REGION Network 198: Step[3048] : Pad Top Left/Right Vacc Off
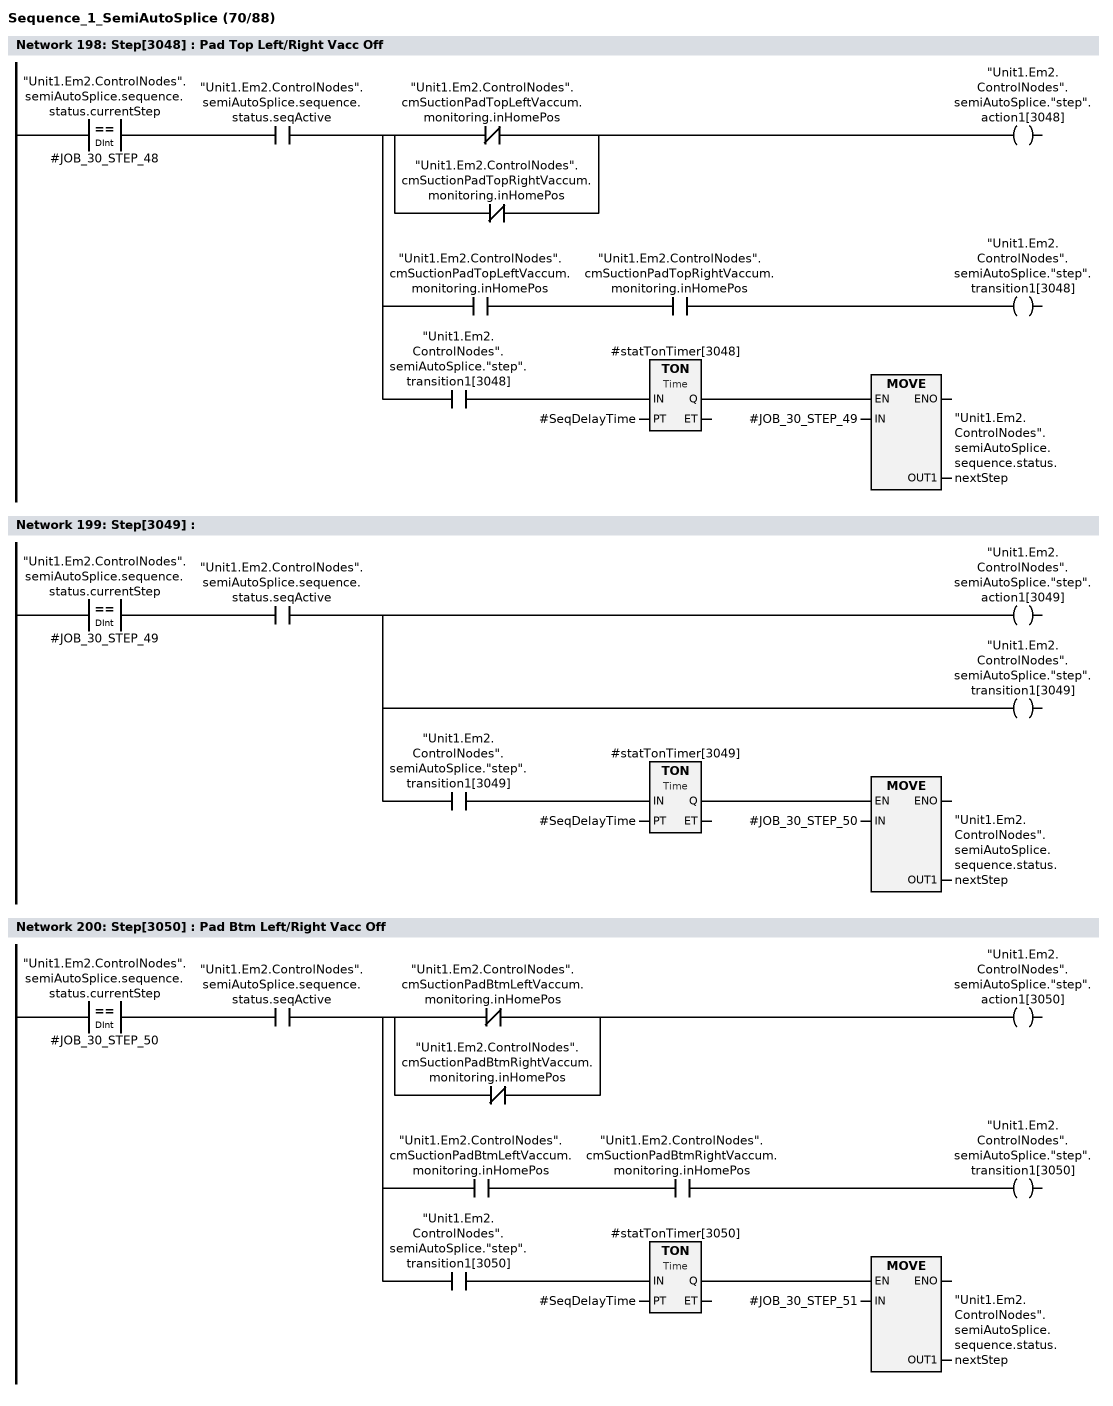
   RUNG wire#powerrail
      { S7_Templates := "SrcType := DInt" } EQ_Contact(in1 := "Unit1.Em2.ControlNodes".semiAutoSplice.sequence.status.currentStep, in2 := #JOB_30_STEP_48)
      Contact( "Unit1.Em2.ControlNodes".semiAutoSplice.sequence.status.seqActive )
      wire#w1
      I_Contact( "Unit1.Em2.ControlNodes".cmSuctionPadTopLeftVaccum.monitoring.inHomePos )
      wire#w2
      Coil( "Unit1.Em2.ControlNodes".semiAutoSplice."step".action1[3048] )
   END_RUNG
   RUNG wire#w1
      I_Contact( "Unit1.Em2.ControlNodes".cmSuctionPadTopRightVaccum.monitoring.inHomePos )
   END_RUNG wire#w2
   RUNG wire#w1
      Contact( "Unit1.Em2.ControlNodes".cmSuctionPadTopLeftVaccum.monitoring.inHomePos )
      Contact( "Unit1.Em2.ControlNodes".cmSuctionPadTopRightVaccum.monitoring.inHomePos )
      Coil( "Unit1.Em2.ControlNodes".semiAutoSplice."step".transition1[3048] )
   END_RUNG
   RUNG wire#w1
      Contact( "Unit1.Em2.ControlNodes".semiAutoSplice."step".transition1[3048] )
      { S7_Templates := "time_type := Time" } #statTonTimer[3048].TON(pt := #SeqDelayTime, et =>)
      Move(in := #JOB_30_STEP_49, out1 => "Unit1.Em2.ControlNodes".semiAutoSplice.sequence.status.nextStep)
   END_RUNG
   // the same network as SCL:
   #_w1 := ("Unit1.Em2.ControlNodes".semiAutoSplice.sequence.status.currentStep = #JOB_30_STEP_48) AND "Unit1.Em2.ControlNodes".semiAutoSplice.sequence.status.seqActive;
   "Unit1.Em2.ControlNodes".semiAutoSplice."step".action1[3048] := #_w1 AND (NOT "Unit1.Em2.ControlNodes".cmSuctionPadTopLeftVaccum.monitoring.inHomePos OR NOT "Unit1.Em2.ControlNodes".cmSuctionPadTopRightVaccum.monitoring.inHomePos);
   "Unit1.Em2.ControlNodes".semiAutoSplice."step".transition1[3048] := #_w1 AND "Unit1.Em2.ControlNodes".cmSuctionPadTopLeftVaccum.monitoring.inHomePos AND "Unit1.Em2.ControlNodes".cmSuctionPadTopRightVaccum.monitoring.inHomePos;
   #statTonTimer[3048].TON(IN := #_w1 AND "Unit1.Em2.ControlNodes".semiAutoSplice."step".transition1[3048],
                           PT := #SeqDelayTime);
   IF #statTonTimer[3048].Q THEN
       "Unit1.Em2.ControlNodes".semiAutoSplice.sequence.status.nextStep := #JOB_30_STEP_49;
   END_IF;
END_REGION

REGION Network 199: Step[3049] :
   RUNG wire#powerrail
      { S7_Templates := "SrcType := DInt" } EQ_Contact(in1 := "Unit1.Em2.ControlNodes".semiAutoSplice.sequence.status.currentStep, in2 := #JOB_30_STEP_49)
      Contact( "Unit1.Em2.ControlNodes".semiAutoSplice.sequence.status.seqActive )
      wire#w1
      Coil( "Unit1.Em2.ControlNodes".semiAutoSplice."step".action1[3049] )
   END_RUNG
   RUNG wire#w1
      Coil( "Unit1.Em2.ControlNodes".semiAutoSplice."step".transition1[3049] )
   END_RUNG
   RUNG wire#w1
      Contact( "Unit1.Em2.ControlNodes".semiAutoSplice."step".transition1[3049] )
      { S7_Templates := "time_type := Time" } #statTonTimer[3049].TON(pt := #SeqDelayTime, et =>)
      Move(in := #JOB_30_STEP_50, out1 => "Unit1.Em2.ControlNodes".semiAutoSplice.sequence.status.nextStep)
   END_RUNG
   // the same network as SCL:
   "Unit1.Em2.ControlNodes".semiAutoSplice."step".action1[3049] := ("Unit1.Em2.ControlNodes".semiAutoSplice.sequence.status.currentStep = #JOB_30_STEP_49) AND "Unit1.Em2.ControlNodes".semiAutoSplice.sequence.status.seqActive;
   "Unit1.Em2.ControlNodes".semiAutoSplice."step".transition1[3049] := ("Unit1.Em2.ControlNodes".semiAutoSplice.sequence.status.currentStep = #JOB_30_STEP_49) AND "Unit1.Em2.ControlNodes".semiAutoSplice.sequence.status.seqActive;
   #statTonTimer[3049].TON(IN := ("Unit1.Em2.ControlNodes".semiAutoSplice.sequence.status.currentStep = #JOB_30_STEP_49) AND "Unit1.Em2.ControlNodes".semiAutoSplice.sequence.status.seqActive AND "Unit1.Em2.ControlNodes".semiAutoSplice."step".transition1[3049],
                           PT := #SeqDelayTime);
   IF #statTonTimer[3049].Q THEN
       "Unit1.Em2.ControlNodes".semiAutoSplice.sequence.status.nextStep := #JOB_30_STEP_50;
   END_IF;
END_REGION

REGION Network 200: Step[3050] : Pad Btm Left/Right Vacc Off
   RUNG wire#powerrail
      { S7_Templates := "SrcType := DInt" } EQ_Contact(in1 := "Unit1.Em2.ControlNodes".semiAutoSplice.sequence.status.currentStep, in2 := #JOB_30_STEP_50)
      Contact( "Unit1.Em2.ControlNodes".semiAutoSplice.sequence.status.seqActive )
      wire#w1
      I_Contact( "Unit1.Em2.ControlNodes".cmSuctionPadBtmLeftVaccum.monitoring.inHomePos )
      wire#w2
      Coil( "Unit1.Em2.ControlNodes".semiAutoSplice."step".action1[3050] )
   END_RUNG
   RUNG wire#w1
      I_Contact( "Unit1.Em2.ControlNodes".cmSuctionPadBtmRightVaccum.monitoring.inHomePos )
   END_RUNG wire#w2
   RUNG wire#w1
      Contact( "Unit1.Em2.ControlNodes".cmSuctionPadBtmLeftVaccum.monitoring.inHomePos )
      Contact( "Unit1.Em2.ControlNodes".cmSuctionPadBtmRightVaccum.monitoring.inHomePos )
      Coil( "Unit1.Em2.ControlNodes".semiAutoSplice."step".transition1[3050] )
   END_RUNG
   RUNG wire#w1
      Contact( "Unit1.Em2.ControlNodes".semiAutoSplice."step".transition1[3050] )
      { S7_Templates := "time_type := Time" } #statTonTimer[3050].TON(pt := #SeqDelayTime, et =>)
      Move(in := #JOB_30_STEP_51, out1 => "Unit1.Em2.ControlNodes".semiAutoSplice.sequence.status.nextStep)
   END_RUNG
   // the same network as SCL:
   #_w1 := ("Unit1.Em2.ControlNodes".semiAutoSplice.sequence.status.currentStep = #JOB_30_STEP_50) AND "Unit1.Em2.ControlNodes".semiAutoSplice.sequence.status.seqActive;
   "Unit1.Em2.ControlNodes".semiAutoSplice."step".action1[3050] := #_w1 AND (NOT "Unit1.Em2.ControlNodes".cmSuctionPadBtmLeftVaccum.monitoring.inHomePos OR NOT "Unit1.Em2.ControlNodes".cmSuctionPadBtmRightVaccum.monitoring.inHomePos);
   "Unit1.Em2.ControlNodes".semiAutoSplice."step".transition1[3050] := #_w1 AND "Unit1.Em2.ControlNodes".cmSuctionPadBtmLeftVaccum.monitoring.inHomePos AND "Unit1.Em2.ControlNodes".cmSuctionPadBtmRightVaccum.monitoring.inHomePos;
   #statTonTimer[3050].TON(IN := #_w1 AND "Unit1.Em2.ControlNodes".semiAutoSplice."step".transition1[3050],
                           PT := #SeqDelayTime);
   IF #statTonTimer[3050].Q THEN
       "Unit1.Em2.ControlNodes".semiAutoSplice.sequence.status.nextStep := #JOB_30_STEP_51;
   END_IF;
END_REGION

REGION Network 201: Step[3051] :
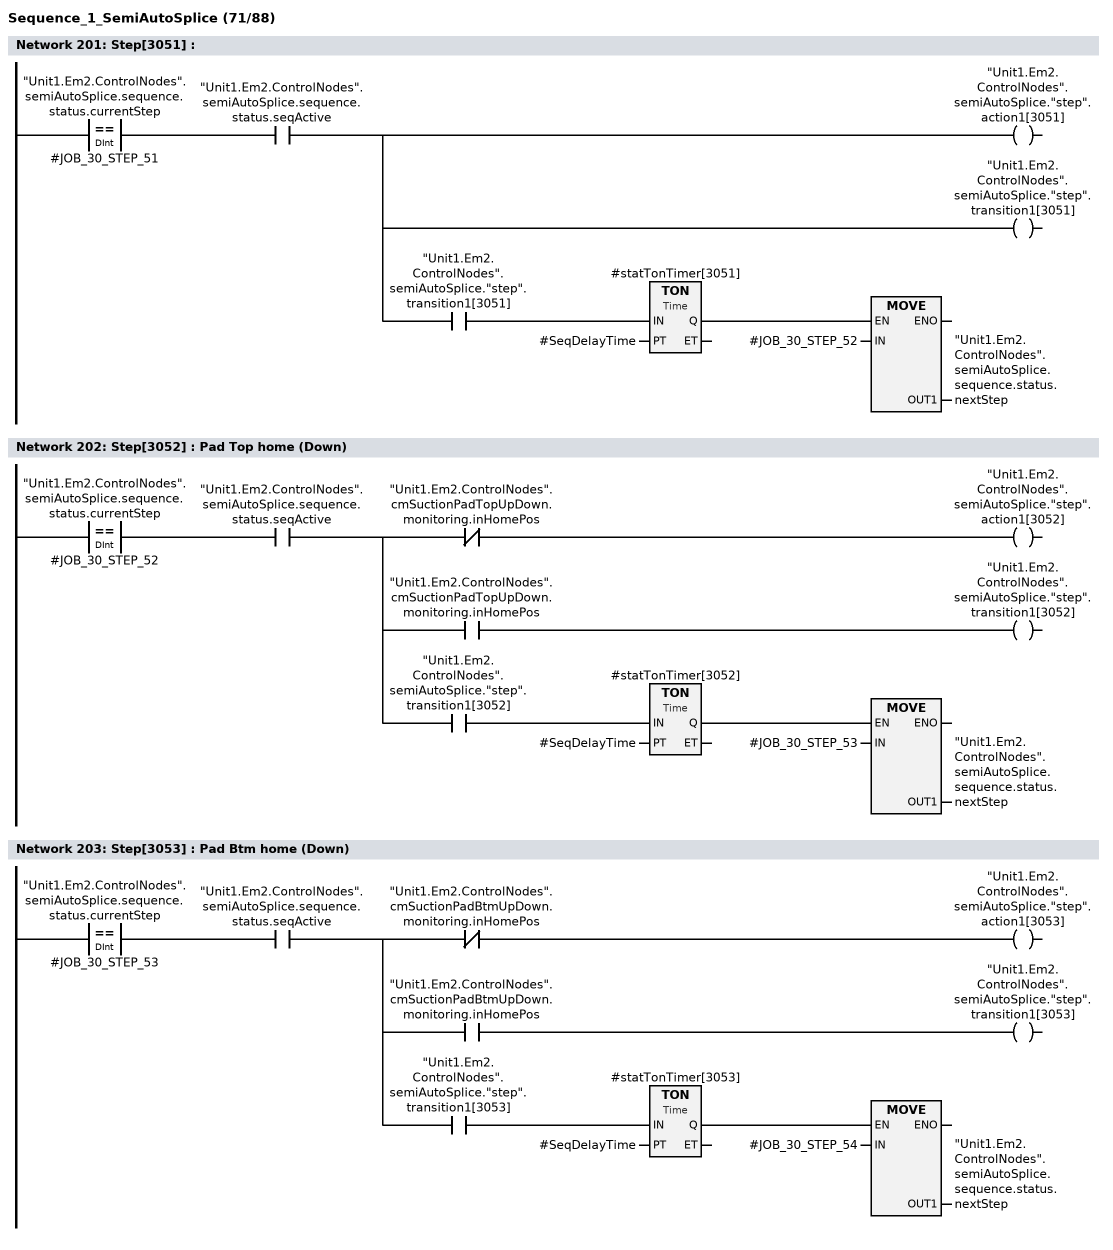
   RUNG wire#powerrail
      { S7_Templates := "SrcType := DInt" } EQ_Contact(in1 := "Unit1.Em2.ControlNodes".semiAutoSplice.sequence.status.currentStep, in2 := #JOB_30_STEP_51)
      Contact( "Unit1.Em2.ControlNodes".semiAutoSplice.sequence.status.seqActive )
      wire#w1
      Coil( "Unit1.Em2.ControlNodes".semiAutoSplice."step".action1[3051] )
   END_RUNG
   RUNG wire#w1
      Coil( "Unit1.Em2.ControlNodes".semiAutoSplice."step".transition1[3051] )
   END_RUNG
   RUNG wire#w1
      Contact( "Unit1.Em2.ControlNodes".semiAutoSplice."step".transition1[3051] )
      { S7_Templates := "time_type := Time" } #statTonTimer[3051].TON(pt := #SeqDelayTime, et =>)
      Move(in := #JOB_30_STEP_52, out1 => "Unit1.Em2.ControlNodes".semiAutoSplice.sequence.status.nextStep)
   END_RUNG
   // the same network as SCL:
   "Unit1.Em2.ControlNodes".semiAutoSplice."step".action1[3051] := ("Unit1.Em2.ControlNodes".semiAutoSplice.sequence.status.currentStep = #JOB_30_STEP_51) AND "Unit1.Em2.ControlNodes".semiAutoSplice.sequence.status.seqActive;
   "Unit1.Em2.ControlNodes".semiAutoSplice."step".transition1[3051] := ("Unit1.Em2.ControlNodes".semiAutoSplice.sequence.status.currentStep = #JOB_30_STEP_51) AND "Unit1.Em2.ControlNodes".semiAutoSplice.sequence.status.seqActive;
   #statTonTimer[3051].TON(IN := ("Unit1.Em2.ControlNodes".semiAutoSplice.sequence.status.currentStep = #JOB_30_STEP_51) AND "Unit1.Em2.ControlNodes".semiAutoSplice.sequence.status.seqActive AND "Unit1.Em2.ControlNodes".semiAutoSplice."step".transition1[3051],
                           PT := #SeqDelayTime);
   IF #statTonTimer[3051].Q THEN
       "Unit1.Em2.ControlNodes".semiAutoSplice.sequence.status.nextStep := #JOB_30_STEP_52;
   END_IF;
END_REGION

REGION Network 202: Step[3052] : Pad Top home (Down)
   RUNG wire#powerrail
      { S7_Templates := "SrcType := DInt" } EQ_Contact(in1 := "Unit1.Em2.ControlNodes".semiAutoSplice.sequence.status.currentStep, in2 := #JOB_30_STEP_52)
      Contact( "Unit1.Em2.ControlNodes".semiAutoSplice.sequence.status.seqActive )
      wire#w1
      I_Contact( "Unit1.Em2.ControlNodes".cmSuctionPadTopUpDown.monitoring.inHomePos )
      Coil( "Unit1.Em2.ControlNodes".semiAutoSplice."step".action1[3052] )
   END_RUNG
   RUNG wire#w1
      Contact( "Unit1.Em2.ControlNodes".cmSuctionPadTopUpDown.monitoring.inHomePos )
      Coil( "Unit1.Em2.ControlNodes".semiAutoSplice."step".transition1[3052] )
   END_RUNG
   RUNG wire#w1
      Contact( "Unit1.Em2.ControlNodes".semiAutoSplice."step".transition1[3052] )
      { S7_Templates := "time_type := Time" } #statTonTimer[3052].TON(pt := #SeqDelayTime, et =>)
      Move(in := #JOB_30_STEP_53, out1 => "Unit1.Em2.ControlNodes".semiAutoSplice.sequence.status.nextStep)
   END_RUNG
   // the same network as SCL:
   #_w1 := ("Unit1.Em2.ControlNodes".semiAutoSplice.sequence.status.currentStep = #JOB_30_STEP_52) AND "Unit1.Em2.ControlNodes".semiAutoSplice.sequence.status.seqActive;
   "Unit1.Em2.ControlNodes".semiAutoSplice."step".action1[3052] := #_w1 AND NOT "Unit1.Em2.ControlNodes".cmSuctionPadTopUpDown.monitoring.inHomePos;
   "Unit1.Em2.ControlNodes".semiAutoSplice."step".transition1[3052] := #_w1 AND "Unit1.Em2.ControlNodes".cmSuctionPadTopUpDown.monitoring.inHomePos;
   #statTonTimer[3052].TON(IN := #_w1 AND "Unit1.Em2.ControlNodes".semiAutoSplice."step".transition1[3052],
                           PT := #SeqDelayTime);
   IF #statTonTimer[3052].Q THEN
       "Unit1.Em2.ControlNodes".semiAutoSplice.sequence.status.nextStep := #JOB_30_STEP_53;
   END_IF;
END_REGION

REGION Network 203: Step[3053] : Pad Btm home (Down)
   RUNG wire#powerrail
      { S7_Templates := "SrcType := DInt" } EQ_Contact(in1 := "Unit1.Em2.ControlNodes".semiAutoSplice.sequence.status.currentStep, in2 := #JOB_30_STEP_53)
      Contact( "Unit1.Em2.ControlNodes".semiAutoSplice.sequence.status.seqActive )
      wire#w1
      I_Contact( "Unit1.Em2.ControlNodes".cmSuctionPadBtmUpDown.monitoring.inHomePos )
      Coil( "Unit1.Em2.ControlNodes".semiAutoSplice."step".action1[3053] )
   END_RUNG
   RUNG wire#w1
      Contact( "Unit1.Em2.ControlNodes".cmSuctionPadBtmUpDown.monitoring.inHomePos )
      Coil( "Unit1.Em2.ControlNodes".semiAutoSplice."step".transition1[3053] )
   END_RUNG
   RUNG wire#w1
      Contact( "Unit1.Em2.ControlNodes".semiAutoSplice."step".transition1[3053] )
      { S7_Templates := "time_type := Time" } #statTonTimer[3053].TON(pt := #SeqDelayTime, et =>)
      Move(in := #JOB_30_STEP_54, out1 => "Unit1.Em2.ControlNodes".semiAutoSplice.sequence.status.nextStep)
   END_RUNG
   // the same network as SCL:
   #_w1 := ("Unit1.Em2.ControlNodes".semiAutoSplice.sequence.status.currentStep = #JOB_30_STEP_53) AND "Unit1.Em2.ControlNodes".semiAutoSplice.sequence.status.seqActive;
   "Unit1.Em2.ControlNodes".semiAutoSplice."step".action1[3053] := #_w1 AND NOT "Unit1.Em2.ControlNodes".cmSuctionPadBtmUpDown.monitoring.inHomePos;
   "Unit1.Em2.ControlNodes".semiAutoSplice."step".transition1[3053] := #_w1 AND "Unit1.Em2.ControlNodes".cmSuctionPadBtmUpDown.monitoring.inHomePos;
   #statTonTimer[3053].TON(IN := #_w1 AND "Unit1.Em2.ControlNodes".semiAutoSplice."step".transition1[3053],
                           PT := #SeqDelayTime);
   IF #statTonTimer[3053].Q THEN
       "Unit1.Em2.ControlNodes".semiAutoSplice.sequence.status.nextStep := #JOB_30_STEP_54;
   END_IF;
END_REGION

REGION Network 204: Step[3054] :
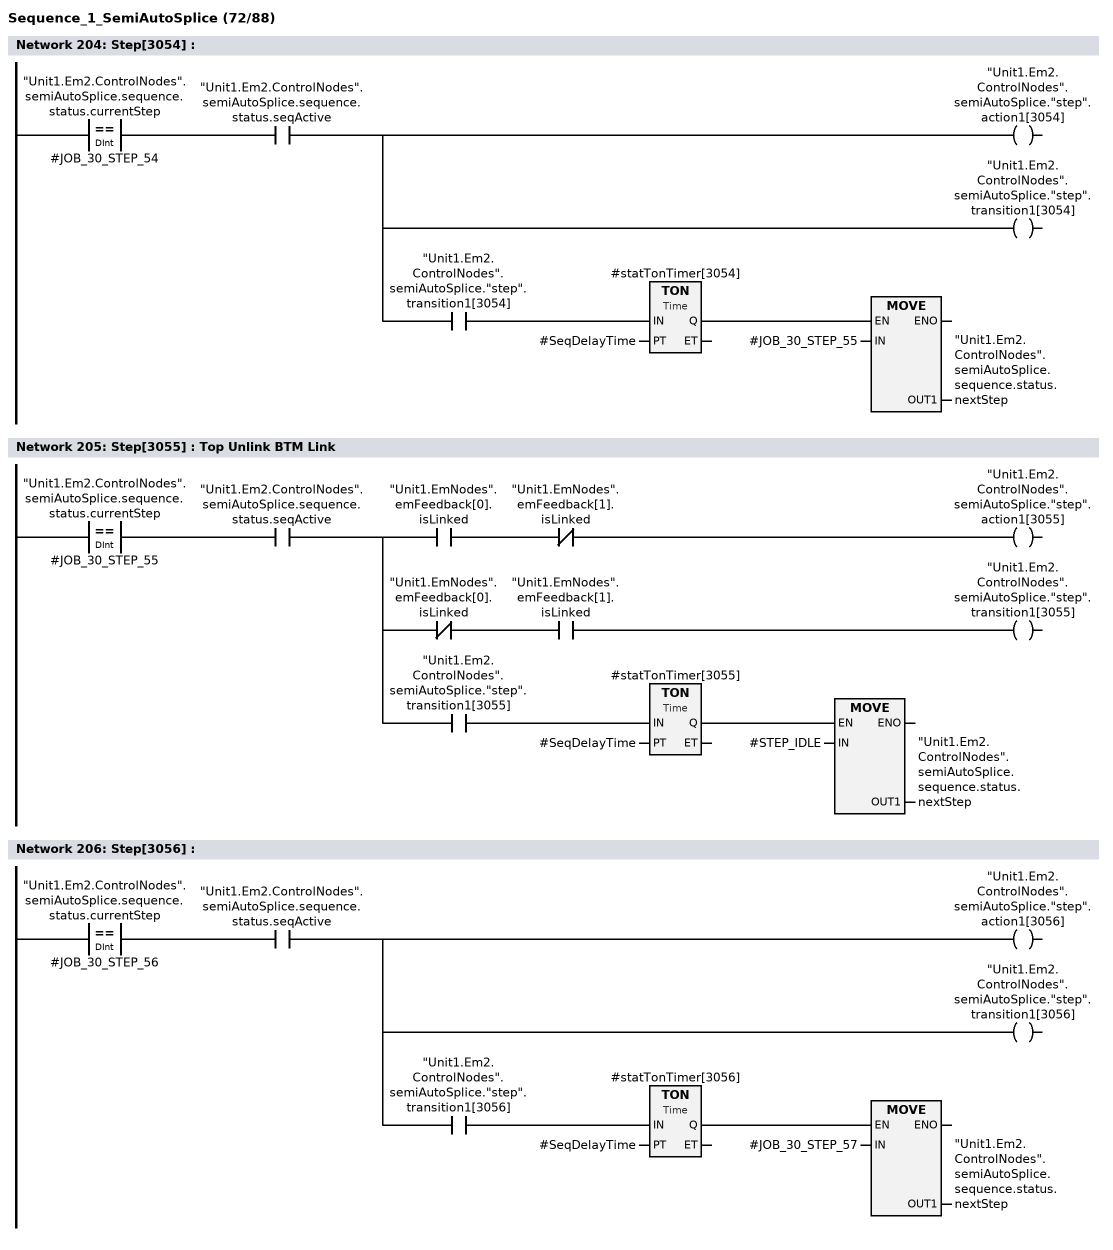
   RUNG wire#powerrail
      { S7_Templates := "SrcType := DInt" } EQ_Contact(in1 := "Unit1.Em2.ControlNodes".semiAutoSplice.sequence.status.currentStep, in2 := #JOB_30_STEP_54)
      Contact( "Unit1.Em2.ControlNodes".semiAutoSplice.sequence.status.seqActive )
      wire#w1
      Coil( "Unit1.Em2.ControlNodes".semiAutoSplice."step".action1[3054] )
   END_RUNG
   RUNG wire#w1
      Coil( "Unit1.Em2.ControlNodes".semiAutoSplice."step".transition1[3054] )
   END_RUNG
   RUNG wire#w1
      Contact( "Unit1.Em2.ControlNodes".semiAutoSplice."step".transition1[3054] )
      { S7_Templates := "time_type := Time" } #statTonTimer[3054].TON(pt := #SeqDelayTime, et =>)
      Move(in := #JOB_30_STEP_55, out1 => "Unit1.Em2.ControlNodes".semiAutoSplice.sequence.status.nextStep)
   END_RUNG
   // the same network as SCL:
   "Unit1.Em2.ControlNodes".semiAutoSplice."step".action1[3054] := ("Unit1.Em2.ControlNodes".semiAutoSplice.sequence.status.currentStep = #JOB_30_STEP_54) AND "Unit1.Em2.ControlNodes".semiAutoSplice.sequence.status.seqActive;
   "Unit1.Em2.ControlNodes".semiAutoSplice."step".transition1[3054] := ("Unit1.Em2.ControlNodes".semiAutoSplice.sequence.status.currentStep = #JOB_30_STEP_54) AND "Unit1.Em2.ControlNodes".semiAutoSplice.sequence.status.seqActive;
   #statTonTimer[3054].TON(IN := ("Unit1.Em2.ControlNodes".semiAutoSplice.sequence.status.currentStep = #JOB_30_STEP_54) AND "Unit1.Em2.ControlNodes".semiAutoSplice.sequence.status.seqActive AND "Unit1.Em2.ControlNodes".semiAutoSplice."step".transition1[3054],
                           PT := #SeqDelayTime);
   IF #statTonTimer[3054].Q THEN
       "Unit1.Em2.ControlNodes".semiAutoSplice.sequence.status.nextStep := #JOB_30_STEP_55;
   END_IF;
END_REGION

REGION Network 205: Step[3055] : Top Unlink BTM Link
   RUNG wire#powerrail
      { S7_Templates := "SrcType := DInt" } EQ_Contact(in1 := "Unit1.Em2.ControlNodes".semiAutoSplice.sequence.status.currentStep, in2 := #JOB_30_STEP_55)
      Contact( "Unit1.Em2.ControlNodes".semiAutoSplice.sequence.status.seqActive )
      wire#w1
      Contact( "Unit1.EmNodes".emFeedback[0].isLinked )
      I_Contact( "Unit1.EmNodes".emFeedback[1].isLinked )
      Coil( "Unit1.Em2.ControlNodes".semiAutoSplice."step".action1[3055] )
   END_RUNG
   RUNG wire#w1
      I_Contact( "Unit1.EmNodes".emFeedback[0].isLinked )
      Contact( "Unit1.EmNodes".emFeedback[1].isLinked )
      Coil( "Unit1.Em2.ControlNodes".semiAutoSplice."step".transition1[3055] )
   END_RUNG
   RUNG wire#w1
      Contact( "Unit1.Em2.ControlNodes".semiAutoSplice."step".transition1[3055] )
      { S7_Templates := "time_type := Time" } #statTonTimer[3055].TON(pt := #SeqDelayTime, et =>)
      Move(in := #STEP_IDLE, out1 => "Unit1.Em2.ControlNodes".semiAutoSplice.sequence.status.nextStep)
   END_RUNG
   // the same network as SCL:
   #_w1 := ("Unit1.Em2.ControlNodes".semiAutoSplice.sequence.status.currentStep = #JOB_30_STEP_55) AND "Unit1.Em2.ControlNodes".semiAutoSplice.sequence.status.seqActive;
   "Unit1.Em2.ControlNodes".semiAutoSplice."step".action1[3055] := #_w1 AND "Unit1.EmNodes".emFeedback[0].isLinked AND NOT "Unit1.EmNodes".emFeedback[1].isLinked;
   "Unit1.Em2.ControlNodes".semiAutoSplice."step".transition1[3055] := #_w1 AND NOT "Unit1.EmNodes".emFeedback[0].isLinked AND "Unit1.EmNodes".emFeedback[1].isLinked;
   #statTonTimer[3055].TON(IN := #_w1 AND "Unit1.Em2.ControlNodes".semiAutoSplice."step".transition1[3055],
                           PT := #SeqDelayTime);
   IF #statTonTimer[3055].Q THEN
       "Unit1.Em2.ControlNodes".semiAutoSplice.sequence.status.nextStep := #STEP_IDLE;
   END_IF;
END_REGION

REGION Network 206: Step[3056] :
   RUNG wire#powerrail
      { S7_Templates := "SrcType := DInt" } EQ_Contact(in1 := "Unit1.Em2.ControlNodes".semiAutoSplice.sequence.status.currentStep, in2 := #JOB_30_STEP_56)
      Contact( "Unit1.Em2.ControlNodes".semiAutoSplice.sequence.status.seqActive )
      wire#w1
      Coil( "Unit1.Em2.ControlNodes".semiAutoSplice."step".action1[3056] )
   END_RUNG
   RUNG wire#w1
      Coil( "Unit1.Em2.ControlNodes".semiAutoSplice."step".transition1[3056] )
   END_RUNG
   RUNG wire#w1
      Contact( "Unit1.Em2.ControlNodes".semiAutoSplice."step".transition1[3056] )
      { S7_Templates := "time_type := Time" } #statTonTimer[3056].TON(pt := #SeqDelayTime, et =>)
      Move(in := #JOB_30_STEP_57, out1 => "Unit1.Em2.ControlNodes".semiAutoSplice.sequence.status.nextStep)
   END_RUNG
   // the same network as SCL:
   "Unit1.Em2.ControlNodes".semiAutoSplice."step".action1[3056] := ("Unit1.Em2.ControlNodes".semiAutoSplice.sequence.status.currentStep = #JOB_30_STEP_56) AND "Unit1.Em2.ControlNodes".semiAutoSplice.sequence.status.seqActive;
   "Unit1.Em2.ControlNodes".semiAutoSplice."step".transition1[3056] := ("Unit1.Em2.ControlNodes".semiAutoSplice.sequence.status.currentStep = #JOB_30_STEP_56) AND "Unit1.Em2.ControlNodes".semiAutoSplice.sequence.status.seqActive;
   #statTonTimer[3056].TON(IN := ("Unit1.Em2.ControlNodes".semiAutoSplice.sequence.status.currentStep = #JOB_30_STEP_56) AND "Unit1.Em2.ControlNodes".semiAutoSplice.sequence.status.seqActive AND "Unit1.Em2.ControlNodes".semiAutoSplice."step".transition1[3056],
                           PT := #SeqDelayTime);
   IF #statTonTimer[3056].Q THEN
       "Unit1.Em2.ControlNodes".semiAutoSplice.sequence.status.nextStep := #JOB_30_STEP_57;
   END_IF;
END_REGION

REGION Network 207: Step[3057] : BTM Link BTM Left/right Vacc Off (Top Left/Right Vacc On)
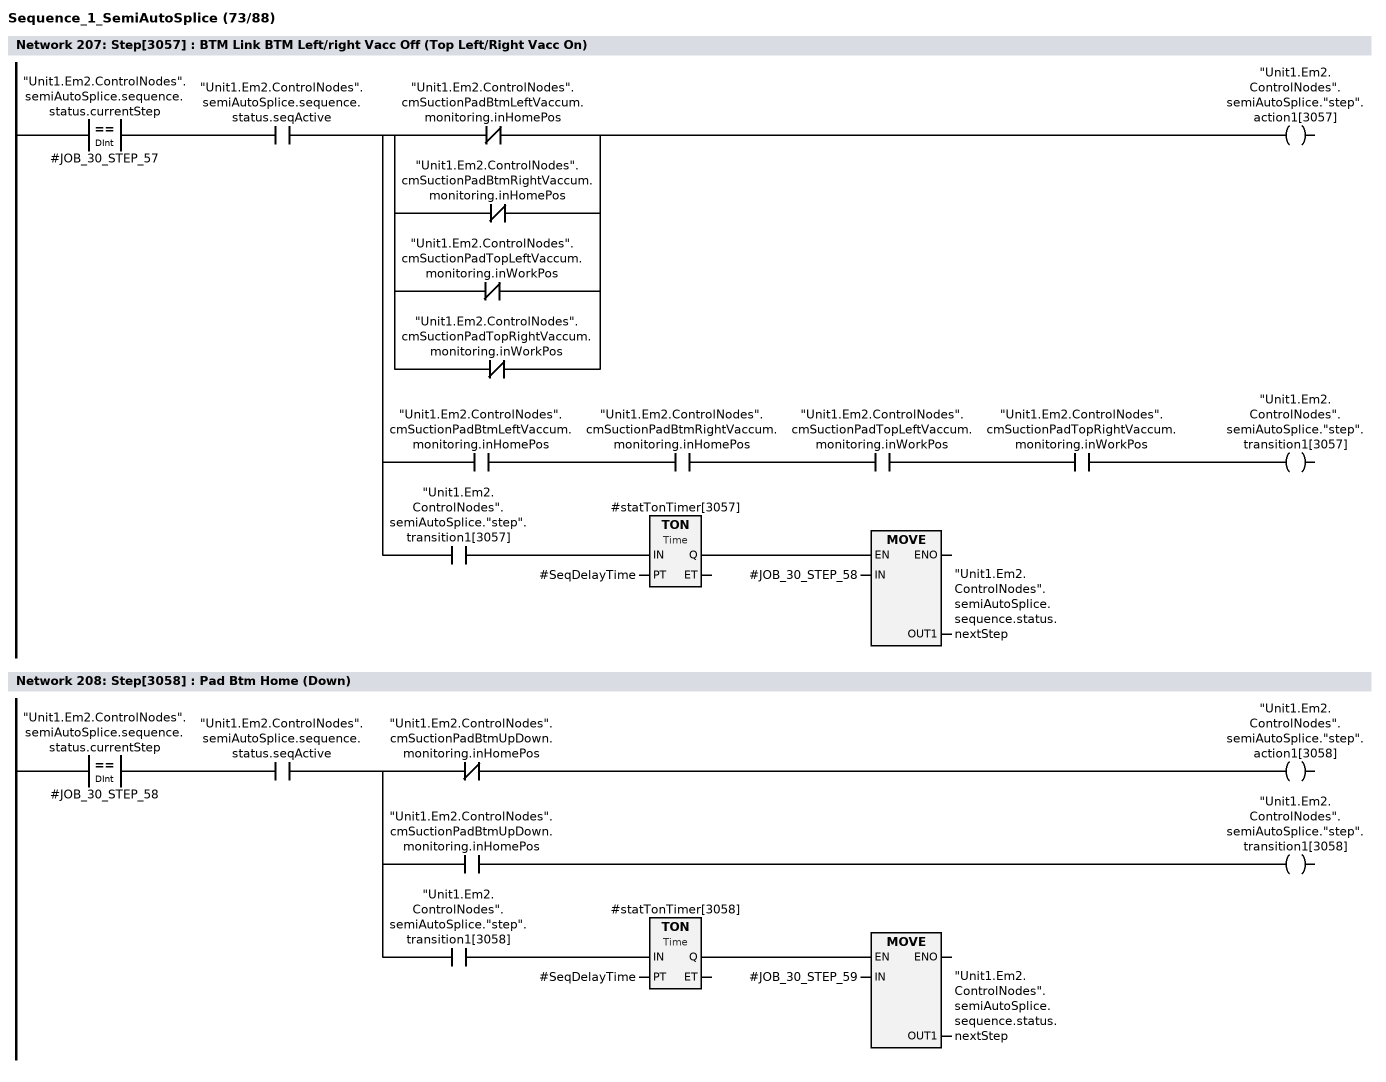
   RUNG wire#powerrail
      { S7_Templates := "SrcType := DInt" } EQ_Contact(in1 := "Unit1.Em2.ControlNodes".semiAutoSplice.sequence.status.currentStep, in2 := #JOB_30_STEP_57)
      Contact( "Unit1.Em2.ControlNodes".semiAutoSplice.sequence.status.seqActive )
      wire#w1
      I_Contact( "Unit1.Em2.ControlNodes".cmSuctionPadBtmLeftVaccum.monitoring.inHomePos )
      wire#w2
      Coil( "Unit1.Em2.ControlNodes".semiAutoSplice."step".action1[3057] )
   END_RUNG
   RUNG wire#w1
      I_Contact( "Unit1.Em2.ControlNodes".cmSuctionPadBtmRightVaccum.monitoring.inHomePos )
   END_RUNG wire#w2
   RUNG wire#w1
      I_Contact( "Unit1.Em2.ControlNodes".cmSuctionPadTopLeftVaccum.monitoring.inWorkPos )
   END_RUNG wire#w2
   RUNG wire#w1
      I_Contact( "Unit1.Em2.ControlNodes".cmSuctionPadTopRightVaccum.monitoring.inWorkPos )
   END_RUNG wire#w2
   RUNG wire#w1
      Contact( "Unit1.Em2.ControlNodes".cmSuctionPadBtmLeftVaccum.monitoring.inHomePos )
      Contact( "Unit1.Em2.ControlNodes".cmSuctionPadBtmRightVaccum.monitoring.inHomePos )
      Contact( "Unit1.Em2.ControlNodes".cmSuctionPadTopLeftVaccum.monitoring.inWorkPos )
      Contact( "Unit1.Em2.ControlNodes".cmSuctionPadTopRightVaccum.monitoring.inWorkPos )
      Coil( "Unit1.Em2.ControlNodes".semiAutoSplice."step".transition1[3057] )
   END_RUNG
   RUNG wire#w1
      Contact( "Unit1.Em2.ControlNodes".semiAutoSplice."step".transition1[3057] )
      { S7_Templates := "time_type := Time" } #statTonTimer[3057].TON(pt := #SeqDelayTime, et =>)
      Move(in := #JOB_30_STEP_58, out1 => "Unit1.Em2.ControlNodes".semiAutoSplice.sequence.status.nextStep)
   END_RUNG
   // the same network as SCL:
   #_w1 := ("Unit1.Em2.ControlNodes".semiAutoSplice.sequence.status.currentStep = #JOB_30_STEP_57) AND "Unit1.Em2.ControlNodes".semiAutoSplice.sequence.status.seqActive;
   "Unit1.Em2.ControlNodes".semiAutoSplice."step".action1[3057] := #_w1 AND (NOT "Unit1.Em2.ControlNodes".cmSuctionPadBtmLeftVaccum.monitoring.inHomePos OR NOT "Unit1.Em2.ControlNodes".cmSuctionPadBtmRightVaccum.monitoring.inHomePos OR NOT "Unit1.Em2.ControlNodes".cmSuctionPadTopLeftVaccum.monitoring.inWorkPos OR NOT "Unit1.Em2.ControlNodes".cmSuctionPadTopRightVaccum.monitoring.inWorkPos);
   "Unit1.Em2.ControlNodes".semiAutoSplice."step".transition1[3057] := #_w1 AND "Unit1.Em2.ControlNodes".cmSuctionPadBtmLeftVaccum.monitoring.inHomePos AND "Unit1.Em2.ControlNodes".cmSuctionPadBtmRightVaccum.monitoring.inHomePos AND "Unit1.Em2.ControlNodes".cmSuctionPadTopLeftVaccum.monitoring.inWorkPos AND "Unit1.Em2.ControlNodes".cmSuctionPadTopRightVaccum.monitoring.inWorkPos;
   #statTonTimer[3057].TON(IN := #_w1 AND "Unit1.Em2.ControlNodes".semiAutoSplice."step".transition1[3057],
                           PT := #SeqDelayTime);
   IF #statTonTimer[3057].Q THEN
       "Unit1.Em2.ControlNodes".semiAutoSplice.sequence.status.nextStep := #JOB_30_STEP_58;
   END_IF;
END_REGION

REGION Network 208: Step[3058] : Pad Btm Home (Down)
   RUNG wire#powerrail
      { S7_Templates := "SrcType := DInt" } EQ_Contact(in1 := "Unit1.Em2.ControlNodes".semiAutoSplice.sequence.status.currentStep, in2 := #JOB_30_STEP_58)
      Contact( "Unit1.Em2.ControlNodes".semiAutoSplice.sequence.status.seqActive )
      wire#w1
      I_Contact( "Unit1.Em2.ControlNodes".cmSuctionPadBtmUpDown.monitoring.inHomePos )
      Coil( "Unit1.Em2.ControlNodes".semiAutoSplice."step".action1[3058] )
   END_RUNG
   RUNG wire#w1
      Contact( "Unit1.Em2.ControlNodes".cmSuctionPadBtmUpDown.monitoring.inHomePos )
      Coil( "Unit1.Em2.ControlNodes".semiAutoSplice."step".transition1[3058] )
   END_RUNG
   RUNG wire#w1
      Contact( "Unit1.Em2.ControlNodes".semiAutoSplice."step".transition1[3058] )
      { S7_Templates := "time_type := Time" } #statTonTimer[3058].TON(pt := #SeqDelayTime, et =>)
      Move(in := #JOB_30_STEP_59, out1 => "Unit1.Em2.ControlNodes".semiAutoSplice.sequence.status.nextStep)
   END_RUNG
   // the same network as SCL:
   #_w1 := ("Unit1.Em2.ControlNodes".semiAutoSplice.sequence.status.currentStep = #JOB_30_STEP_58) AND "Unit1.Em2.ControlNodes".semiAutoSplice.sequence.status.seqActive;
   "Unit1.Em2.ControlNodes".semiAutoSplice."step".action1[3058] := #_w1 AND NOT "Unit1.Em2.ControlNodes".cmSuctionPadBtmUpDown.monitoring.inHomePos;
   "Unit1.Em2.ControlNodes".semiAutoSplice."step".transition1[3058] := #_w1 AND "Unit1.Em2.ControlNodes".cmSuctionPadBtmUpDown.monitoring.inHomePos;
   #statTonTimer[3058].TON(IN := #_w1 AND "Unit1.Em2.ControlNodes".semiAutoSplice."step".transition1[3058],
                           PT := #SeqDelayTime);
   IF #statTonTimer[3058].Q THEN
       "Unit1.Em2.ControlNodes".semiAutoSplice.sequence.status.nextStep := #JOB_30_STEP_59;
   END_IF;
END_REGION

REGION Network 209: Step[3059] :
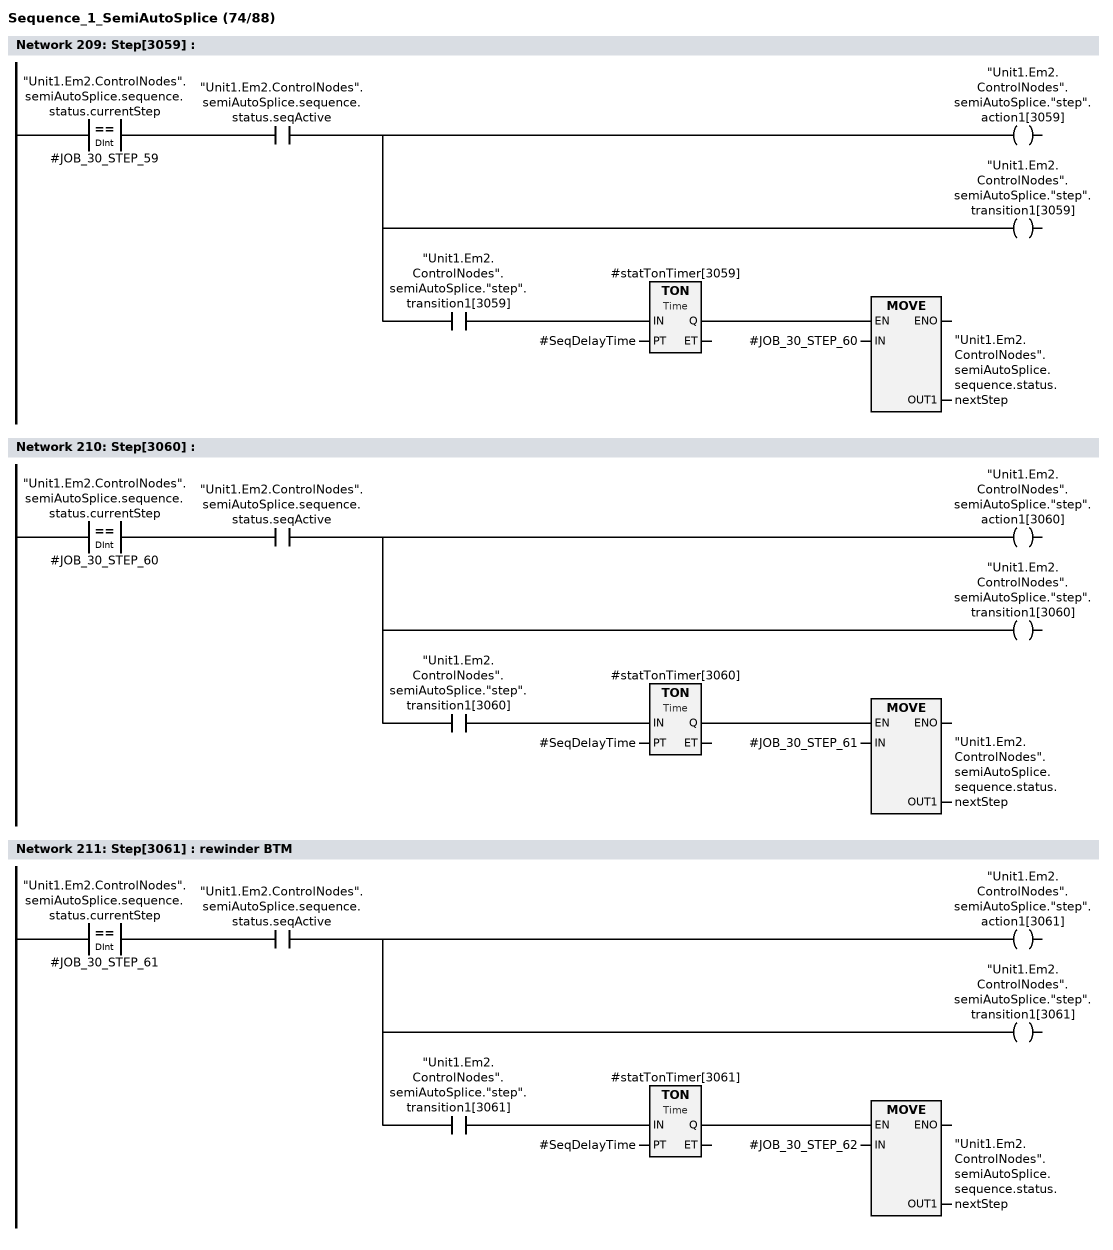
   RUNG wire#powerrail
      { S7_Templates := "SrcType := DInt" } EQ_Contact(in1 := "Unit1.Em2.ControlNodes".semiAutoSplice.sequence.status.currentStep, in2 := #JOB_30_STEP_59)
      Contact( "Unit1.Em2.ControlNodes".semiAutoSplice.sequence.status.seqActive )
      wire#w1
      Coil( "Unit1.Em2.ControlNodes".semiAutoSplice."step".action1[3059] )
   END_RUNG
   RUNG wire#w1
      Coil( "Unit1.Em2.ControlNodes".semiAutoSplice."step".transition1[3059] )
   END_RUNG
   RUNG wire#w1
      Contact( "Unit1.Em2.ControlNodes".semiAutoSplice."step".transition1[3059] )
      { S7_Templates := "time_type := Time" } #statTonTimer[3059].TON(pt := #SeqDelayTime, et =>)
      Move(in := #JOB_30_STEP_60, out1 => "Unit1.Em2.ControlNodes".semiAutoSplice.sequence.status.nextStep)
   END_RUNG
   // the same network as SCL:
   "Unit1.Em2.ControlNodes".semiAutoSplice."step".action1[3059] := ("Unit1.Em2.ControlNodes".semiAutoSplice.sequence.status.currentStep = #JOB_30_STEP_59) AND "Unit1.Em2.ControlNodes".semiAutoSplice.sequence.status.seqActive;
   "Unit1.Em2.ControlNodes".semiAutoSplice."step".transition1[3059] := ("Unit1.Em2.ControlNodes".semiAutoSplice.sequence.status.currentStep = #JOB_30_STEP_59) AND "Unit1.Em2.ControlNodes".semiAutoSplice.sequence.status.seqActive;
   #statTonTimer[3059].TON(IN := ("Unit1.Em2.ControlNodes".semiAutoSplice.sequence.status.currentStep = #JOB_30_STEP_59) AND "Unit1.Em2.ControlNodes".semiAutoSplice.sequence.status.seqActive AND "Unit1.Em2.ControlNodes".semiAutoSplice."step".transition1[3059],
                           PT := #SeqDelayTime);
   IF #statTonTimer[3059].Q THEN
       "Unit1.Em2.ControlNodes".semiAutoSplice.sequence.status.nextStep := #JOB_30_STEP_60;
   END_IF;
END_REGION

REGION Network 210: Step[3060] :
   RUNG wire#powerrail
      { S7_Templates := "SrcType := DInt" } EQ_Contact(in1 := "Unit1.Em2.ControlNodes".semiAutoSplice.sequence.status.currentStep, in2 := #JOB_30_STEP_60)
      Contact( "Unit1.Em2.ControlNodes".semiAutoSplice.sequence.status.seqActive )
      wire#w1
      Coil( "Unit1.Em2.ControlNodes".semiAutoSplice."step".action1[3060] )
   END_RUNG
   RUNG wire#w1
      Coil( "Unit1.Em2.ControlNodes".semiAutoSplice."step".transition1[3060] )
   END_RUNG
   RUNG wire#w1
      Contact( "Unit1.Em2.ControlNodes".semiAutoSplice."step".transition1[3060] )
      { S7_Templates := "time_type := Time" } #statTonTimer[3060].TON(pt := #SeqDelayTime, et =>)
      Move(in := #JOB_30_STEP_61, out1 => "Unit1.Em2.ControlNodes".semiAutoSplice.sequence.status.nextStep)
   END_RUNG
   // the same network as SCL:
   "Unit1.Em2.ControlNodes".semiAutoSplice."step".action1[3060] := ("Unit1.Em2.ControlNodes".semiAutoSplice.sequence.status.currentStep = #JOB_30_STEP_60) AND "Unit1.Em2.ControlNodes".semiAutoSplice.sequence.status.seqActive;
   "Unit1.Em2.ControlNodes".semiAutoSplice."step".transition1[3060] := ("Unit1.Em2.ControlNodes".semiAutoSplice.sequence.status.currentStep = #JOB_30_STEP_60) AND "Unit1.Em2.ControlNodes".semiAutoSplice.sequence.status.seqActive;
   #statTonTimer[3060].TON(IN := ("Unit1.Em2.ControlNodes".semiAutoSplice.sequence.status.currentStep = #JOB_30_STEP_60) AND "Unit1.Em2.ControlNodes".semiAutoSplice.sequence.status.seqActive AND "Unit1.Em2.ControlNodes".semiAutoSplice."step".transition1[3060],
                           PT := #SeqDelayTime);
   IF #statTonTimer[3060].Q THEN
       "Unit1.Em2.ControlNodes".semiAutoSplice.sequence.status.nextStep := #JOB_30_STEP_61;
   END_IF;
END_REGION

REGION Network 211: Step[3061] : rewinder BTM
   RUNG wire#powerrail
      { S7_Templates := "SrcType := DInt" } EQ_Contact(in1 := "Unit1.Em2.ControlNodes".semiAutoSplice.sequence.status.currentStep, in2 := #JOB_30_STEP_61)
      Contact( "Unit1.Em2.ControlNodes".semiAutoSplice.sequence.status.seqActive )
      wire#w1
      Coil( "Unit1.Em2.ControlNodes".semiAutoSplice."step".action1[3061] )
   END_RUNG
   RUNG wire#w1
      Coil( "Unit1.Em2.ControlNodes".semiAutoSplice."step".transition1[3061] )
   END_RUNG
   RUNG wire#w1
      Contact( "Unit1.Em2.ControlNodes".semiAutoSplice."step".transition1[3061] )
      { S7_Templates := "time_type := Time" } #statTonTimer[3061].TON(pt := #SeqDelayTime, et =>)
      Move(in := #JOB_30_STEP_62, out1 => "Unit1.Em2.ControlNodes".semiAutoSplice.sequence.status.nextStep)
   END_RUNG
   // the same network as SCL:
   "Unit1.Em2.ControlNodes".semiAutoSplice."step".action1[3061] := ("Unit1.Em2.ControlNodes".semiAutoSplice.sequence.status.currentStep = #JOB_30_STEP_61) AND "Unit1.Em2.ControlNodes".semiAutoSplice.sequence.status.seqActive;
   "Unit1.Em2.ControlNodes".semiAutoSplice."step".transition1[3061] := ("Unit1.Em2.ControlNodes".semiAutoSplice.sequence.status.currentStep = #JOB_30_STEP_61) AND "Unit1.Em2.ControlNodes".semiAutoSplice.sequence.status.seqActive;
   #statTonTimer[3061].TON(IN := ("Unit1.Em2.ControlNodes".semiAutoSplice.sequence.status.currentStep = #JOB_30_STEP_61) AND "Unit1.Em2.ControlNodes".semiAutoSplice.sequence.status.seqActive AND "Unit1.Em2.ControlNodes".semiAutoSplice."step".transition1[3061],
                           PT := #SeqDelayTime);
   IF #statTonTimer[3061].Q THEN
       "Unit1.Em2.ControlNodes".semiAutoSplice.sequence.status.nextStep := #JOB_30_STEP_62;
   END_IF;
END_REGION

REGION Network 212: Step[3062] :
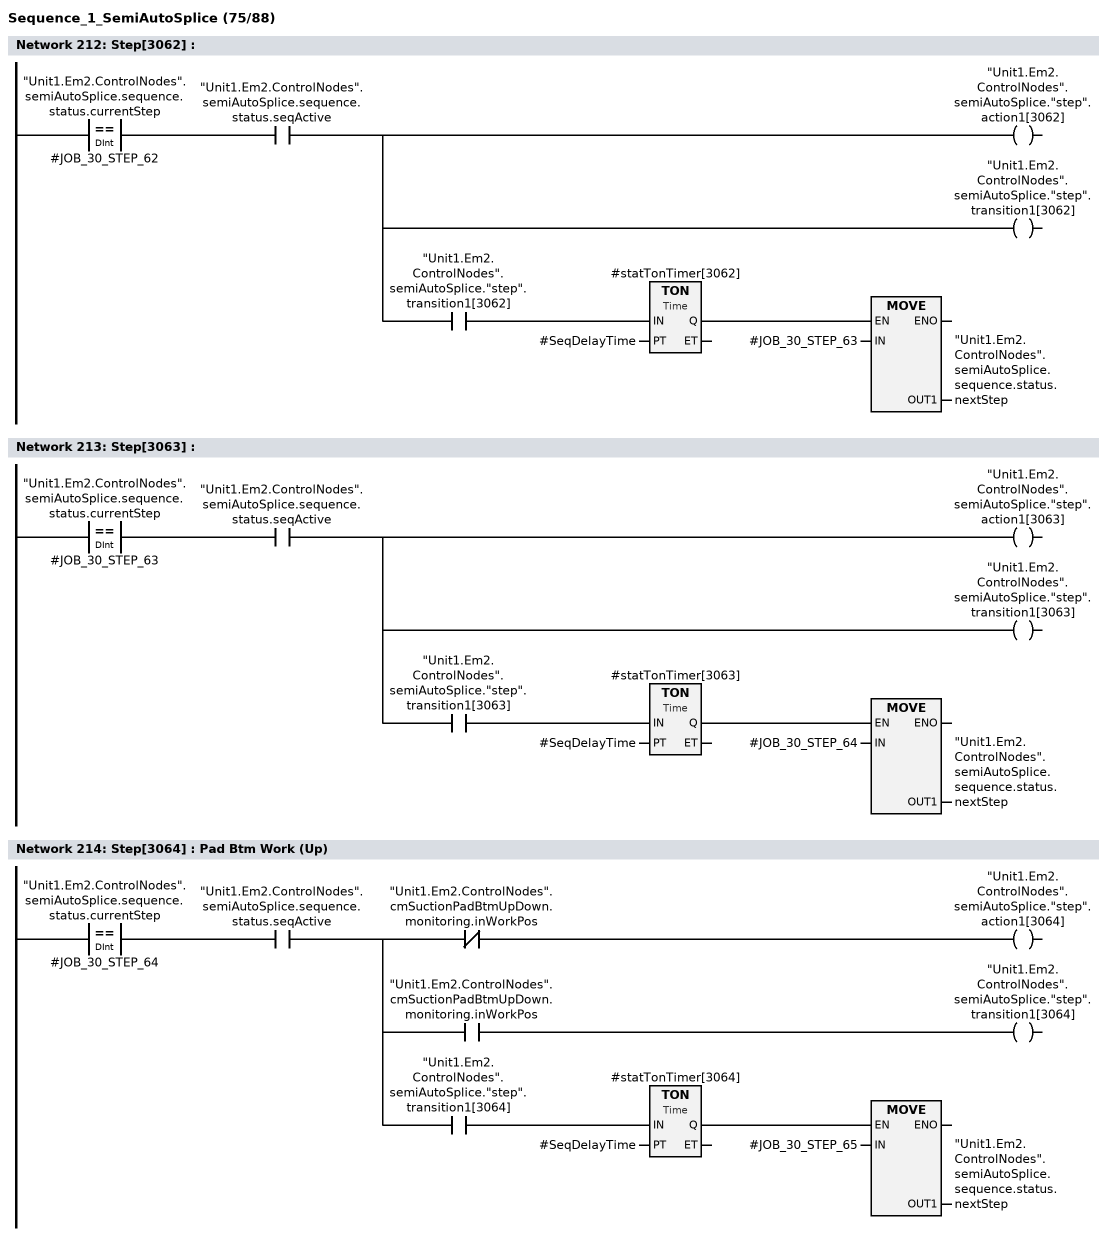
   RUNG wire#powerrail
      { S7_Templates := "SrcType := DInt" } EQ_Contact(in1 := "Unit1.Em2.ControlNodes".semiAutoSplice.sequence.status.currentStep, in2 := #JOB_30_STEP_62)
      Contact( "Unit1.Em2.ControlNodes".semiAutoSplice.sequence.status.seqActive )
      wire#w1
      Coil( "Unit1.Em2.ControlNodes".semiAutoSplice."step".action1[3062] )
   END_RUNG
   RUNG wire#w1
      Coil( "Unit1.Em2.ControlNodes".semiAutoSplice."step".transition1[3062] )
   END_RUNG
   RUNG wire#w1
      Contact( "Unit1.Em2.ControlNodes".semiAutoSplice."step".transition1[3062] )
      { S7_Templates := "time_type := Time" } #statTonTimer[3062].TON(pt := #SeqDelayTime, et =>)
      Move(in := #JOB_30_STEP_63, out1 => "Unit1.Em2.ControlNodes".semiAutoSplice.sequence.status.nextStep)
   END_RUNG
   // the same network as SCL:
   "Unit1.Em2.ControlNodes".semiAutoSplice."step".action1[3062] := ("Unit1.Em2.ControlNodes".semiAutoSplice.sequence.status.currentStep = #JOB_30_STEP_62) AND "Unit1.Em2.ControlNodes".semiAutoSplice.sequence.status.seqActive;
   "Unit1.Em2.ControlNodes".semiAutoSplice."step".transition1[3062] := ("Unit1.Em2.ControlNodes".semiAutoSplice.sequence.status.currentStep = #JOB_30_STEP_62) AND "Unit1.Em2.ControlNodes".semiAutoSplice.sequence.status.seqActive;
   #statTonTimer[3062].TON(IN := ("Unit1.Em2.ControlNodes".semiAutoSplice.sequence.status.currentStep = #JOB_30_STEP_62) AND "Unit1.Em2.ControlNodes".semiAutoSplice.sequence.status.seqActive AND "Unit1.Em2.ControlNodes".semiAutoSplice."step".transition1[3062],
                           PT := #SeqDelayTime);
   IF #statTonTimer[3062].Q THEN
       "Unit1.Em2.ControlNodes".semiAutoSplice.sequence.status.nextStep := #JOB_30_STEP_63;
   END_IF;
END_REGION

REGION Network 213: Step[3063] :
   RUNG wire#powerrail
      { S7_Templates := "SrcType := DInt" } EQ_Contact(in1 := "Unit1.Em2.ControlNodes".semiAutoSplice.sequence.status.currentStep, in2 := #JOB_30_STEP_63)
      Contact( "Unit1.Em2.ControlNodes".semiAutoSplice.sequence.status.seqActive )
      wire#w1
      Coil( "Unit1.Em2.ControlNodes".semiAutoSplice."step".action1[3063] )
   END_RUNG
   RUNG wire#w1
      Coil( "Unit1.Em2.ControlNodes".semiAutoSplice."step".transition1[3063] )
   END_RUNG
   RUNG wire#w1
      Contact( "Unit1.Em2.ControlNodes".semiAutoSplice."step".transition1[3063] )
      { S7_Templates := "time_type := Time" } #statTonTimer[3063].TON(pt := #SeqDelayTime, et =>)
      Move(in := #JOB_30_STEP_64, out1 => "Unit1.Em2.ControlNodes".semiAutoSplice.sequence.status.nextStep)
   END_RUNG
   // the same network as SCL:
   "Unit1.Em2.ControlNodes".semiAutoSplice."step".action1[3063] := ("Unit1.Em2.ControlNodes".semiAutoSplice.sequence.status.currentStep = #JOB_30_STEP_63) AND "Unit1.Em2.ControlNodes".semiAutoSplice.sequence.status.seqActive;
   "Unit1.Em2.ControlNodes".semiAutoSplice."step".transition1[3063] := ("Unit1.Em2.ControlNodes".semiAutoSplice.sequence.status.currentStep = #JOB_30_STEP_63) AND "Unit1.Em2.ControlNodes".semiAutoSplice.sequence.status.seqActive;
   #statTonTimer[3063].TON(IN := ("Unit1.Em2.ControlNodes".semiAutoSplice.sequence.status.currentStep = #JOB_30_STEP_63) AND "Unit1.Em2.ControlNodes".semiAutoSplice.sequence.status.seqActive AND "Unit1.Em2.ControlNodes".semiAutoSplice."step".transition1[3063],
                           PT := #SeqDelayTime);
   IF #statTonTimer[3063].Q THEN
       "Unit1.Em2.ControlNodes".semiAutoSplice.sequence.status.nextStep := #JOB_30_STEP_64;
   END_IF;
END_REGION

REGION Network 214: Step[3064] : Pad Btm Work (Up)
   RUNG wire#powerrail
      { S7_Templates := "SrcType := DInt" } EQ_Contact(in1 := "Unit1.Em2.ControlNodes".semiAutoSplice.sequence.status.currentStep, in2 := #JOB_30_STEP_64)
      Contact( "Unit1.Em2.ControlNodes".semiAutoSplice.sequence.status.seqActive )
      wire#w1
      I_Contact( "Unit1.Em2.ControlNodes".cmSuctionPadBtmUpDown.monitoring.inWorkPos )
      Coil( "Unit1.Em2.ControlNodes".semiAutoSplice."step".action1[3064] )
   END_RUNG
   RUNG wire#w1
      Contact( "Unit1.Em2.ControlNodes".cmSuctionPadBtmUpDown.monitoring.inWorkPos )
      Coil( "Unit1.Em2.ControlNodes".semiAutoSplice."step".transition1[3064] )
   END_RUNG
   RUNG wire#w1
      Contact( "Unit1.Em2.ControlNodes".semiAutoSplice."step".transition1[3064] )
      { S7_Templates := "time_type := Time" } #statTonTimer[3064].TON(pt := #SeqDelayTime, et =>)
      Move(in := #JOB_30_STEP_65, out1 => "Unit1.Em2.ControlNodes".semiAutoSplice.sequence.status.nextStep)
   END_RUNG
   // the same network as SCL:
   #_w1 := ("Unit1.Em2.ControlNodes".semiAutoSplice.sequence.status.currentStep = #JOB_30_STEP_64) AND "Unit1.Em2.ControlNodes".semiAutoSplice.sequence.status.seqActive;
   "Unit1.Em2.ControlNodes".semiAutoSplice."step".action1[3064] := #_w1 AND NOT "Unit1.Em2.ControlNodes".cmSuctionPadBtmUpDown.monitoring.inWorkPos;
   "Unit1.Em2.ControlNodes".semiAutoSplice."step".transition1[3064] := #_w1 AND "Unit1.Em2.ControlNodes".cmSuctionPadBtmUpDown.monitoring.inWorkPos;
   #statTonTimer[3064].TON(IN := #_w1 AND "Unit1.Em2.ControlNodes".semiAutoSplice."step".transition1[3064],
                           PT := #SeqDelayTime);
   IF #statTonTimer[3064].Q THEN
       "Unit1.Em2.ControlNodes".semiAutoSplice.sequence.status.nextStep := #JOB_30_STEP_65;
   END_IF;
END_REGION

REGION Network 215: Step[3065] :
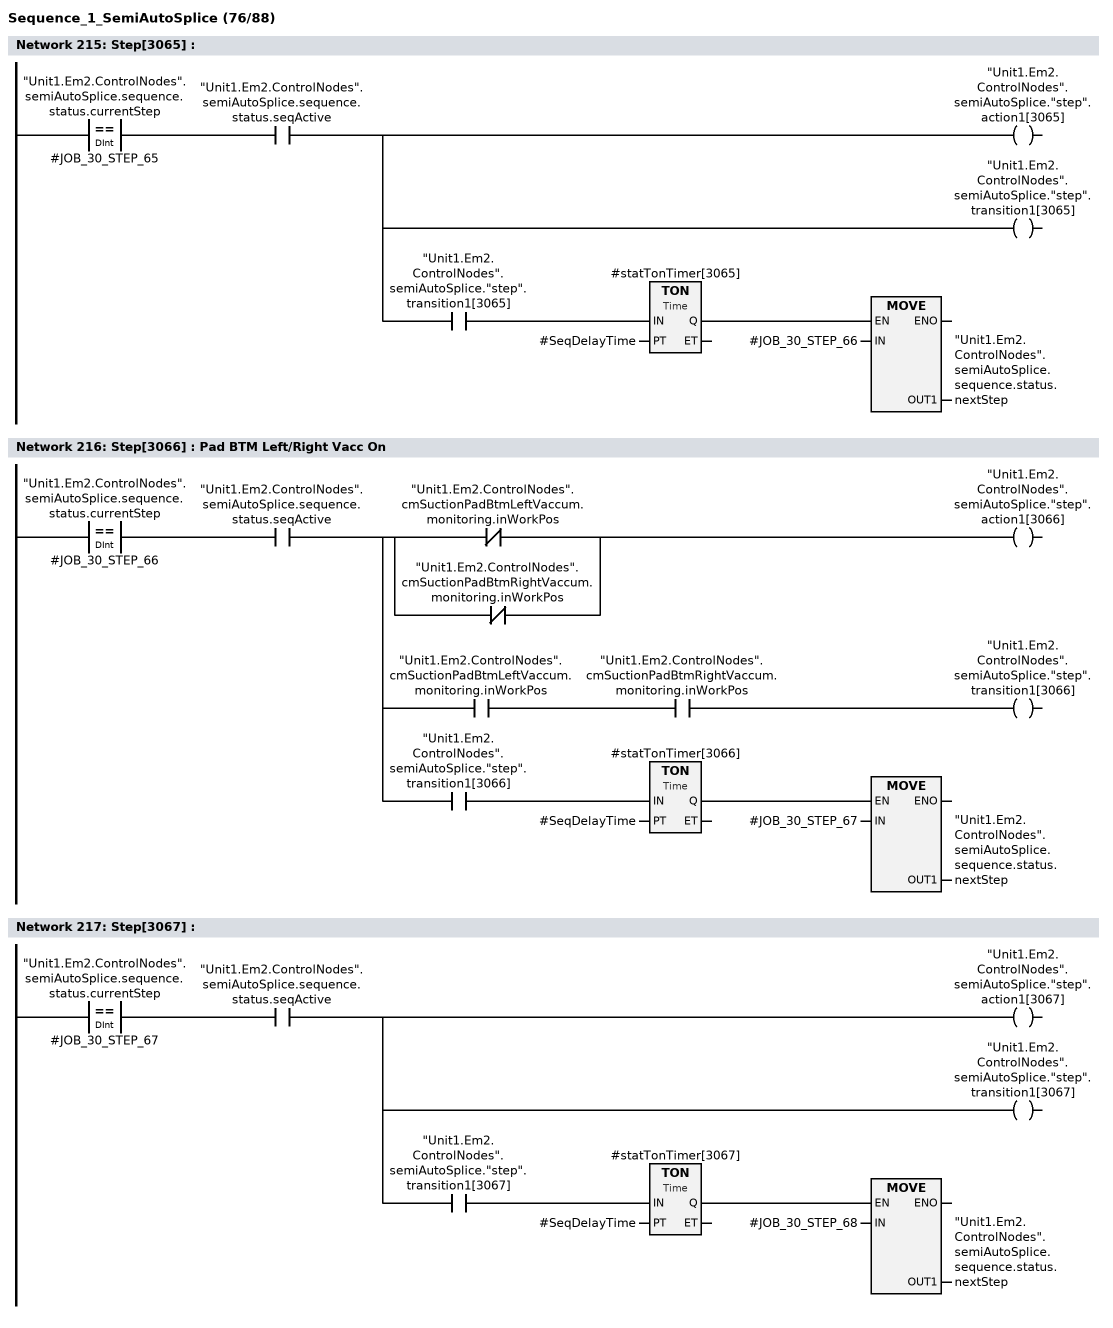
   RUNG wire#powerrail
      { S7_Templates := "SrcType := DInt" } EQ_Contact(in1 := "Unit1.Em2.ControlNodes".semiAutoSplice.sequence.status.currentStep, in2 := #JOB_30_STEP_65)
      Contact( "Unit1.Em2.ControlNodes".semiAutoSplice.sequence.status.seqActive )
      wire#w1
      Coil( "Unit1.Em2.ControlNodes".semiAutoSplice."step".action1[3065] )
   END_RUNG
   RUNG wire#w1
      Coil( "Unit1.Em2.ControlNodes".semiAutoSplice."step".transition1[3065] )
   END_RUNG
   RUNG wire#w1
      Contact( "Unit1.Em2.ControlNodes".semiAutoSplice."step".transition1[3065] )
      { S7_Templates := "time_type := Time" } #statTonTimer[3065].TON(pt := #SeqDelayTime, et =>)
      Move(in := #JOB_30_STEP_66, out1 => "Unit1.Em2.ControlNodes".semiAutoSplice.sequence.status.nextStep)
   END_RUNG
   // the same network as SCL:
   "Unit1.Em2.ControlNodes".semiAutoSplice."step".action1[3065] := ("Unit1.Em2.ControlNodes".semiAutoSplice.sequence.status.currentStep = #JOB_30_STEP_65) AND "Unit1.Em2.ControlNodes".semiAutoSplice.sequence.status.seqActive;
   "Unit1.Em2.ControlNodes".semiAutoSplice."step".transition1[3065] := ("Unit1.Em2.ControlNodes".semiAutoSplice.sequence.status.currentStep = #JOB_30_STEP_65) AND "Unit1.Em2.ControlNodes".semiAutoSplice.sequence.status.seqActive;
   #statTonTimer[3065].TON(IN := ("Unit1.Em2.ControlNodes".semiAutoSplice.sequence.status.currentStep = #JOB_30_STEP_65) AND "Unit1.Em2.ControlNodes".semiAutoSplice.sequence.status.seqActive AND "Unit1.Em2.ControlNodes".semiAutoSplice."step".transition1[3065],
                           PT := #SeqDelayTime);
   IF #statTonTimer[3065].Q THEN
       "Unit1.Em2.ControlNodes".semiAutoSplice.sequence.status.nextStep := #JOB_30_STEP_66;
   END_IF;
END_REGION

REGION Network 216: Step[3066] : Pad BTM Left/Right Vacc On
   RUNG wire#powerrail
      { S7_Templates := "SrcType := DInt" } EQ_Contact(in1 := "Unit1.Em2.ControlNodes".semiAutoSplice.sequence.status.currentStep, in2 := #JOB_30_STEP_66)
      Contact( "Unit1.Em2.ControlNodes".semiAutoSplice.sequence.status.seqActive )
      wire#w1
      I_Contact( "Unit1.Em2.ControlNodes".cmSuctionPadBtmLeftVaccum.monitoring.inWorkPos )
      wire#w2
      Coil( "Unit1.Em2.ControlNodes".semiAutoSplice."step".action1[3066] )
   END_RUNG
   RUNG wire#w1
      I_Contact( "Unit1.Em2.ControlNodes".cmSuctionPadBtmRightVaccum.monitoring.inWorkPos )
   END_RUNG wire#w2
   RUNG wire#w1
      Contact( "Unit1.Em2.ControlNodes".cmSuctionPadBtmLeftVaccum.monitoring.inWorkPos )
      Contact( "Unit1.Em2.ControlNodes".cmSuctionPadBtmRightVaccum.monitoring.inWorkPos )
      Coil( "Unit1.Em2.ControlNodes".semiAutoSplice."step".transition1[3066] )
   END_RUNG
   RUNG wire#w1
      Contact( "Unit1.Em2.ControlNodes".semiAutoSplice."step".transition1[3066] )
      { S7_Templates := "time_type := Time" } #statTonTimer[3066].TON(pt := #SeqDelayTime, et =>)
      Move(in := #JOB_30_STEP_67, out1 => "Unit1.Em2.ControlNodes".semiAutoSplice.sequence.status.nextStep)
   END_RUNG
   // the same network as SCL:
   #_w1 := ("Unit1.Em2.ControlNodes".semiAutoSplice.sequence.status.currentStep = #JOB_30_STEP_66) AND "Unit1.Em2.ControlNodes".semiAutoSplice.sequence.status.seqActive;
   "Unit1.Em2.ControlNodes".semiAutoSplice."step".action1[3066] := #_w1 AND (NOT "Unit1.Em2.ControlNodes".cmSuctionPadBtmLeftVaccum.monitoring.inWorkPos OR NOT "Unit1.Em2.ControlNodes".cmSuctionPadBtmRightVaccum.monitoring.inWorkPos);
   "Unit1.Em2.ControlNodes".semiAutoSplice."step".transition1[3066] := #_w1 AND "Unit1.Em2.ControlNodes".cmSuctionPadBtmLeftVaccum.monitoring.inWorkPos AND "Unit1.Em2.ControlNodes".cmSuctionPadBtmRightVaccum.monitoring.inWorkPos;
   #statTonTimer[3066].TON(IN := #_w1 AND "Unit1.Em2.ControlNodes".semiAutoSplice."step".transition1[3066],
                           PT := #SeqDelayTime);
   IF #statTonTimer[3066].Q THEN
       "Unit1.Em2.ControlNodes".semiAutoSplice.sequence.status.nextStep := #JOB_30_STEP_67;
   END_IF;
END_REGION

REGION Network 217: Step[3067] :
   RUNG wire#powerrail
      { S7_Templates := "SrcType := DInt" } EQ_Contact(in1 := "Unit1.Em2.ControlNodes".semiAutoSplice.sequence.status.currentStep, in2 := #JOB_30_STEP_67)
      Contact( "Unit1.Em2.ControlNodes".semiAutoSplice.sequence.status.seqActive )
      wire#w1
      Coil( "Unit1.Em2.ControlNodes".semiAutoSplice."step".action1[3067] )
   END_RUNG
   RUNG wire#w1
      Coil( "Unit1.Em2.ControlNodes".semiAutoSplice."step".transition1[3067] )
   END_RUNG
   RUNG wire#w1
      Contact( "Unit1.Em2.ControlNodes".semiAutoSplice."step".transition1[3067] )
      { S7_Templates := "time_type := Time" } #statTonTimer[3067].TON(pt := #SeqDelayTime, et =>)
      Move(in := #JOB_30_STEP_68, out1 => "Unit1.Em2.ControlNodes".semiAutoSplice.sequence.status.nextStep)
   END_RUNG
   // the same network as SCL:
   "Unit1.Em2.ControlNodes".semiAutoSplice."step".action1[3067] := ("Unit1.Em2.ControlNodes".semiAutoSplice.sequence.status.currentStep = #JOB_30_STEP_67) AND "Unit1.Em2.ControlNodes".semiAutoSplice.sequence.status.seqActive;
   "Unit1.Em2.ControlNodes".semiAutoSplice."step".transition1[3067] := ("Unit1.Em2.ControlNodes".semiAutoSplice.sequence.status.currentStep = #JOB_30_STEP_67) AND "Unit1.Em2.ControlNodes".semiAutoSplice.sequence.status.seqActive;
   #statTonTimer[3067].TON(IN := ("Unit1.Em2.ControlNodes".semiAutoSplice.sequence.status.currentStep = #JOB_30_STEP_67) AND "Unit1.Em2.ControlNodes".semiAutoSplice.sequence.status.seqActive AND "Unit1.Em2.ControlNodes".semiAutoSplice."step".transition1[3067],
                           PT := #SeqDelayTime);
   IF #statTonTimer[3067].Q THEN
       "Unit1.Em2.ControlNodes".semiAutoSplice.sequence.status.nextStep := #JOB_30_STEP_68;
   END_IF;
END_REGION

REGION Network 218: Step[3068] :
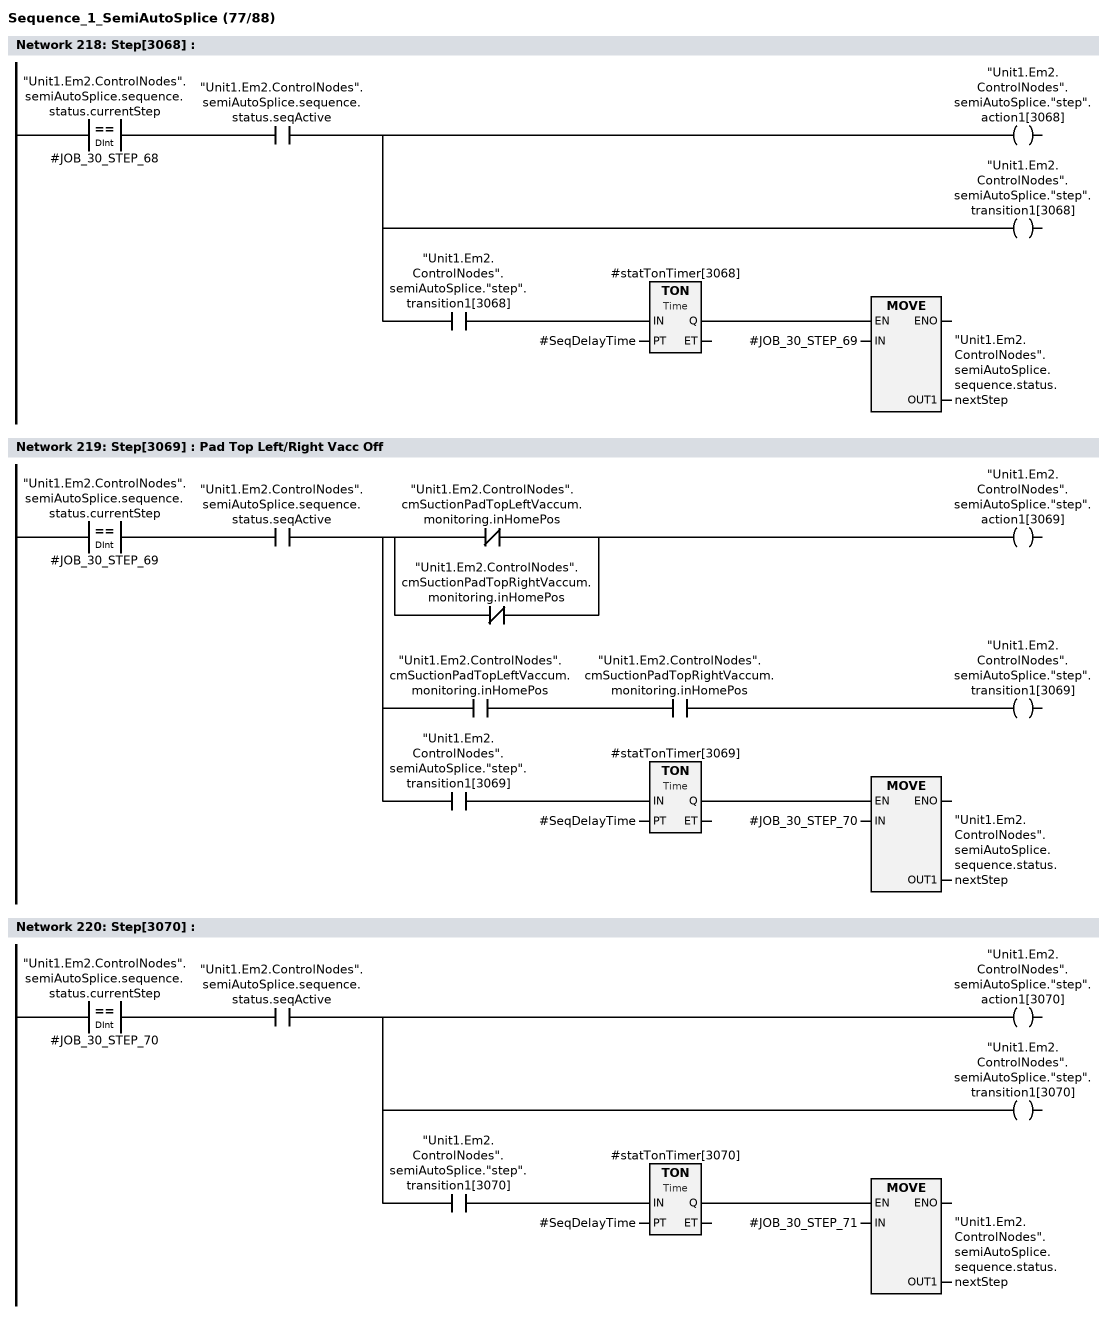
   RUNG wire#powerrail
      { S7_Templates := "SrcType := DInt" } EQ_Contact(in1 := "Unit1.Em2.ControlNodes".semiAutoSplice.sequence.status.currentStep, in2 := #JOB_30_STEP_68)
      Contact( "Unit1.Em2.ControlNodes".semiAutoSplice.sequence.status.seqActive )
      wire#w1
      Coil( "Unit1.Em2.ControlNodes".semiAutoSplice."step".action1[3068] )
   END_RUNG
   RUNG wire#w1
      Coil( "Unit1.Em2.ControlNodes".semiAutoSplice."step".transition1[3068] )
   END_RUNG
   RUNG wire#w1
      Contact( "Unit1.Em2.ControlNodes".semiAutoSplice."step".transition1[3068] )
      { S7_Templates := "time_type := Time" } #statTonTimer[3068].TON(pt := #SeqDelayTime, et =>)
      Move(in := #JOB_30_STEP_69, out1 => "Unit1.Em2.ControlNodes".semiAutoSplice.sequence.status.nextStep)
   END_RUNG
   // the same network as SCL:
   "Unit1.Em2.ControlNodes".semiAutoSplice."step".action1[3068] := ("Unit1.Em2.ControlNodes".semiAutoSplice.sequence.status.currentStep = #JOB_30_STEP_68) AND "Unit1.Em2.ControlNodes".semiAutoSplice.sequence.status.seqActive;
   "Unit1.Em2.ControlNodes".semiAutoSplice."step".transition1[3068] := ("Unit1.Em2.ControlNodes".semiAutoSplice.sequence.status.currentStep = #JOB_30_STEP_68) AND "Unit1.Em2.ControlNodes".semiAutoSplice.sequence.status.seqActive;
   #statTonTimer[3068].TON(IN := ("Unit1.Em2.ControlNodes".semiAutoSplice.sequence.status.currentStep = #JOB_30_STEP_68) AND "Unit1.Em2.ControlNodes".semiAutoSplice.sequence.status.seqActive AND "Unit1.Em2.ControlNodes".semiAutoSplice."step".transition1[3068],
                           PT := #SeqDelayTime);
   IF #statTonTimer[3068].Q THEN
       "Unit1.Em2.ControlNodes".semiAutoSplice.sequence.status.nextStep := #JOB_30_STEP_69;
   END_IF;
END_REGION

REGION Network 219: Step[3069] : Pad Top Left/Right Vacc Off
   RUNG wire#powerrail
      { S7_Templates := "SrcType := DInt" } EQ_Contact(in1 := "Unit1.Em2.ControlNodes".semiAutoSplice.sequence.status.currentStep, in2 := #JOB_30_STEP_69)
      Contact( "Unit1.Em2.ControlNodes".semiAutoSplice.sequence.status.seqActive )
      wire#w1
      I_Contact( "Unit1.Em2.ControlNodes".cmSuctionPadTopLeftVaccum.monitoring.inHomePos )
      wire#w2
      Coil( "Unit1.Em2.ControlNodes".semiAutoSplice."step".action1[3069] )
   END_RUNG
   RUNG wire#w1
      I_Contact( "Unit1.Em2.ControlNodes".cmSuctionPadTopRightVaccum.monitoring.inHomePos )
   END_RUNG wire#w2
   RUNG wire#w1
      Contact( "Unit1.Em2.ControlNodes".cmSuctionPadTopLeftVaccum.monitoring.inHomePos )
      Contact( "Unit1.Em2.ControlNodes".cmSuctionPadTopRightVaccum.monitoring.inHomePos )
      Coil( "Unit1.Em2.ControlNodes".semiAutoSplice."step".transition1[3069] )
   END_RUNG
   RUNG wire#w1
      Contact( "Unit1.Em2.ControlNodes".semiAutoSplice."step".transition1[3069] )
      { S7_Templates := "time_type := Time" } #statTonTimer[3069].TON(pt := #SeqDelayTime, et =>)
      Move(in := #JOB_30_STEP_70, out1 => "Unit1.Em2.ControlNodes".semiAutoSplice.sequence.status.nextStep)
   END_RUNG
   // the same network as SCL:
   #_w1 := ("Unit1.Em2.ControlNodes".semiAutoSplice.sequence.status.currentStep = #JOB_30_STEP_69) AND "Unit1.Em2.ControlNodes".semiAutoSplice.sequence.status.seqActive;
   "Unit1.Em2.ControlNodes".semiAutoSplice."step".action1[3069] := #_w1 AND (NOT "Unit1.Em2.ControlNodes".cmSuctionPadTopLeftVaccum.monitoring.inHomePos OR NOT "Unit1.Em2.ControlNodes".cmSuctionPadTopRightVaccum.monitoring.inHomePos);
   "Unit1.Em2.ControlNodes".semiAutoSplice."step".transition1[3069] := #_w1 AND "Unit1.Em2.ControlNodes".cmSuctionPadTopLeftVaccum.monitoring.inHomePos AND "Unit1.Em2.ControlNodes".cmSuctionPadTopRightVaccum.monitoring.inHomePos;
   #statTonTimer[3069].TON(IN := #_w1 AND "Unit1.Em2.ControlNodes".semiAutoSplice."step".transition1[3069],
                           PT := #SeqDelayTime);
   IF #statTonTimer[3069].Q THEN
       "Unit1.Em2.ControlNodes".semiAutoSplice.sequence.status.nextStep := #JOB_30_STEP_70;
   END_IF;
END_REGION

REGION Network 220: Step[3070] :
   RUNG wire#powerrail
      { S7_Templates := "SrcType := DInt" } EQ_Contact(in1 := "Unit1.Em2.ControlNodes".semiAutoSplice.sequence.status.currentStep, in2 := #JOB_30_STEP_70)
      Contact( "Unit1.Em2.ControlNodes".semiAutoSplice.sequence.status.seqActive )
      wire#w1
      Coil( "Unit1.Em2.ControlNodes".semiAutoSplice."step".action1[3070] )
   END_RUNG
   RUNG wire#w1
      Coil( "Unit1.Em2.ControlNodes".semiAutoSplice."step".transition1[3070] )
   END_RUNG
   RUNG wire#w1
      Contact( "Unit1.Em2.ControlNodes".semiAutoSplice."step".transition1[3070] )
      { S7_Templates := "time_type := Time" } #statTonTimer[3070].TON(pt := #SeqDelayTime, et =>)
      Move(in := #JOB_30_STEP_71, out1 => "Unit1.Em2.ControlNodes".semiAutoSplice.sequence.status.nextStep)
   END_RUNG
   // the same network as SCL:
   "Unit1.Em2.ControlNodes".semiAutoSplice."step".action1[3070] := ("Unit1.Em2.ControlNodes".semiAutoSplice.sequence.status.currentStep = #JOB_30_STEP_70) AND "Unit1.Em2.ControlNodes".semiAutoSplice.sequence.status.seqActive;
   "Unit1.Em2.ControlNodes".semiAutoSplice."step".transition1[3070] := ("Unit1.Em2.ControlNodes".semiAutoSplice.sequence.status.currentStep = #JOB_30_STEP_70) AND "Unit1.Em2.ControlNodes".semiAutoSplice.sequence.status.seqActive;
   #statTonTimer[3070].TON(IN := ("Unit1.Em2.ControlNodes".semiAutoSplice.sequence.status.currentStep = #JOB_30_STEP_70) AND "Unit1.Em2.ControlNodes".semiAutoSplice.sequence.status.seqActive AND "Unit1.Em2.ControlNodes".semiAutoSplice."step".transition1[3070],
                           PT := #SeqDelayTime);
   IF #statTonTimer[3070].Q THEN
       "Unit1.Em2.ControlNodes".semiAutoSplice.sequence.status.nextStep := #JOB_30_STEP_71;
   END_IF;
END_REGION

REGION Network 221: Step[3071] :
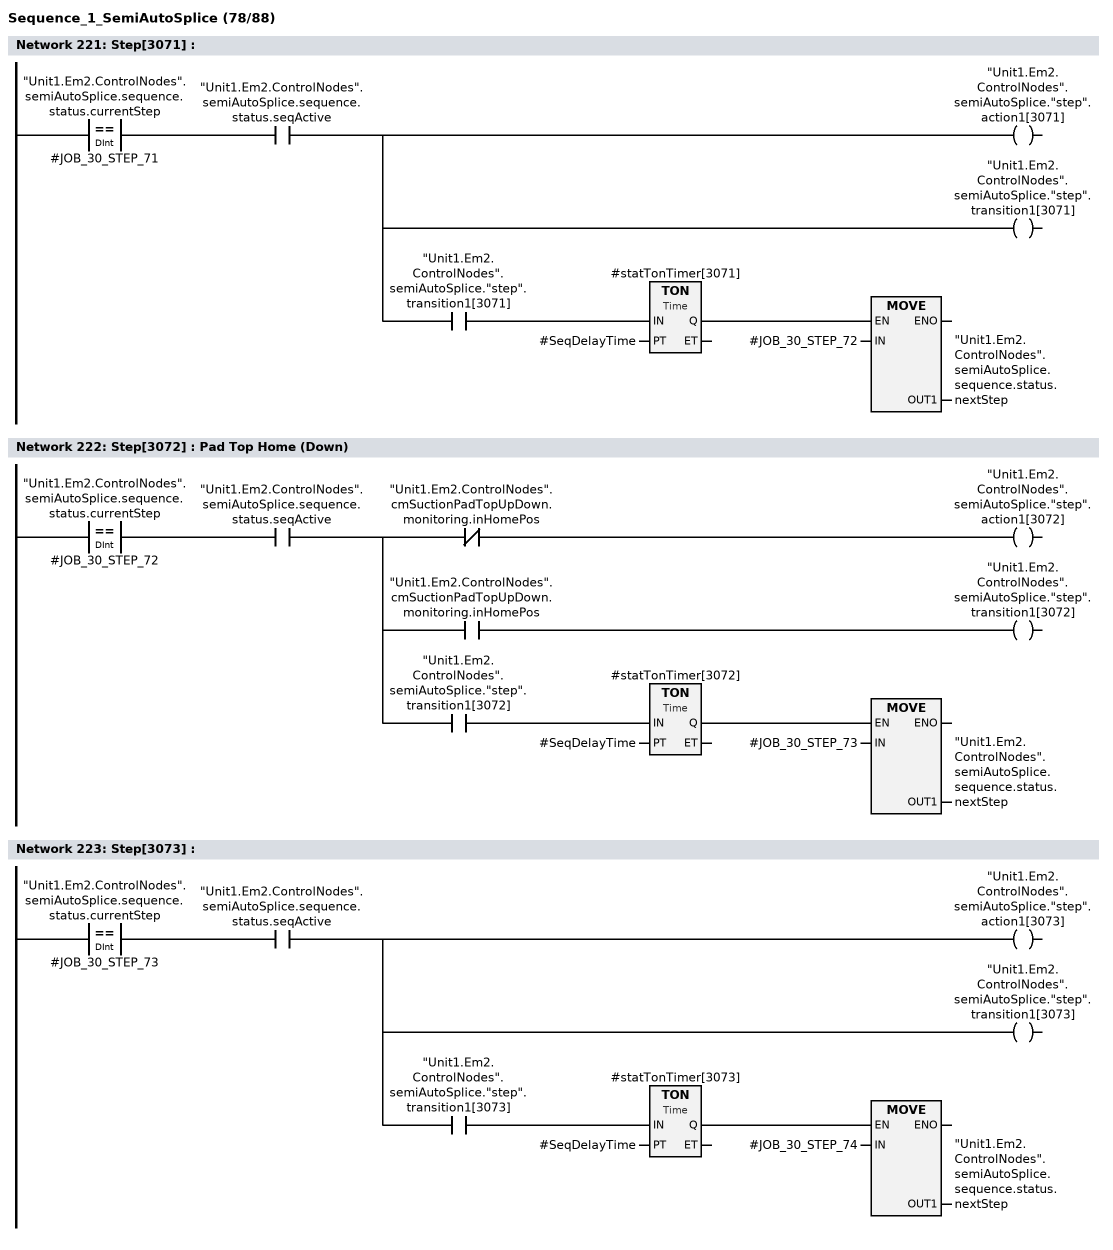
   RUNG wire#powerrail
      { S7_Templates := "SrcType := DInt" } EQ_Contact(in1 := "Unit1.Em2.ControlNodes".semiAutoSplice.sequence.status.currentStep, in2 := #JOB_30_STEP_71)
      Contact( "Unit1.Em2.ControlNodes".semiAutoSplice.sequence.status.seqActive )
      wire#w1
      Coil( "Unit1.Em2.ControlNodes".semiAutoSplice."step".action1[3071] )
   END_RUNG
   RUNG wire#w1
      Coil( "Unit1.Em2.ControlNodes".semiAutoSplice."step".transition1[3071] )
   END_RUNG
   RUNG wire#w1
      Contact( "Unit1.Em2.ControlNodes".semiAutoSplice."step".transition1[3071] )
      { S7_Templates := "time_type := Time" } #statTonTimer[3071].TON(pt := #SeqDelayTime, et =>)
      Move(in := #JOB_30_STEP_72, out1 => "Unit1.Em2.ControlNodes".semiAutoSplice.sequence.status.nextStep)
   END_RUNG
   // the same network as SCL:
   "Unit1.Em2.ControlNodes".semiAutoSplice."step".action1[3071] := ("Unit1.Em2.ControlNodes".semiAutoSplice.sequence.status.currentStep = #JOB_30_STEP_71) AND "Unit1.Em2.ControlNodes".semiAutoSplice.sequence.status.seqActive;
   "Unit1.Em2.ControlNodes".semiAutoSplice."step".transition1[3071] := ("Unit1.Em2.ControlNodes".semiAutoSplice.sequence.status.currentStep = #JOB_30_STEP_71) AND "Unit1.Em2.ControlNodes".semiAutoSplice.sequence.status.seqActive;
   #statTonTimer[3071].TON(IN := ("Unit1.Em2.ControlNodes".semiAutoSplice.sequence.status.currentStep = #JOB_30_STEP_71) AND "Unit1.Em2.ControlNodes".semiAutoSplice.sequence.status.seqActive AND "Unit1.Em2.ControlNodes".semiAutoSplice."step".transition1[3071],
                           PT := #SeqDelayTime);
   IF #statTonTimer[3071].Q THEN
       "Unit1.Em2.ControlNodes".semiAutoSplice.sequence.status.nextStep := #JOB_30_STEP_72;
   END_IF;
END_REGION

REGION Network 222: Step[3072] : Pad Top Home (Down)
   RUNG wire#powerrail
      { S7_Templates := "SrcType := DInt" } EQ_Contact(in1 := "Unit1.Em2.ControlNodes".semiAutoSplice.sequence.status.currentStep, in2 := #JOB_30_STEP_72)
      Contact( "Unit1.Em2.ControlNodes".semiAutoSplice.sequence.status.seqActive )
      wire#w1
      I_Contact( "Unit1.Em2.ControlNodes".cmSuctionPadTopUpDown.monitoring.inHomePos )
      Coil( "Unit1.Em2.ControlNodes".semiAutoSplice."step".action1[3072] )
   END_RUNG
   RUNG wire#w1
      Contact( "Unit1.Em2.ControlNodes".cmSuctionPadTopUpDown.monitoring.inHomePos )
      Coil( "Unit1.Em2.ControlNodes".semiAutoSplice."step".transition1[3072] )
   END_RUNG
   RUNG wire#w1
      Contact( "Unit1.Em2.ControlNodes".semiAutoSplice."step".transition1[3072] )
      { S7_Templates := "time_type := Time" } #statTonTimer[3072].TON(pt := #SeqDelayTime, et =>)
      Move(in := #JOB_30_STEP_73, out1 => "Unit1.Em2.ControlNodes".semiAutoSplice.sequence.status.nextStep)
   END_RUNG
   // the same network as SCL:
   #_w1 := ("Unit1.Em2.ControlNodes".semiAutoSplice.sequence.status.currentStep = #JOB_30_STEP_72) AND "Unit1.Em2.ControlNodes".semiAutoSplice.sequence.status.seqActive;
   "Unit1.Em2.ControlNodes".semiAutoSplice."step".action1[3072] := #_w1 AND NOT "Unit1.Em2.ControlNodes".cmSuctionPadTopUpDown.monitoring.inHomePos;
   "Unit1.Em2.ControlNodes".semiAutoSplice."step".transition1[3072] := #_w1 AND "Unit1.Em2.ControlNodes".cmSuctionPadTopUpDown.monitoring.inHomePos;
   #statTonTimer[3072].TON(IN := #_w1 AND "Unit1.Em2.ControlNodes".semiAutoSplice."step".transition1[3072],
                           PT := #SeqDelayTime);
   IF #statTonTimer[3072].Q THEN
       "Unit1.Em2.ControlNodes".semiAutoSplice.sequence.status.nextStep := #JOB_30_STEP_73;
   END_IF;
END_REGION

REGION Network 223: Step[3073] :
   RUNG wire#powerrail
      { S7_Templates := "SrcType := DInt" } EQ_Contact(in1 := "Unit1.Em2.ControlNodes".semiAutoSplice.sequence.status.currentStep, in2 := #JOB_30_STEP_73)
      Contact( "Unit1.Em2.ControlNodes".semiAutoSplice.sequence.status.seqActive )
      wire#w1
      Coil( "Unit1.Em2.ControlNodes".semiAutoSplice."step".action1[3073] )
   END_RUNG
   RUNG wire#w1
      Coil( "Unit1.Em2.ControlNodes".semiAutoSplice."step".transition1[3073] )
   END_RUNG
   RUNG wire#w1
      Contact( "Unit1.Em2.ControlNodes".semiAutoSplice."step".transition1[3073] )
      { S7_Templates := "time_type := Time" } #statTonTimer[3073].TON(pt := #SeqDelayTime, et =>)
      Move(in := #JOB_30_STEP_74, out1 => "Unit1.Em2.ControlNodes".semiAutoSplice.sequence.status.nextStep)
   END_RUNG
   // the same network as SCL:
   "Unit1.Em2.ControlNodes".semiAutoSplice."step".action1[3073] := ("Unit1.Em2.ControlNodes".semiAutoSplice.sequence.status.currentStep = #JOB_30_STEP_73) AND "Unit1.Em2.ControlNodes".semiAutoSplice.sequence.status.seqActive;
   "Unit1.Em2.ControlNodes".semiAutoSplice."step".transition1[3073] := ("Unit1.Em2.ControlNodes".semiAutoSplice.sequence.status.currentStep = #JOB_30_STEP_73) AND "Unit1.Em2.ControlNodes".semiAutoSplice.sequence.status.seqActive;
   #statTonTimer[3073].TON(IN := ("Unit1.Em2.ControlNodes".semiAutoSplice.sequence.status.currentStep = #JOB_30_STEP_73) AND "Unit1.Em2.ControlNodes".semiAutoSplice.sequence.status.seqActive AND "Unit1.Em2.ControlNodes".semiAutoSplice."step".transition1[3073],
                           PT := #SeqDelayTime);
   IF #statTonTimer[3073].Q THEN
       "Unit1.Em2.ControlNodes".semiAutoSplice.sequence.status.nextStep := #JOB_30_STEP_74;
   END_IF;
END_REGION

REGION Network 224: Step[3074] : Head rotate Top work (FWD)
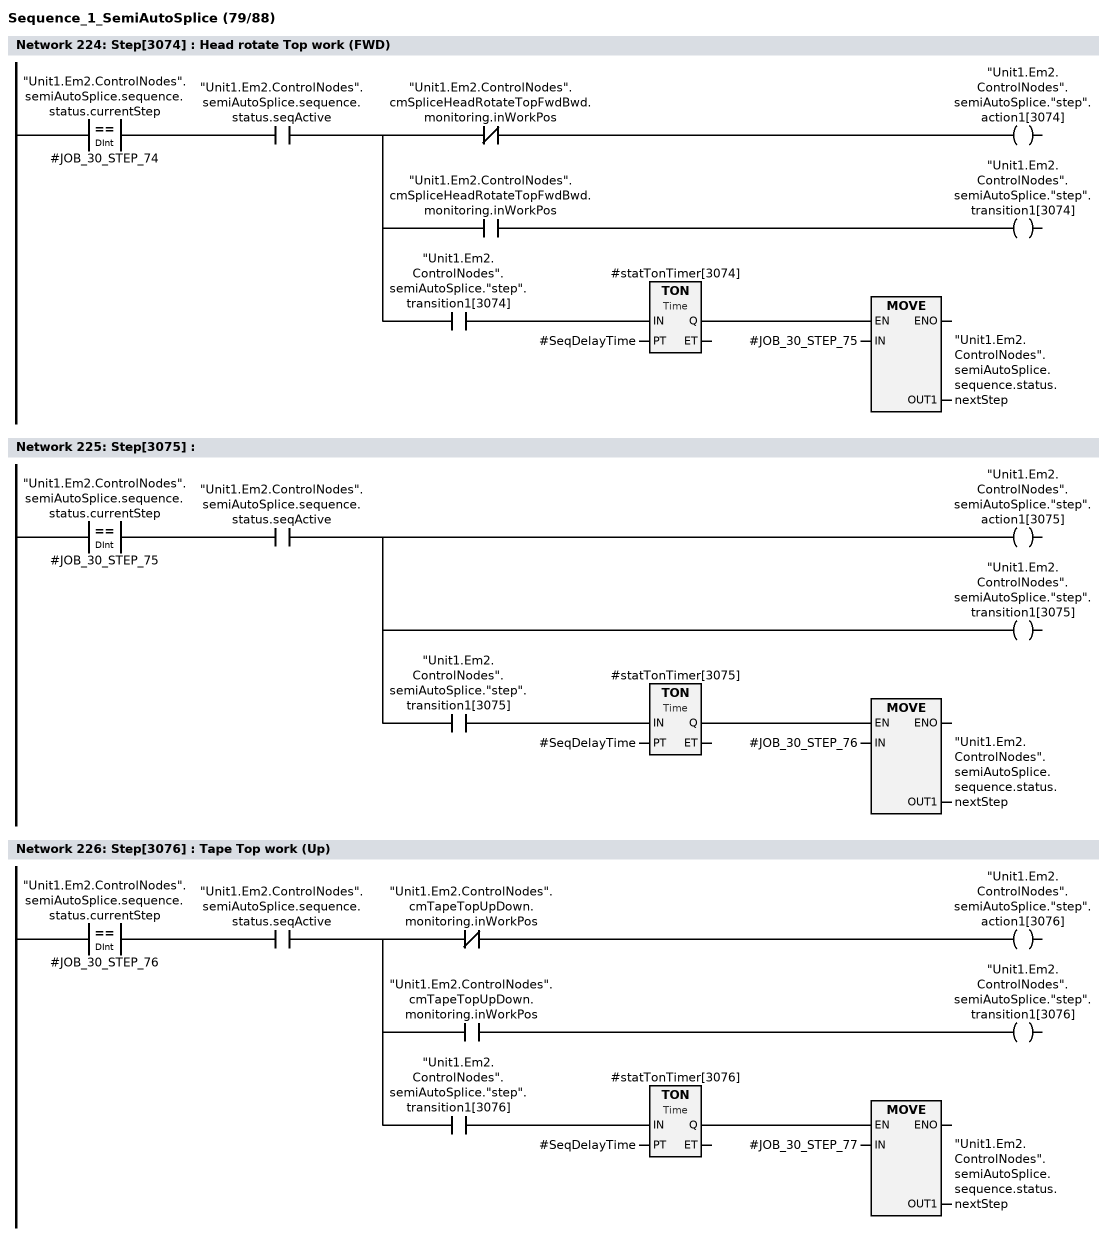
   RUNG wire#powerrail
      { S7_Templates := "SrcType := DInt" } EQ_Contact(in1 := "Unit1.Em2.ControlNodes".semiAutoSplice.sequence.status.currentStep, in2 := #JOB_30_STEP_74)
      Contact( "Unit1.Em2.ControlNodes".semiAutoSplice.sequence.status.seqActive )
      wire#w1
      I_Contact( "Unit1.Em2.ControlNodes".cmSpliceHeadRotateTopFwdBwd.monitoring.inWorkPos )
      Coil( "Unit1.Em2.ControlNodes".semiAutoSplice."step".action1[3074] )
   END_RUNG
   RUNG wire#w1
      Contact( "Unit1.Em2.ControlNodes".cmSpliceHeadRotateTopFwdBwd.monitoring.inWorkPos )
      Coil( "Unit1.Em2.ControlNodes".semiAutoSplice."step".transition1[3074] )
   END_RUNG
   RUNG wire#w1
      Contact( "Unit1.Em2.ControlNodes".semiAutoSplice."step".transition1[3074] )
      { S7_Templates := "time_type := Time" } #statTonTimer[3074].TON(pt := #SeqDelayTime, et =>)
      Move(in := #JOB_30_STEP_75, out1 => "Unit1.Em2.ControlNodes".semiAutoSplice.sequence.status.nextStep)
   END_RUNG
   // the same network as SCL:
   #_w1 := ("Unit1.Em2.ControlNodes".semiAutoSplice.sequence.status.currentStep = #JOB_30_STEP_74) AND "Unit1.Em2.ControlNodes".semiAutoSplice.sequence.status.seqActive;
   "Unit1.Em2.ControlNodes".semiAutoSplice."step".action1[3074] := #_w1 AND NOT "Unit1.Em2.ControlNodes".cmSpliceHeadRotateTopFwdBwd.monitoring.inWorkPos;
   "Unit1.Em2.ControlNodes".semiAutoSplice."step".transition1[3074] := #_w1 AND "Unit1.Em2.ControlNodes".cmSpliceHeadRotateTopFwdBwd.monitoring.inWorkPos;
   #statTonTimer[3074].TON(IN := #_w1 AND "Unit1.Em2.ControlNodes".semiAutoSplice."step".transition1[3074],
                           PT := #SeqDelayTime);
   IF #statTonTimer[3074].Q THEN
       "Unit1.Em2.ControlNodes".semiAutoSplice.sequence.status.nextStep := #JOB_30_STEP_75;
   END_IF;
END_REGION

REGION Network 225: Step[3075] :
   RUNG wire#powerrail
      { S7_Templates := "SrcType := DInt" } EQ_Contact(in1 := "Unit1.Em2.ControlNodes".semiAutoSplice.sequence.status.currentStep, in2 := #JOB_30_STEP_75)
      Contact( "Unit1.Em2.ControlNodes".semiAutoSplice.sequence.status.seqActive )
      wire#w1
      Coil( "Unit1.Em2.ControlNodes".semiAutoSplice."step".action1[3075] )
   END_RUNG
   RUNG wire#w1
      Coil( "Unit1.Em2.ControlNodes".semiAutoSplice."step".transition1[3075] )
   END_RUNG
   RUNG wire#w1
      Contact( "Unit1.Em2.ControlNodes".semiAutoSplice."step".transition1[3075] )
      { S7_Templates := "time_type := Time" } #statTonTimer[3075].TON(pt := #SeqDelayTime, et =>)
      Move(in := #JOB_30_STEP_76, out1 => "Unit1.Em2.ControlNodes".semiAutoSplice.sequence.status.nextStep)
   END_RUNG
   // the same network as SCL:
   "Unit1.Em2.ControlNodes".semiAutoSplice."step".action1[3075] := ("Unit1.Em2.ControlNodes".semiAutoSplice.sequence.status.currentStep = #JOB_30_STEP_75) AND "Unit1.Em2.ControlNodes".semiAutoSplice.sequence.status.seqActive;
   "Unit1.Em2.ControlNodes".semiAutoSplice."step".transition1[3075] := ("Unit1.Em2.ControlNodes".semiAutoSplice.sequence.status.currentStep = #JOB_30_STEP_75) AND "Unit1.Em2.ControlNodes".semiAutoSplice.sequence.status.seqActive;
   #statTonTimer[3075].TON(IN := ("Unit1.Em2.ControlNodes".semiAutoSplice.sequence.status.currentStep = #JOB_30_STEP_75) AND "Unit1.Em2.ControlNodes".semiAutoSplice.sequence.status.seqActive AND "Unit1.Em2.ControlNodes".semiAutoSplice."step".transition1[3075],
                           PT := #SeqDelayTime);
   IF #statTonTimer[3075].Q THEN
       "Unit1.Em2.ControlNodes".semiAutoSplice.sequence.status.nextStep := #JOB_30_STEP_76;
   END_IF;
END_REGION

REGION Network 226: Step[3076] : Tape Top work (Up)
   RUNG wire#powerrail
      { S7_Templates := "SrcType := DInt" } EQ_Contact(in1 := "Unit1.Em2.ControlNodes".semiAutoSplice.sequence.status.currentStep, in2 := #JOB_30_STEP_76)
      Contact( "Unit1.Em2.ControlNodes".semiAutoSplice.sequence.status.seqActive )
      wire#w1
      I_Contact( "Unit1.Em2.ControlNodes".cmTapeTopUpDown.monitoring.inWorkPos )
      Coil( "Unit1.Em2.ControlNodes".semiAutoSplice."step".action1[3076] )
   END_RUNG
   RUNG wire#w1
      Contact( "Unit1.Em2.ControlNodes".cmTapeTopUpDown.monitoring.inWorkPos )
      Coil( "Unit1.Em2.ControlNodes".semiAutoSplice."step".transition1[3076] )
   END_RUNG
   RUNG wire#w1
      Contact( "Unit1.Em2.ControlNodes".semiAutoSplice."step".transition1[3076] )
      { S7_Templates := "time_type := Time" } #statTonTimer[3076].TON(pt := #SeqDelayTime, et =>)
      Move(in := #JOB_30_STEP_77, out1 => "Unit1.Em2.ControlNodes".semiAutoSplice.sequence.status.nextStep)
   END_RUNG
   // the same network as SCL:
   #_w1 := ("Unit1.Em2.ControlNodes".semiAutoSplice.sequence.status.currentStep = #JOB_30_STEP_76) AND "Unit1.Em2.ControlNodes".semiAutoSplice.sequence.status.seqActive;
   "Unit1.Em2.ControlNodes".semiAutoSplice."step".action1[3076] := #_w1 AND NOT "Unit1.Em2.ControlNodes".cmTapeTopUpDown.monitoring.inWorkPos;
   "Unit1.Em2.ControlNodes".semiAutoSplice."step".transition1[3076] := #_w1 AND "Unit1.Em2.ControlNodes".cmTapeTopUpDown.monitoring.inWorkPos;
   #statTonTimer[3076].TON(IN := #_w1 AND "Unit1.Em2.ControlNodes".semiAutoSplice."step".transition1[3076],
                           PT := #SeqDelayTime);
   IF #statTonTimer[3076].Q THEN
       "Unit1.Em2.ControlNodes".semiAutoSplice.sequence.status.nextStep := #JOB_30_STEP_77;
   END_IF;
END_REGION

REGION Network 227: Step[3077] :
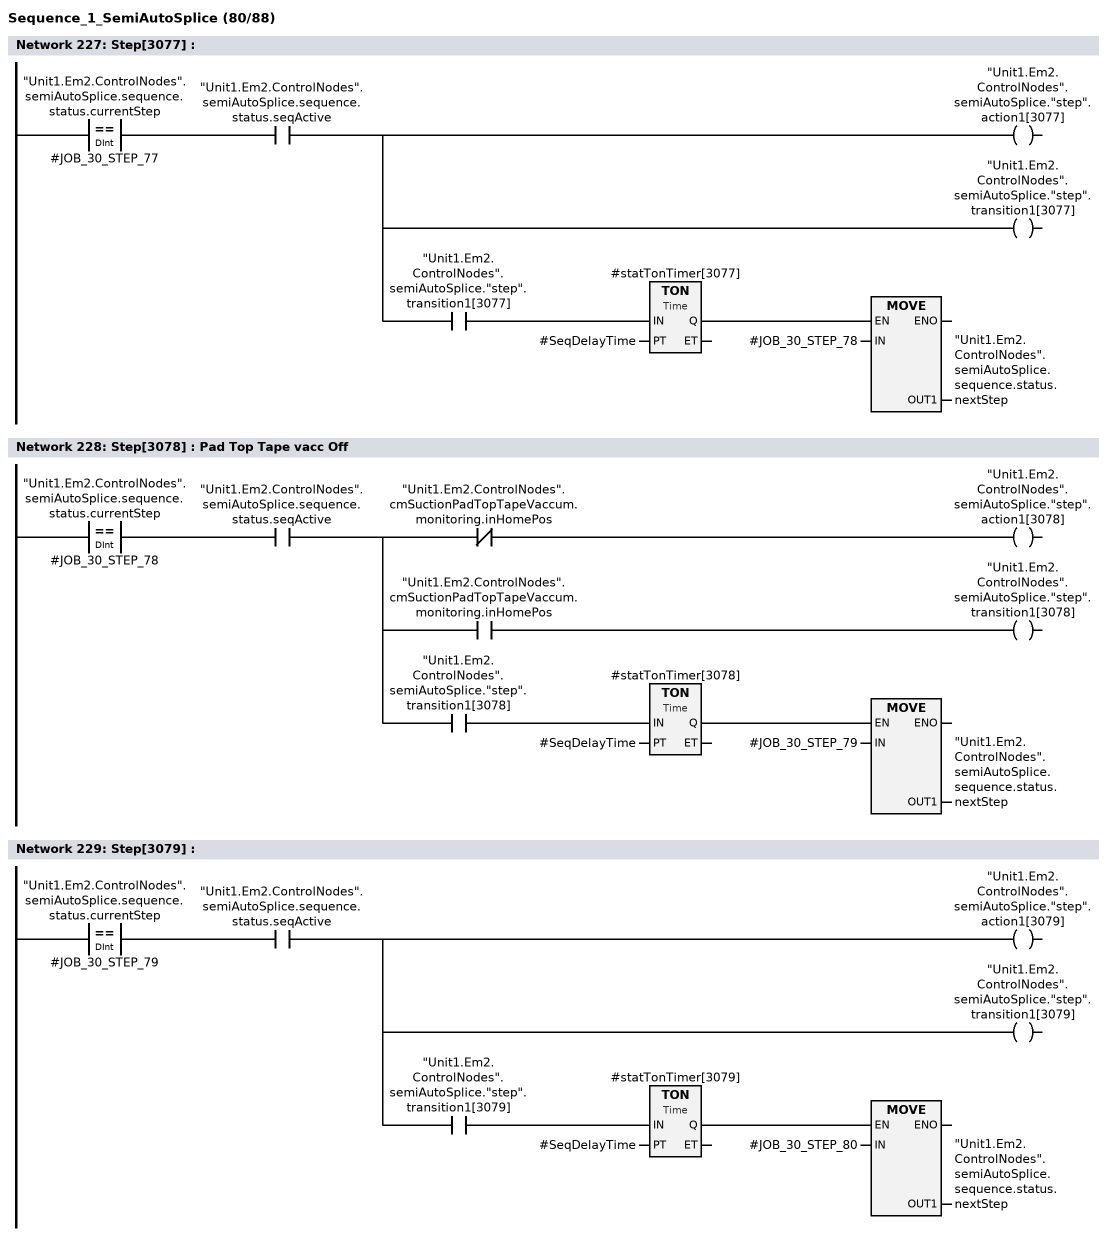
   RUNG wire#powerrail
      { S7_Templates := "SrcType := DInt" } EQ_Contact(in1 := "Unit1.Em2.ControlNodes".semiAutoSplice.sequence.status.currentStep, in2 := #JOB_30_STEP_77)
      Contact( "Unit1.Em2.ControlNodes".semiAutoSplice.sequence.status.seqActive )
      wire#w1
      Coil( "Unit1.Em2.ControlNodes".semiAutoSplice."step".action1[3077] )
   END_RUNG
   RUNG wire#w1
      Coil( "Unit1.Em2.ControlNodes".semiAutoSplice."step".transition1[3077] )
   END_RUNG
   RUNG wire#w1
      Contact( "Unit1.Em2.ControlNodes".semiAutoSplice."step".transition1[3077] )
      { S7_Templates := "time_type := Time" } #statTonTimer[3077].TON(pt := #SeqDelayTime, et =>)
      Move(in := #JOB_30_STEP_78, out1 => "Unit1.Em2.ControlNodes".semiAutoSplice.sequence.status.nextStep)
   END_RUNG
   // the same network as SCL:
   "Unit1.Em2.ControlNodes".semiAutoSplice."step".action1[3077] := ("Unit1.Em2.ControlNodes".semiAutoSplice.sequence.status.currentStep = #JOB_30_STEP_77) AND "Unit1.Em2.ControlNodes".semiAutoSplice.sequence.status.seqActive;
   "Unit1.Em2.ControlNodes".semiAutoSplice."step".transition1[3077] := ("Unit1.Em2.ControlNodes".semiAutoSplice.sequence.status.currentStep = #JOB_30_STEP_77) AND "Unit1.Em2.ControlNodes".semiAutoSplice.sequence.status.seqActive;
   #statTonTimer[3077].TON(IN := ("Unit1.Em2.ControlNodes".semiAutoSplice.sequence.status.currentStep = #JOB_30_STEP_77) AND "Unit1.Em2.ControlNodes".semiAutoSplice.sequence.status.seqActive AND "Unit1.Em2.ControlNodes".semiAutoSplice."step".transition1[3077],
                           PT := #SeqDelayTime);
   IF #statTonTimer[3077].Q THEN
       "Unit1.Em2.ControlNodes".semiAutoSplice.sequence.status.nextStep := #JOB_30_STEP_78;
   END_IF;
END_REGION

REGION Network 228: Step[3078] : Pad Top Tape vacc Off
   RUNG wire#powerrail
      { S7_Templates := "SrcType := DInt" } EQ_Contact(in1 := "Unit1.Em2.ControlNodes".semiAutoSplice.sequence.status.currentStep, in2 := #JOB_30_STEP_78)
      Contact( "Unit1.Em2.ControlNodes".semiAutoSplice.sequence.status.seqActive )
      wire#w1
      I_Contact( "Unit1.Em2.ControlNodes".cmSuctionPadTopTapeVaccum.monitoring.inHomePos )
      Coil( "Unit1.Em2.ControlNodes".semiAutoSplice."step".action1[3078] )
   END_RUNG
   RUNG wire#w1
      Contact( "Unit1.Em2.ControlNodes".cmSuctionPadTopTapeVaccum.monitoring.inHomePos )
      Coil( "Unit1.Em2.ControlNodes".semiAutoSplice."step".transition1[3078] )
   END_RUNG
   RUNG wire#w1
      Contact( "Unit1.Em2.ControlNodes".semiAutoSplice."step".transition1[3078] )
      { S7_Templates := "time_type := Time" } #statTonTimer[3078].TON(pt := #SeqDelayTime, et =>)
      Move(in := #JOB_30_STEP_79, out1 => "Unit1.Em2.ControlNodes".semiAutoSplice.sequence.status.nextStep)
   END_RUNG
   // the same network as SCL:
   #_w1 := ("Unit1.Em2.ControlNodes".semiAutoSplice.sequence.status.currentStep = #JOB_30_STEP_78) AND "Unit1.Em2.ControlNodes".semiAutoSplice.sequence.status.seqActive;
   "Unit1.Em2.ControlNodes".semiAutoSplice."step".action1[3078] := #_w1 AND NOT "Unit1.Em2.ControlNodes".cmSuctionPadTopTapeVaccum.monitoring.inHomePos;
   "Unit1.Em2.ControlNodes".semiAutoSplice."step".transition1[3078] := #_w1 AND "Unit1.Em2.ControlNodes".cmSuctionPadTopTapeVaccum.monitoring.inHomePos;
   #statTonTimer[3078].TON(IN := #_w1 AND "Unit1.Em2.ControlNodes".semiAutoSplice."step".transition1[3078],
                           PT := #SeqDelayTime);
   IF #statTonTimer[3078].Q THEN
       "Unit1.Em2.ControlNodes".semiAutoSplice.sequence.status.nextStep := #JOB_30_STEP_79;
   END_IF;
END_REGION

REGION Network 229: Step[3079] :
   RUNG wire#powerrail
      { S7_Templates := "SrcType := DInt" } EQ_Contact(in1 := "Unit1.Em2.ControlNodes".semiAutoSplice.sequence.status.currentStep, in2 := #JOB_30_STEP_79)
      Contact( "Unit1.Em2.ControlNodes".semiAutoSplice.sequence.status.seqActive )
      wire#w1
      Coil( "Unit1.Em2.ControlNodes".semiAutoSplice."step".action1[3079] )
   END_RUNG
   RUNG wire#w1
      Coil( "Unit1.Em2.ControlNodes".semiAutoSplice."step".transition1[3079] )
   END_RUNG
   RUNG wire#w1
      Contact( "Unit1.Em2.ControlNodes".semiAutoSplice."step".transition1[3079] )
      { S7_Templates := "time_type := Time" } #statTonTimer[3079].TON(pt := #SeqDelayTime, et =>)
      Move(in := #JOB_30_STEP_80, out1 => "Unit1.Em2.ControlNodes".semiAutoSplice.sequence.status.nextStep)
   END_RUNG
   // the same network as SCL:
   "Unit1.Em2.ControlNodes".semiAutoSplice."step".action1[3079] := ("Unit1.Em2.ControlNodes".semiAutoSplice.sequence.status.currentStep = #JOB_30_STEP_79) AND "Unit1.Em2.ControlNodes".semiAutoSplice.sequence.status.seqActive;
   "Unit1.Em2.ControlNodes".semiAutoSplice."step".transition1[3079] := ("Unit1.Em2.ControlNodes".semiAutoSplice.sequence.status.currentStep = #JOB_30_STEP_79) AND "Unit1.Em2.ControlNodes".semiAutoSplice.sequence.status.seqActive;
   #statTonTimer[3079].TON(IN := ("Unit1.Em2.ControlNodes".semiAutoSplice.sequence.status.currentStep = #JOB_30_STEP_79) AND "Unit1.Em2.ControlNodes".semiAutoSplice.sequence.status.seqActive AND "Unit1.Em2.ControlNodes".semiAutoSplice."step".transition1[3079],
                           PT := #SeqDelayTime);
   IF #statTonTimer[3079].Q THEN
       "Unit1.Em2.ControlNodes".semiAutoSplice.sequence.status.nextStep := #JOB_30_STEP_80;
   END_IF;
END_REGION

REGION Network 230: Step[3080] : Tape Top home (Down)
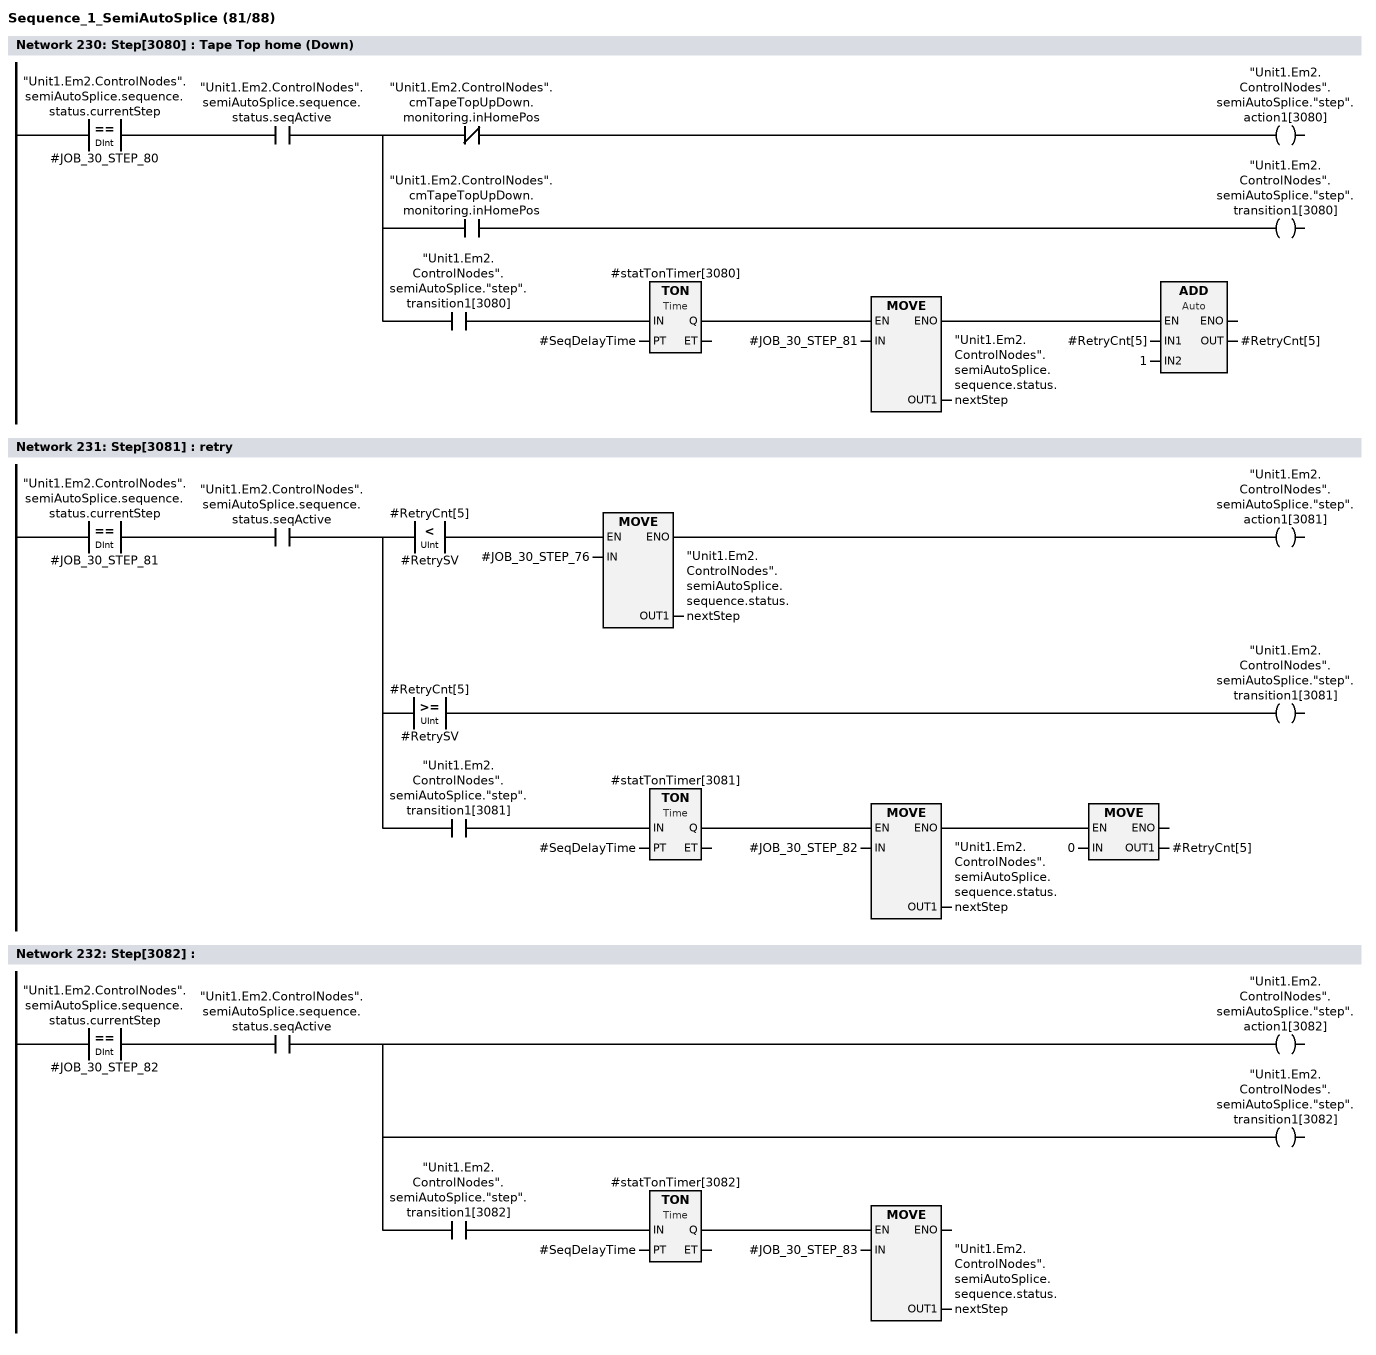
   RUNG wire#powerrail
      { S7_Templates := "SrcType := DInt" } EQ_Contact(in1 := "Unit1.Em2.ControlNodes".semiAutoSplice.sequence.status.currentStep, in2 := #JOB_30_STEP_80)
      Contact( "Unit1.Em2.ControlNodes".semiAutoSplice.sequence.status.seqActive )
      wire#w1
      I_Contact( "Unit1.Em2.ControlNodes".cmTapeTopUpDown.monitoring.inHomePos )
      Coil( "Unit1.Em2.ControlNodes".semiAutoSplice."step".action1[3080] )
   END_RUNG
   RUNG wire#w1
      Contact( "Unit1.Em2.ControlNodes".cmTapeTopUpDown.monitoring.inHomePos )
      Coil( "Unit1.Em2.ControlNodes".semiAutoSplice."step".transition1[3080] )
   END_RUNG
   RUNG wire#w1
      Contact( "Unit1.Em2.ControlNodes".semiAutoSplice."step".transition1[3080] )
      { S7_Templates := "time_type := Time" } #statTonTimer[3080].TON(pt := #SeqDelayTime, et =>)
      Move(in := #JOB_30_STEP_81, out1 => "Unit1.Em2.ControlNodes".semiAutoSplice.sequence.status.nextStep)
      Add(in1 := #RetryCnt[5], in2 := 1, out => #RetryCnt[5])
   END_RUNG
   // the same network as SCL:
   #_w1 := ("Unit1.Em2.ControlNodes".semiAutoSplice.sequence.status.currentStep = #JOB_30_STEP_80) AND "Unit1.Em2.ControlNodes".semiAutoSplice.sequence.status.seqActive;
   "Unit1.Em2.ControlNodes".semiAutoSplice."step".action1[3080] := #_w1 AND NOT "Unit1.Em2.ControlNodes".cmTapeTopUpDown.monitoring.inHomePos;
   "Unit1.Em2.ControlNodes".semiAutoSplice."step".transition1[3080] := #_w1 AND "Unit1.Em2.ControlNodes".cmTapeTopUpDown.monitoring.inHomePos;
   #statTonTimer[3080].TON(IN := #_w1 AND "Unit1.Em2.ControlNodes".semiAutoSplice."step".transition1[3080],
                           PT := #SeqDelayTime);
   IF #statTonTimer[3080].Q THEN
       "Unit1.Em2.ControlNodes".semiAutoSplice.sequence.status.nextStep := #JOB_30_STEP_81;
       #RetryCnt[5] := #RetryCnt[5] + 1;
   END_IF;
END_REGION

REGION Network 231: Step[3081] : retry
   RUNG wire#powerrail
      { S7_Templates := "SrcType := DInt" } EQ_Contact(in1 := "Unit1.Em2.ControlNodes".semiAutoSplice.sequence.status.currentStep, in2 := #JOB_30_STEP_81)
      Contact( "Unit1.Em2.ControlNodes".semiAutoSplice.sequence.status.seqActive )
      wire#w1
      { S7_Templates := "SrcType := UInt" } LT_Contact(in1 := #RetryCnt[5], in2 := #RetrySV)
      Move(in := #JOB_30_STEP_76, out1 => "Unit1.Em2.ControlNodes".semiAutoSplice.sequence.status.nextStep)
      Coil( "Unit1.Em2.ControlNodes".semiAutoSplice."step".action1[3081] )
   END_RUNG
   RUNG wire#w1
      { S7_Templates := "SrcType := UInt" } GE_Contact(in1 := #RetryCnt[5], in2 := #RetrySV)
      Coil( "Unit1.Em2.ControlNodes".semiAutoSplice."step".transition1[3081] )
   END_RUNG
   RUNG wire#w1
      Contact( "Unit1.Em2.ControlNodes".semiAutoSplice."step".transition1[3081] )
      { S7_Templates := "time_type := Time" } #statTonTimer[3081].TON(pt := #SeqDelayTime, et =>)
      Move(in := #JOB_30_STEP_82, out1 => "Unit1.Em2.ControlNodes".semiAutoSplice.sequence.status.nextStep)
      Move(in := 0, out1 => #RetryCnt[5])
   END_RUNG
   // the same network as SCL:
   #_w1 := ("Unit1.Em2.ControlNodes".semiAutoSplice.sequence.status.currentStep = #JOB_30_STEP_81) AND "Unit1.Em2.ControlNodes".semiAutoSplice.sequence.status.seqActive;
   #_w2 := #_w1 AND (#RetryCnt[5] < #RetrySV);
   IF #_w2 THEN "Unit1.Em2.ControlNodes".semiAutoSplice.sequence.status.nextStep := #JOB_30_STEP_76; END_IF;
   "Unit1.Em2.ControlNodes".semiAutoSplice."step".action1[3081] := #_w2;
   "Unit1.Em2.ControlNodes".semiAutoSplice."step".transition1[3081] := #_w1 AND (#RetryCnt[5] >= #RetrySV);
   #statTonTimer[3081].TON(IN := #_w1 AND "Unit1.Em2.ControlNodes".semiAutoSplice."step".transition1[3081],
                           PT := #SeqDelayTime);
   IF #statTonTimer[3081].Q THEN
       "Unit1.Em2.ControlNodes".semiAutoSplice.sequence.status.nextStep := #JOB_30_STEP_82;
       #RetryCnt[5] := 0;
   END_IF;
END_REGION

REGION Network 232: Step[3082] :
   RUNG wire#powerrail
      { S7_Templates := "SrcType := DInt" } EQ_Contact(in1 := "Unit1.Em2.ControlNodes".semiAutoSplice.sequence.status.currentStep, in2 := #JOB_30_STEP_82)
      Contact( "Unit1.Em2.ControlNodes".semiAutoSplice.sequence.status.seqActive )
      wire#w1
      Coil( "Unit1.Em2.ControlNodes".semiAutoSplice."step".action1[3082] )
   END_RUNG
   RUNG wire#w1
      Coil( "Unit1.Em2.ControlNodes".semiAutoSplice."step".transition1[3082] )
   END_RUNG
   RUNG wire#w1
      Contact( "Unit1.Em2.ControlNodes".semiAutoSplice."step".transition1[3082] )
      { S7_Templates := "time_type := Time" } #statTonTimer[3082].TON(pt := #SeqDelayTime, et =>)
      Move(in := #JOB_30_STEP_83, out1 => "Unit1.Em2.ControlNodes".semiAutoSplice.sequence.status.nextStep)
   END_RUNG
   // the same network as SCL:
   "Unit1.Em2.ControlNodes".semiAutoSplice."step".action1[3082] := ("Unit1.Em2.ControlNodes".semiAutoSplice.sequence.status.currentStep = #JOB_30_STEP_82) AND "Unit1.Em2.ControlNodes".semiAutoSplice.sequence.status.seqActive;
   "Unit1.Em2.ControlNodes".semiAutoSplice."step".transition1[3082] := ("Unit1.Em2.ControlNodes".semiAutoSplice.sequence.status.currentStep = #JOB_30_STEP_82) AND "Unit1.Em2.ControlNodes".semiAutoSplice.sequence.status.seqActive;
   #statTonTimer[3082].TON(IN := ("Unit1.Em2.ControlNodes".semiAutoSplice.sequence.status.currentStep = #JOB_30_STEP_82) AND "Unit1.Em2.ControlNodes".semiAutoSplice.sequence.status.seqActive AND "Unit1.Em2.ControlNodes".semiAutoSplice."step".transition1[3082],
                           PT := #SeqDelayTime);
   IF #statTonTimer[3082].Q THEN
       "Unit1.Em2.ControlNodes".semiAutoSplice.sequence.status.nextStep := #JOB_30_STEP_83;
   END_IF;
END_REGION

REGION Network 233: Step[3083] : Head rotate top home (BWD)
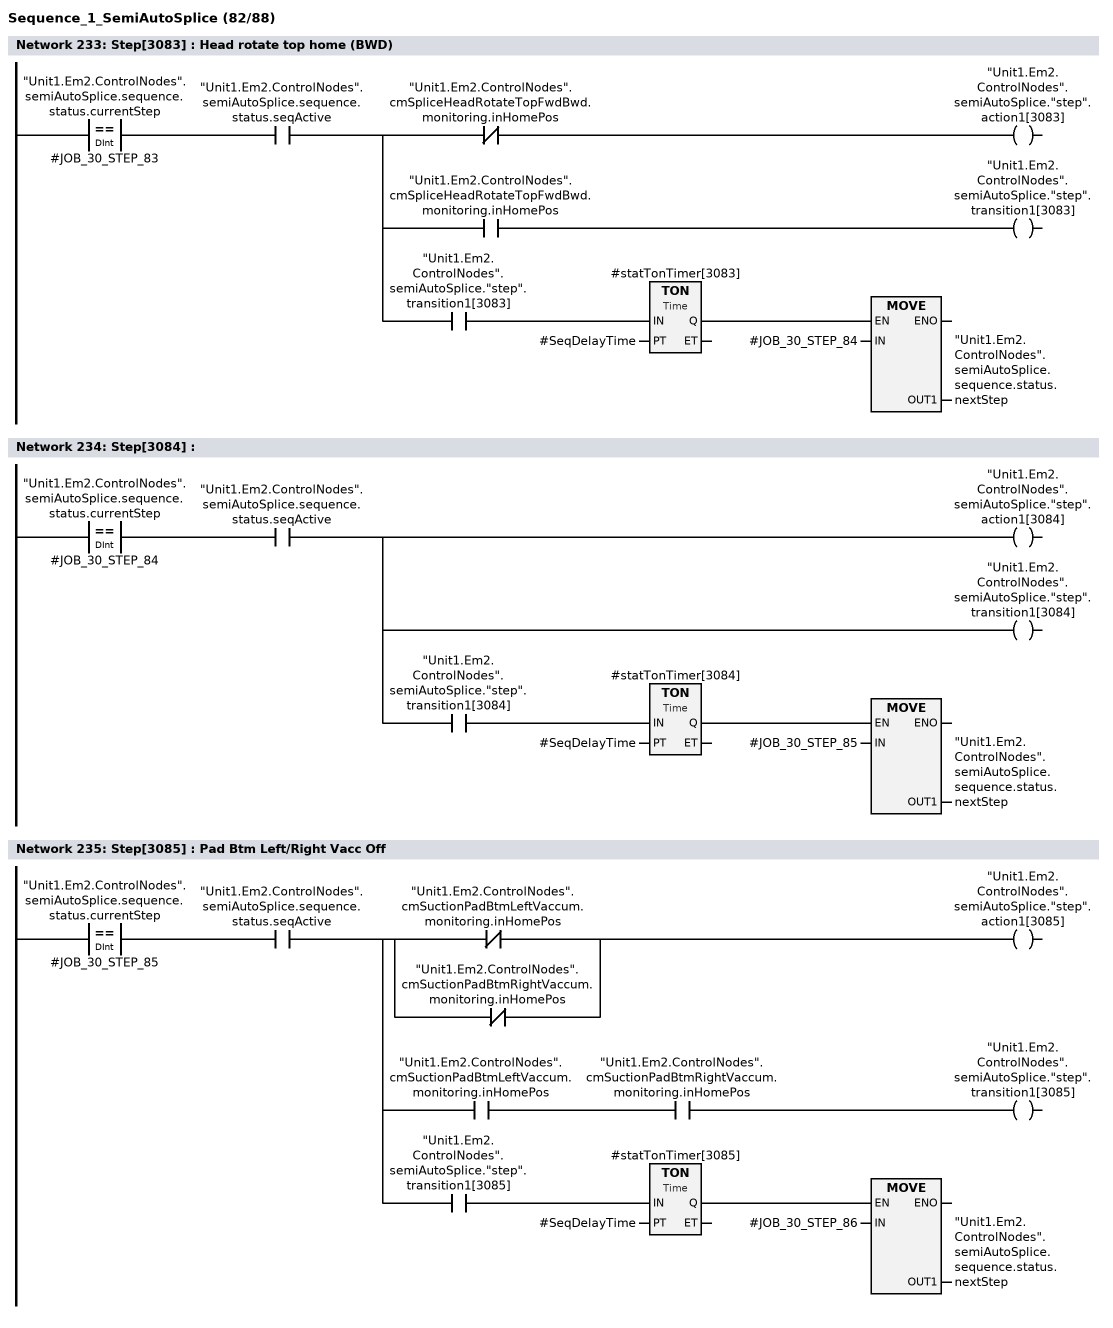
   RUNG wire#powerrail
      { S7_Templates := "SrcType := DInt" } EQ_Contact(in1 := "Unit1.Em2.ControlNodes".semiAutoSplice.sequence.status.currentStep, in2 := #JOB_30_STEP_83)
      Contact( "Unit1.Em2.ControlNodes".semiAutoSplice.sequence.status.seqActive )
      wire#w1
      I_Contact( "Unit1.Em2.ControlNodes".cmSpliceHeadRotateTopFwdBwd.monitoring.inHomePos )
      Coil( "Unit1.Em2.ControlNodes".semiAutoSplice."step".action1[3083] )
   END_RUNG
   RUNG wire#w1
      Contact( "Unit1.Em2.ControlNodes".cmSpliceHeadRotateTopFwdBwd.monitoring.inHomePos )
      Coil( "Unit1.Em2.ControlNodes".semiAutoSplice."step".transition1[3083] )
   END_RUNG
   RUNG wire#w1
      Contact( "Unit1.Em2.ControlNodes".semiAutoSplice."step".transition1[3083] )
      { S7_Templates := "time_type := Time" } #statTonTimer[3083].TON(pt := #SeqDelayTime, et =>)
      Move(in := #JOB_30_STEP_84, out1 => "Unit1.Em2.ControlNodes".semiAutoSplice.sequence.status.nextStep)
   END_RUNG
   // the same network as SCL:
   #_w1 := ("Unit1.Em2.ControlNodes".semiAutoSplice.sequence.status.currentStep = #JOB_30_STEP_83) AND "Unit1.Em2.ControlNodes".semiAutoSplice.sequence.status.seqActive;
   "Unit1.Em2.ControlNodes".semiAutoSplice."step".action1[3083] := #_w1 AND NOT "Unit1.Em2.ControlNodes".cmSpliceHeadRotateTopFwdBwd.monitoring.inHomePos;
   "Unit1.Em2.ControlNodes".semiAutoSplice."step".transition1[3083] := #_w1 AND "Unit1.Em2.ControlNodes".cmSpliceHeadRotateTopFwdBwd.monitoring.inHomePos;
   #statTonTimer[3083].TON(IN := #_w1 AND "Unit1.Em2.ControlNodes".semiAutoSplice."step".transition1[3083],
                           PT := #SeqDelayTime);
   IF #statTonTimer[3083].Q THEN
       "Unit1.Em2.ControlNodes".semiAutoSplice.sequence.status.nextStep := #JOB_30_STEP_84;
   END_IF;
END_REGION

REGION Network 234: Step[3084] :
   RUNG wire#powerrail
      { S7_Templates := "SrcType := DInt" } EQ_Contact(in1 := "Unit1.Em2.ControlNodes".semiAutoSplice.sequence.status.currentStep, in2 := #JOB_30_STEP_84)
      Contact( "Unit1.Em2.ControlNodes".semiAutoSplice.sequence.status.seqActive )
      wire#w1
      Coil( "Unit1.Em2.ControlNodes".semiAutoSplice."step".action1[3084] )
   END_RUNG
   RUNG wire#w1
      Coil( "Unit1.Em2.ControlNodes".semiAutoSplice."step".transition1[3084] )
   END_RUNG
   RUNG wire#w1
      Contact( "Unit1.Em2.ControlNodes".semiAutoSplice."step".transition1[3084] )
      { S7_Templates := "time_type := Time" } #statTonTimer[3084].TON(pt := #SeqDelayTime, et =>)
      Move(in := #JOB_30_STEP_85, out1 => "Unit1.Em2.ControlNodes".semiAutoSplice.sequence.status.nextStep)
   END_RUNG
   // the same network as SCL:
   "Unit1.Em2.ControlNodes".semiAutoSplice."step".action1[3084] := ("Unit1.Em2.ControlNodes".semiAutoSplice.sequence.status.currentStep = #JOB_30_STEP_84) AND "Unit1.Em2.ControlNodes".semiAutoSplice.sequence.status.seqActive;
   "Unit1.Em2.ControlNodes".semiAutoSplice."step".transition1[3084] := ("Unit1.Em2.ControlNodes".semiAutoSplice.sequence.status.currentStep = #JOB_30_STEP_84) AND "Unit1.Em2.ControlNodes".semiAutoSplice.sequence.status.seqActive;
   #statTonTimer[3084].TON(IN := ("Unit1.Em2.ControlNodes".semiAutoSplice.sequence.status.currentStep = #JOB_30_STEP_84) AND "Unit1.Em2.ControlNodes".semiAutoSplice.sequence.status.seqActive AND "Unit1.Em2.ControlNodes".semiAutoSplice."step".transition1[3084],
                           PT := #SeqDelayTime);
   IF #statTonTimer[3084].Q THEN
       "Unit1.Em2.ControlNodes".semiAutoSplice.sequence.status.nextStep := #JOB_30_STEP_85;
   END_IF;
END_REGION

REGION Network 235: Step[3085] : Pad Btm Left/Right Vacc Off
   RUNG wire#powerrail
      { S7_Templates := "SrcType := DInt" } EQ_Contact(in1 := "Unit1.Em2.ControlNodes".semiAutoSplice.sequence.status.currentStep, in2 := #JOB_30_STEP_85)
      Contact( "Unit1.Em2.ControlNodes".semiAutoSplice.sequence.status.seqActive )
      wire#w1
      I_Contact( "Unit1.Em2.ControlNodes".cmSuctionPadBtmLeftVaccum.monitoring.inHomePos )
      wire#w2
      Coil( "Unit1.Em2.ControlNodes".semiAutoSplice."step".action1[3085] )
   END_RUNG
   RUNG wire#w1
      I_Contact( "Unit1.Em2.ControlNodes".cmSuctionPadBtmRightVaccum.monitoring.inHomePos )
   END_RUNG wire#w2
   RUNG wire#w1
      Contact( "Unit1.Em2.ControlNodes".cmSuctionPadBtmLeftVaccum.monitoring.inHomePos )
      Contact( "Unit1.Em2.ControlNodes".cmSuctionPadBtmRightVaccum.monitoring.inHomePos )
      Coil( "Unit1.Em2.ControlNodes".semiAutoSplice."step".transition1[3085] )
   END_RUNG
   RUNG wire#w1
      Contact( "Unit1.Em2.ControlNodes".semiAutoSplice."step".transition1[3085] )
      { S7_Templates := "time_type := Time" } #statTonTimer[3085].TON(pt := #SeqDelayTime, et =>)
      Move(in := #JOB_30_STEP_86, out1 => "Unit1.Em2.ControlNodes".semiAutoSplice.sequence.status.nextStep)
   END_RUNG
   // the same network as SCL:
   #_w1 := ("Unit1.Em2.ControlNodes".semiAutoSplice.sequence.status.currentStep = #JOB_30_STEP_85) AND "Unit1.Em2.ControlNodes".semiAutoSplice.sequence.status.seqActive;
   "Unit1.Em2.ControlNodes".semiAutoSplice."step".action1[3085] := #_w1 AND (NOT "Unit1.Em2.ControlNodes".cmSuctionPadBtmLeftVaccum.monitoring.inHomePos OR NOT "Unit1.Em2.ControlNodes".cmSuctionPadBtmRightVaccum.monitoring.inHomePos);
   "Unit1.Em2.ControlNodes".semiAutoSplice."step".transition1[3085] := #_w1 AND "Unit1.Em2.ControlNodes".cmSuctionPadBtmLeftVaccum.monitoring.inHomePos AND "Unit1.Em2.ControlNodes".cmSuctionPadBtmRightVaccum.monitoring.inHomePos;
   #statTonTimer[3085].TON(IN := #_w1 AND "Unit1.Em2.ControlNodes".semiAutoSplice."step".transition1[3085],
                           PT := #SeqDelayTime);
   IF #statTonTimer[3085].Q THEN
       "Unit1.Em2.ControlNodes".semiAutoSplice.sequence.status.nextStep := #JOB_30_STEP_86;
   END_IF;
END_REGION

REGION Network 236: Step[3086] :
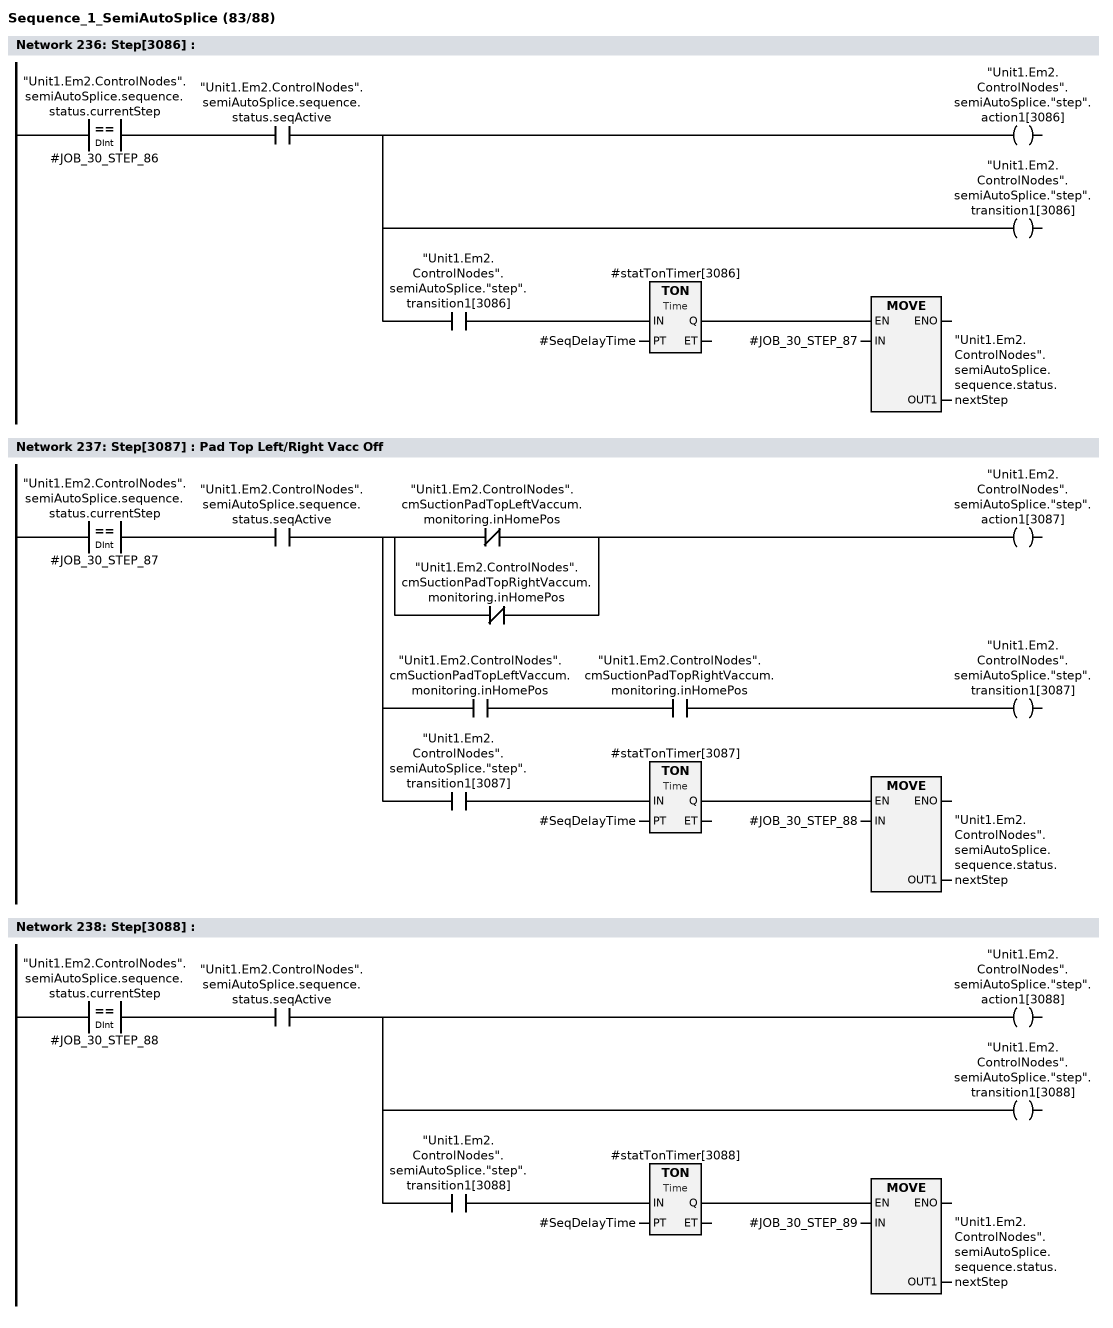
   RUNG wire#powerrail
      { S7_Templates := "SrcType := DInt" } EQ_Contact(in1 := "Unit1.Em2.ControlNodes".semiAutoSplice.sequence.status.currentStep, in2 := #JOB_30_STEP_86)
      Contact( "Unit1.Em2.ControlNodes".semiAutoSplice.sequence.status.seqActive )
      wire#w1
      Coil( "Unit1.Em2.ControlNodes".semiAutoSplice."step".action1[3086] )
   END_RUNG
   RUNG wire#w1
      Coil( "Unit1.Em2.ControlNodes".semiAutoSplice."step".transition1[3086] )
   END_RUNG
   RUNG wire#w1
      Contact( "Unit1.Em2.ControlNodes".semiAutoSplice."step".transition1[3086] )
      { S7_Templates := "time_type := Time" } #statTonTimer[3086].TON(pt := #SeqDelayTime, et =>)
      Move(in := #JOB_30_STEP_87, out1 => "Unit1.Em2.ControlNodes".semiAutoSplice.sequence.status.nextStep)
   END_RUNG
   // the same network as SCL:
   "Unit1.Em2.ControlNodes".semiAutoSplice."step".action1[3086] := ("Unit1.Em2.ControlNodes".semiAutoSplice.sequence.status.currentStep = #JOB_30_STEP_86) AND "Unit1.Em2.ControlNodes".semiAutoSplice.sequence.status.seqActive;
   "Unit1.Em2.ControlNodes".semiAutoSplice."step".transition1[3086] := ("Unit1.Em2.ControlNodes".semiAutoSplice.sequence.status.currentStep = #JOB_30_STEP_86) AND "Unit1.Em2.ControlNodes".semiAutoSplice.sequence.status.seqActive;
   #statTonTimer[3086].TON(IN := ("Unit1.Em2.ControlNodes".semiAutoSplice.sequence.status.currentStep = #JOB_30_STEP_86) AND "Unit1.Em2.ControlNodes".semiAutoSplice.sequence.status.seqActive AND "Unit1.Em2.ControlNodes".semiAutoSplice."step".transition1[3086],
                           PT := #SeqDelayTime);
   IF #statTonTimer[3086].Q THEN
       "Unit1.Em2.ControlNodes".semiAutoSplice.sequence.status.nextStep := #JOB_30_STEP_87;
   END_IF;
END_REGION

REGION Network 237: Step[3087] : Pad Top Left/Right Vacc Off
   RUNG wire#powerrail
      { S7_Templates := "SrcType := DInt" } EQ_Contact(in1 := "Unit1.Em2.ControlNodes".semiAutoSplice.sequence.status.currentStep, in2 := #JOB_30_STEP_87)
      Contact( "Unit1.Em2.ControlNodes".semiAutoSplice.sequence.status.seqActive )
      wire#w1
      I_Contact( "Unit1.Em2.ControlNodes".cmSuctionPadTopLeftVaccum.monitoring.inHomePos )
      wire#w2
      Coil( "Unit1.Em2.ControlNodes".semiAutoSplice."step".action1[3087] )
   END_RUNG
   RUNG wire#w1
      I_Contact( "Unit1.Em2.ControlNodes".cmSuctionPadTopRightVaccum.monitoring.inHomePos )
   END_RUNG wire#w2
   RUNG wire#w1
      Contact( "Unit1.Em2.ControlNodes".cmSuctionPadTopLeftVaccum.monitoring.inHomePos )
      Contact( "Unit1.Em2.ControlNodes".cmSuctionPadTopRightVaccum.monitoring.inHomePos )
      Coil( "Unit1.Em2.ControlNodes".semiAutoSplice."step".transition1[3087] )
   END_RUNG
   RUNG wire#w1
      Contact( "Unit1.Em2.ControlNodes".semiAutoSplice."step".transition1[3087] )
      { S7_Templates := "time_type := Time" } #statTonTimer[3087].TON(pt := #SeqDelayTime, et =>)
      Move(in := #JOB_30_STEP_88, out1 => "Unit1.Em2.ControlNodes".semiAutoSplice.sequence.status.nextStep)
   END_RUNG
   // the same network as SCL:
   #_w1 := ("Unit1.Em2.ControlNodes".semiAutoSplice.sequence.status.currentStep = #JOB_30_STEP_87) AND "Unit1.Em2.ControlNodes".semiAutoSplice.sequence.status.seqActive;
   "Unit1.Em2.ControlNodes".semiAutoSplice."step".action1[3087] := #_w1 AND (NOT "Unit1.Em2.ControlNodes".cmSuctionPadTopLeftVaccum.monitoring.inHomePos OR NOT "Unit1.Em2.ControlNodes".cmSuctionPadTopRightVaccum.monitoring.inHomePos);
   "Unit1.Em2.ControlNodes".semiAutoSplice."step".transition1[3087] := #_w1 AND "Unit1.Em2.ControlNodes".cmSuctionPadTopLeftVaccum.monitoring.inHomePos AND "Unit1.Em2.ControlNodes".cmSuctionPadTopRightVaccum.monitoring.inHomePos;
   #statTonTimer[3087].TON(IN := #_w1 AND "Unit1.Em2.ControlNodes".semiAutoSplice."step".transition1[3087],
                           PT := #SeqDelayTime);
   IF #statTonTimer[3087].Q THEN
       "Unit1.Em2.ControlNodes".semiAutoSplice.sequence.status.nextStep := #JOB_30_STEP_88;
   END_IF;
END_REGION

REGION Network 238: Step[3088] :
   RUNG wire#powerrail
      { S7_Templates := "SrcType := DInt" } EQ_Contact(in1 := "Unit1.Em2.ControlNodes".semiAutoSplice.sequence.status.currentStep, in2 := #JOB_30_STEP_88)
      Contact( "Unit1.Em2.ControlNodes".semiAutoSplice.sequence.status.seqActive )
      wire#w1
      Coil( "Unit1.Em2.ControlNodes".semiAutoSplice."step".action1[3088] )
   END_RUNG
   RUNG wire#w1
      Coil( "Unit1.Em2.ControlNodes".semiAutoSplice."step".transition1[3088] )
   END_RUNG
   RUNG wire#w1
      Contact( "Unit1.Em2.ControlNodes".semiAutoSplice."step".transition1[3088] )
      { S7_Templates := "time_type := Time" } #statTonTimer[3088].TON(pt := #SeqDelayTime, et =>)
      Move(in := #JOB_30_STEP_89, out1 => "Unit1.Em2.ControlNodes".semiAutoSplice.sequence.status.nextStep)
   END_RUNG
   // the same network as SCL:
   "Unit1.Em2.ControlNodes".semiAutoSplice."step".action1[3088] := ("Unit1.Em2.ControlNodes".semiAutoSplice.sequence.status.currentStep = #JOB_30_STEP_88) AND "Unit1.Em2.ControlNodes".semiAutoSplice.sequence.status.seqActive;
   "Unit1.Em2.ControlNodes".semiAutoSplice."step".transition1[3088] := ("Unit1.Em2.ControlNodes".semiAutoSplice.sequence.status.currentStep = #JOB_30_STEP_88) AND "Unit1.Em2.ControlNodes".semiAutoSplice.sequence.status.seqActive;
   #statTonTimer[3088].TON(IN := ("Unit1.Em2.ControlNodes".semiAutoSplice.sequence.status.currentStep = #JOB_30_STEP_88) AND "Unit1.Em2.ControlNodes".semiAutoSplice.sequence.status.seqActive AND "Unit1.Em2.ControlNodes".semiAutoSplice."step".transition1[3088],
                           PT := #SeqDelayTime);
   IF #statTonTimer[3088].Q THEN
       "Unit1.Em2.ControlNodes".semiAutoSplice.sequence.status.nextStep := #JOB_30_STEP_89;
   END_IF;
END_REGION

REGION Network 239: Step[3089] : Pad Btm home (Down)
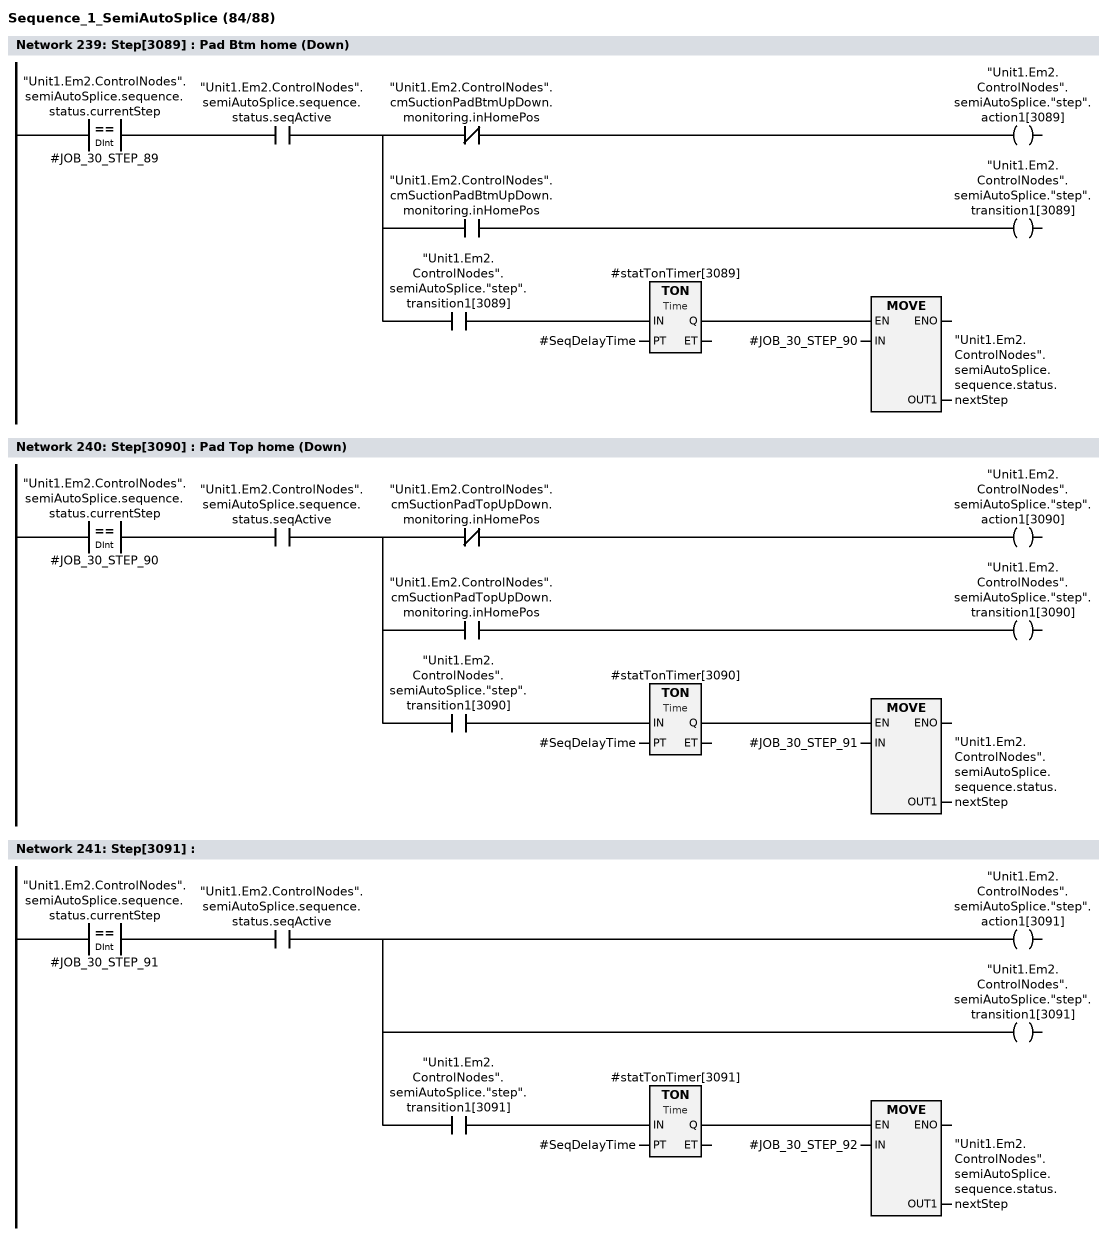
   RUNG wire#powerrail
      { S7_Templates := "SrcType := DInt" } EQ_Contact(in1 := "Unit1.Em2.ControlNodes".semiAutoSplice.sequence.status.currentStep, in2 := #JOB_30_STEP_89)
      Contact( "Unit1.Em2.ControlNodes".semiAutoSplice.sequence.status.seqActive )
      wire#w1
      I_Contact( "Unit1.Em2.ControlNodes".cmSuctionPadBtmUpDown.monitoring.inHomePos )
      Coil( "Unit1.Em2.ControlNodes".semiAutoSplice."step".action1[3089] )
   END_RUNG
   RUNG wire#w1
      Contact( "Unit1.Em2.ControlNodes".cmSuctionPadBtmUpDown.monitoring.inHomePos )
      Coil( "Unit1.Em2.ControlNodes".semiAutoSplice."step".transition1[3089] )
   END_RUNG
   RUNG wire#w1
      Contact( "Unit1.Em2.ControlNodes".semiAutoSplice."step".transition1[3089] )
      { S7_Templates := "time_type := Time" } #statTonTimer[3089].TON(pt := #SeqDelayTime, et =>)
      Move(in := #JOB_30_STEP_90, out1 => "Unit1.Em2.ControlNodes".semiAutoSplice.sequence.status.nextStep)
   END_RUNG
   // the same network as SCL:
   #_w1 := ("Unit1.Em2.ControlNodes".semiAutoSplice.sequence.status.currentStep = #JOB_30_STEP_89) AND "Unit1.Em2.ControlNodes".semiAutoSplice.sequence.status.seqActive;
   "Unit1.Em2.ControlNodes".semiAutoSplice."step".action1[3089] := #_w1 AND NOT "Unit1.Em2.ControlNodes".cmSuctionPadBtmUpDown.monitoring.inHomePos;
   "Unit1.Em2.ControlNodes".semiAutoSplice."step".transition1[3089] := #_w1 AND "Unit1.Em2.ControlNodes".cmSuctionPadBtmUpDown.monitoring.inHomePos;
   #statTonTimer[3089].TON(IN := #_w1 AND "Unit1.Em2.ControlNodes".semiAutoSplice."step".transition1[3089],
                           PT := #SeqDelayTime);
   IF #statTonTimer[3089].Q THEN
       "Unit1.Em2.ControlNodes".semiAutoSplice.sequence.status.nextStep := #JOB_30_STEP_90;
   END_IF;
END_REGION

REGION Network 240: Step[3090] : Pad Top home (Down)
   RUNG wire#powerrail
      { S7_Templates := "SrcType := DInt" } EQ_Contact(in1 := "Unit1.Em2.ControlNodes".semiAutoSplice.sequence.status.currentStep, in2 := #JOB_30_STEP_90)
      Contact( "Unit1.Em2.ControlNodes".semiAutoSplice.sequence.status.seqActive )
      wire#w1
      I_Contact( "Unit1.Em2.ControlNodes".cmSuctionPadTopUpDown.monitoring.inHomePos )
      Coil( "Unit1.Em2.ControlNodes".semiAutoSplice."step".action1[3090] )
   END_RUNG
   RUNG wire#w1
      Contact( "Unit1.Em2.ControlNodes".cmSuctionPadTopUpDown.monitoring.inHomePos )
      Coil( "Unit1.Em2.ControlNodes".semiAutoSplice."step".transition1[3090] )
   END_RUNG
   RUNG wire#w1
      Contact( "Unit1.Em2.ControlNodes".semiAutoSplice."step".transition1[3090] )
      { S7_Templates := "time_type := Time" } #statTonTimer[3090].TON(pt := #SeqDelayTime, et =>)
      Move(in := #JOB_30_STEP_91, out1 => "Unit1.Em2.ControlNodes".semiAutoSplice.sequence.status.nextStep)
   END_RUNG
   // the same network as SCL:
   #_w1 := ("Unit1.Em2.ControlNodes".semiAutoSplice.sequence.status.currentStep = #JOB_30_STEP_90) AND "Unit1.Em2.ControlNodes".semiAutoSplice.sequence.status.seqActive;
   "Unit1.Em2.ControlNodes".semiAutoSplice."step".action1[3090] := #_w1 AND NOT "Unit1.Em2.ControlNodes".cmSuctionPadTopUpDown.monitoring.inHomePos;
   "Unit1.Em2.ControlNodes".semiAutoSplice."step".transition1[3090] := #_w1 AND "Unit1.Em2.ControlNodes".cmSuctionPadTopUpDown.monitoring.inHomePos;
   #statTonTimer[3090].TON(IN := #_w1 AND "Unit1.Em2.ControlNodes".semiAutoSplice."step".transition1[3090],
                           PT := #SeqDelayTime);
   IF #statTonTimer[3090].Q THEN
       "Unit1.Em2.ControlNodes".semiAutoSplice.sequence.status.nextStep := #JOB_30_STEP_91;
   END_IF;
END_REGION

REGION Network 241: Step[3091] :
   RUNG wire#powerrail
      { S7_Templates := "SrcType := DInt" } EQ_Contact(in1 := "Unit1.Em2.ControlNodes".semiAutoSplice.sequence.status.currentStep, in2 := #JOB_30_STEP_91)
      Contact( "Unit1.Em2.ControlNodes".semiAutoSplice.sequence.status.seqActive )
      wire#w1
      Coil( "Unit1.Em2.ControlNodes".semiAutoSplice."step".action1[3091] )
   END_RUNG
   RUNG wire#w1
      Coil( "Unit1.Em2.ControlNodes".semiAutoSplice."step".transition1[3091] )
   END_RUNG
   RUNG wire#w1
      Contact( "Unit1.Em2.ControlNodes".semiAutoSplice."step".transition1[3091] )
      { S7_Templates := "time_type := Time" } #statTonTimer[3091].TON(pt := #SeqDelayTime, et =>)
      Move(in := #JOB_30_STEP_92, out1 => "Unit1.Em2.ControlNodes".semiAutoSplice.sequence.status.nextStep)
   END_RUNG
   // the same network as SCL:
   "Unit1.Em2.ControlNodes".semiAutoSplice."step".action1[3091] := ("Unit1.Em2.ControlNodes".semiAutoSplice.sequence.status.currentStep = #JOB_30_STEP_91) AND "Unit1.Em2.ControlNodes".semiAutoSplice.sequence.status.seqActive;
   "Unit1.Em2.ControlNodes".semiAutoSplice."step".transition1[3091] := ("Unit1.Em2.ControlNodes".semiAutoSplice.sequence.status.currentStep = #JOB_30_STEP_91) AND "Unit1.Em2.ControlNodes".semiAutoSplice.sequence.status.seqActive;
   #statTonTimer[3091].TON(IN := ("Unit1.Em2.ControlNodes".semiAutoSplice.sequence.status.currentStep = #JOB_30_STEP_91) AND "Unit1.Em2.ControlNodes".semiAutoSplice.sequence.status.seqActive AND "Unit1.Em2.ControlNodes".semiAutoSplice."step".transition1[3091],
                           PT := #SeqDelayTime);
   IF #statTonTimer[3091].Q THEN
       "Unit1.Em2.ControlNodes".semiAutoSplice.sequence.status.nextStep := #JOB_30_STEP_92;
   END_IF;
END_REGION

REGION Network 242: Step[3092] : BTM Unlink TOP Link
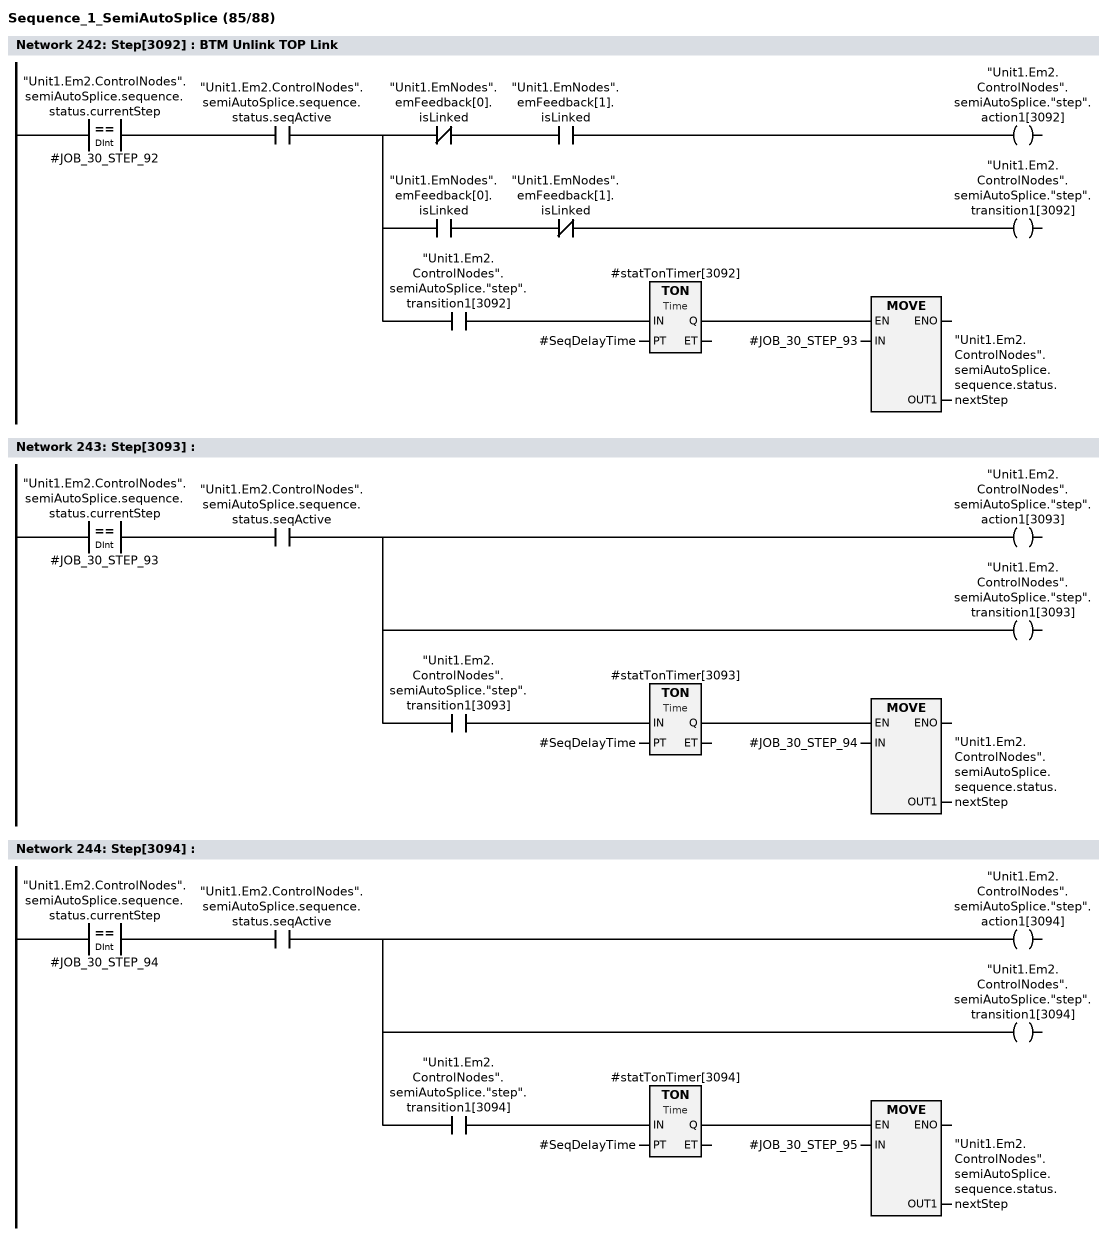
   RUNG wire#powerrail
      { S7_Templates := "SrcType := DInt" } EQ_Contact(in1 := "Unit1.Em2.ControlNodes".semiAutoSplice.sequence.status.currentStep, in2 := #JOB_30_STEP_92)
      Contact( "Unit1.Em2.ControlNodes".semiAutoSplice.sequence.status.seqActive )
      wire#w1
      I_Contact( "Unit1.EmNodes".emFeedback[0].isLinked )
      Contact( "Unit1.EmNodes".emFeedback[1].isLinked )
      Coil( "Unit1.Em2.ControlNodes".semiAutoSplice."step".action1[3092] )
   END_RUNG
   RUNG wire#w1
      Contact( "Unit1.EmNodes".emFeedback[0].isLinked )
      I_Contact( "Unit1.EmNodes".emFeedback[1].isLinked )
      Coil( "Unit1.Em2.ControlNodes".semiAutoSplice."step".transition1[3092] )
   END_RUNG
   RUNG wire#w1
      Contact( "Unit1.Em2.ControlNodes".semiAutoSplice."step".transition1[3092] )
      { S7_Templates := "time_type := Time" } #statTonTimer[3092].TON(pt := #SeqDelayTime, et =>)
      Move(in := #JOB_30_STEP_93, out1 => "Unit1.Em2.ControlNodes".semiAutoSplice.sequence.status.nextStep)
   END_RUNG
   // the same network as SCL:
   #_w1 := ("Unit1.Em2.ControlNodes".semiAutoSplice.sequence.status.currentStep = #JOB_30_STEP_92) AND "Unit1.Em2.ControlNodes".semiAutoSplice.sequence.status.seqActive;
   "Unit1.Em2.ControlNodes".semiAutoSplice."step".action1[3092] := #_w1 AND NOT "Unit1.EmNodes".emFeedback[0].isLinked AND "Unit1.EmNodes".emFeedback[1].isLinked;
   "Unit1.Em2.ControlNodes".semiAutoSplice."step".transition1[3092] := #_w1 AND "Unit1.EmNodes".emFeedback[0].isLinked AND NOT "Unit1.EmNodes".emFeedback[1].isLinked;
   #statTonTimer[3092].TON(IN := #_w1 AND "Unit1.Em2.ControlNodes".semiAutoSplice."step".transition1[3092],
                           PT := #SeqDelayTime);
   IF #statTonTimer[3092].Q THEN
       "Unit1.Em2.ControlNodes".semiAutoSplice.sequence.status.nextStep := #JOB_30_STEP_93;
   END_IF;
END_REGION

REGION Network 243: Step[3093] :
   RUNG wire#powerrail
      { S7_Templates := "SrcType := DInt" } EQ_Contact(in1 := "Unit1.Em2.ControlNodes".semiAutoSplice.sequence.status.currentStep, in2 := #JOB_30_STEP_93)
      Contact( "Unit1.Em2.ControlNodes".semiAutoSplice.sequence.status.seqActive )
      wire#w1
      Coil( "Unit1.Em2.ControlNodes".semiAutoSplice."step".action1[3093] )
   END_RUNG
   RUNG wire#w1
      Coil( "Unit1.Em2.ControlNodes".semiAutoSplice."step".transition1[3093] )
   END_RUNG
   RUNG wire#w1
      Contact( "Unit1.Em2.ControlNodes".semiAutoSplice."step".transition1[3093] )
      { S7_Templates := "time_type := Time" } #statTonTimer[3093].TON(pt := #SeqDelayTime, et =>)
      Move(in := #JOB_30_STEP_94, out1 => "Unit1.Em2.ControlNodes".semiAutoSplice.sequence.status.nextStep)
   END_RUNG
   // the same network as SCL:
   "Unit1.Em2.ControlNodes".semiAutoSplice."step".action1[3093] := ("Unit1.Em2.ControlNodes".semiAutoSplice.sequence.status.currentStep = #JOB_30_STEP_93) AND "Unit1.Em2.ControlNodes".semiAutoSplice.sequence.status.seqActive;
   "Unit1.Em2.ControlNodes".semiAutoSplice."step".transition1[3093] := ("Unit1.Em2.ControlNodes".semiAutoSplice.sequence.status.currentStep = #JOB_30_STEP_93) AND "Unit1.Em2.ControlNodes".semiAutoSplice.sequence.status.seqActive;
   #statTonTimer[3093].TON(IN := ("Unit1.Em2.ControlNodes".semiAutoSplice.sequence.status.currentStep = #JOB_30_STEP_93) AND "Unit1.Em2.ControlNodes".semiAutoSplice.sequence.status.seqActive AND "Unit1.Em2.ControlNodes".semiAutoSplice."step".transition1[3093],
                           PT := #SeqDelayTime);
   IF #statTonTimer[3093].Q THEN
       "Unit1.Em2.ControlNodes".semiAutoSplice.sequence.status.nextStep := #JOB_30_STEP_94;
   END_IF;
END_REGION

REGION Network 244: Step[3094] :
   RUNG wire#powerrail
      { S7_Templates := "SrcType := DInt" } EQ_Contact(in1 := "Unit1.Em2.ControlNodes".semiAutoSplice.sequence.status.currentStep, in2 := #JOB_30_STEP_94)
      Contact( "Unit1.Em2.ControlNodes".semiAutoSplice.sequence.status.seqActive )
      wire#w1
      Coil( "Unit1.Em2.ControlNodes".semiAutoSplice."step".action1[3094] )
   END_RUNG
   RUNG wire#w1
      Coil( "Unit1.Em2.ControlNodes".semiAutoSplice."step".transition1[3094] )
   END_RUNG
   RUNG wire#w1
      Contact( "Unit1.Em2.ControlNodes".semiAutoSplice."step".transition1[3094] )
      { S7_Templates := "time_type := Time" } #statTonTimer[3094].TON(pt := #SeqDelayTime, et =>)
      Move(in := #JOB_30_STEP_95, out1 => "Unit1.Em2.ControlNodes".semiAutoSplice.sequence.status.nextStep)
   END_RUNG
   // the same network as SCL:
   "Unit1.Em2.ControlNodes".semiAutoSplice."step".action1[3094] := ("Unit1.Em2.ControlNodes".semiAutoSplice.sequence.status.currentStep = #JOB_30_STEP_94) AND "Unit1.Em2.ControlNodes".semiAutoSplice.sequence.status.seqActive;
   "Unit1.Em2.ControlNodes".semiAutoSplice."step".transition1[3094] := ("Unit1.Em2.ControlNodes".semiAutoSplice.sequence.status.currentStep = #JOB_30_STEP_94) AND "Unit1.Em2.ControlNodes".semiAutoSplice.sequence.status.seqActive;
   #statTonTimer[3094].TON(IN := ("Unit1.Em2.ControlNodes".semiAutoSplice.sequence.status.currentStep = #JOB_30_STEP_94) AND "Unit1.Em2.ControlNodes".semiAutoSplice.sequence.status.seqActive AND "Unit1.Em2.ControlNodes".semiAutoSplice."step".transition1[3094],
                           PT := #SeqDelayTime);
   IF #statTonTimer[3094].Q THEN
       "Unit1.Em2.ControlNodes".semiAutoSplice.sequence.status.nextStep := #JOB_30_STEP_95;
   END_IF;
END_REGION

REGION Network 245: Step[3095] :
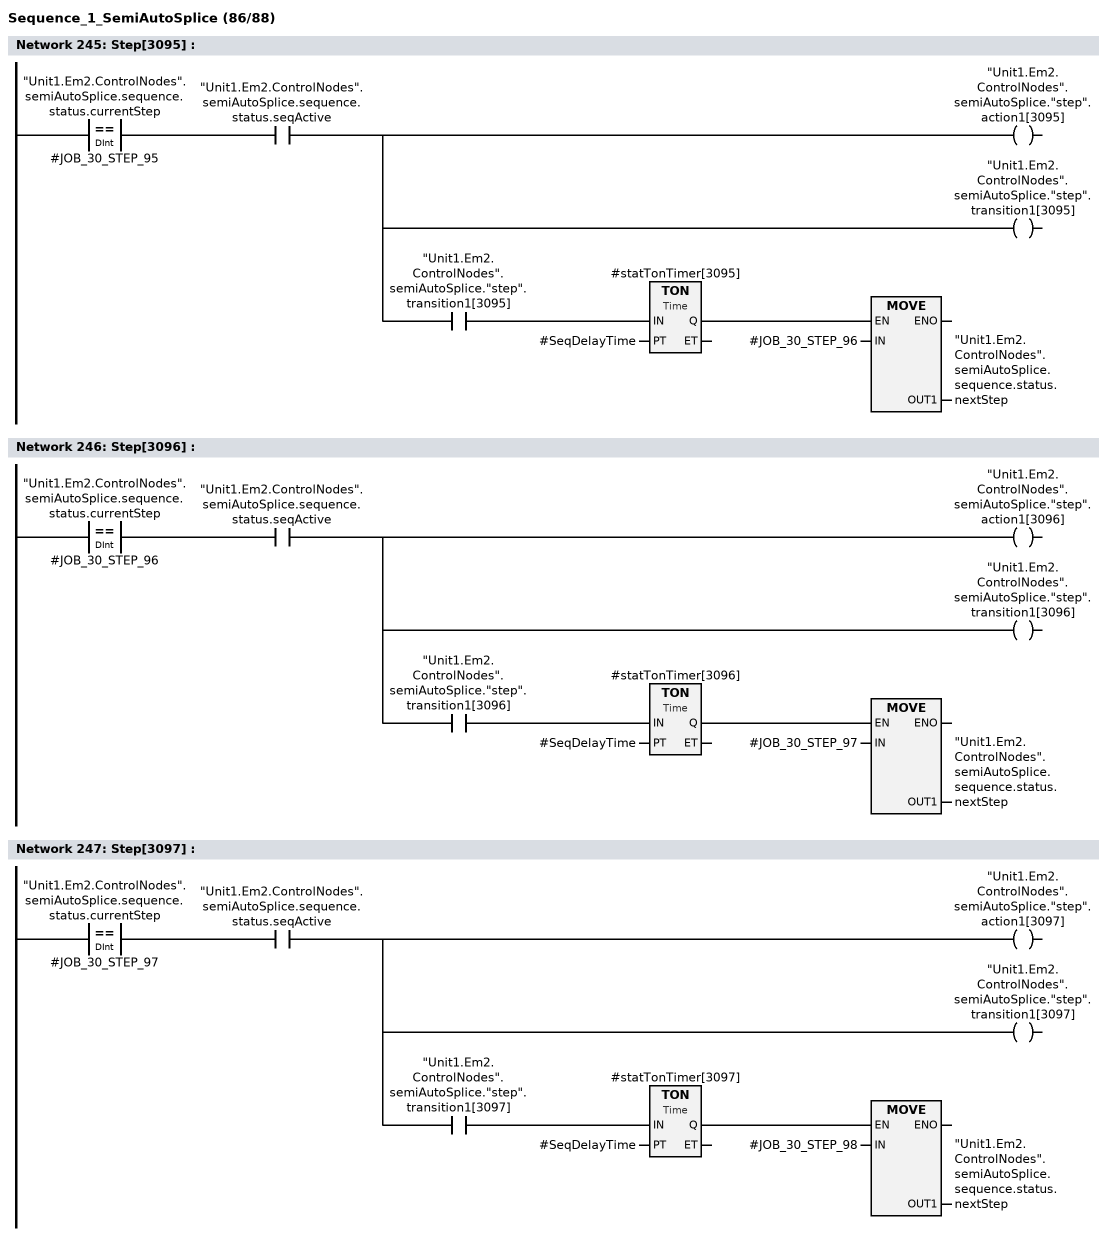
   RUNG wire#powerrail
      { S7_Templates := "SrcType := DInt" } EQ_Contact(in1 := "Unit1.Em2.ControlNodes".semiAutoSplice.sequence.status.currentStep, in2 := #JOB_30_STEP_95)
      Contact( "Unit1.Em2.ControlNodes".semiAutoSplice.sequence.status.seqActive )
      wire#w1
      Coil( "Unit1.Em2.ControlNodes".semiAutoSplice."step".action1[3095] )
   END_RUNG
   RUNG wire#w1
      Coil( "Unit1.Em2.ControlNodes".semiAutoSplice."step".transition1[3095] )
   END_RUNG
   RUNG wire#w1
      Contact( "Unit1.Em2.ControlNodes".semiAutoSplice."step".transition1[3095] )
      { S7_Templates := "time_type := Time" } #statTonTimer[3095].TON(pt := #SeqDelayTime, et =>)
      Move(in := #JOB_30_STEP_96, out1 => "Unit1.Em2.ControlNodes".semiAutoSplice.sequence.status.nextStep)
   END_RUNG
   // the same network as SCL:
   "Unit1.Em2.ControlNodes".semiAutoSplice."step".action1[3095] := ("Unit1.Em2.ControlNodes".semiAutoSplice.sequence.status.currentStep = #JOB_30_STEP_95) AND "Unit1.Em2.ControlNodes".semiAutoSplice.sequence.status.seqActive;
   "Unit1.Em2.ControlNodes".semiAutoSplice."step".transition1[3095] := ("Unit1.Em2.ControlNodes".semiAutoSplice.sequence.status.currentStep = #JOB_30_STEP_95) AND "Unit1.Em2.ControlNodes".semiAutoSplice.sequence.status.seqActive;
   #statTonTimer[3095].TON(IN := ("Unit1.Em2.ControlNodes".semiAutoSplice.sequence.status.currentStep = #JOB_30_STEP_95) AND "Unit1.Em2.ControlNodes".semiAutoSplice.sequence.status.seqActive AND "Unit1.Em2.ControlNodes".semiAutoSplice."step".transition1[3095],
                           PT := #SeqDelayTime);
   IF #statTonTimer[3095].Q THEN
       "Unit1.Em2.ControlNodes".semiAutoSplice.sequence.status.nextStep := #JOB_30_STEP_96;
   END_IF;
END_REGION

REGION Network 246: Step[3096] :
   RUNG wire#powerrail
      { S7_Templates := "SrcType := DInt" } EQ_Contact(in1 := "Unit1.Em2.ControlNodes".semiAutoSplice.sequence.status.currentStep, in2 := #JOB_30_STEP_96)
      Contact( "Unit1.Em2.ControlNodes".semiAutoSplice.sequence.status.seqActive )
      wire#w1
      Coil( "Unit1.Em2.ControlNodes".semiAutoSplice."step".action1[3096] )
   END_RUNG
   RUNG wire#w1
      Coil( "Unit1.Em2.ControlNodes".semiAutoSplice."step".transition1[3096] )
   END_RUNG
   RUNG wire#w1
      Contact( "Unit1.Em2.ControlNodes".semiAutoSplice."step".transition1[3096] )
      { S7_Templates := "time_type := Time" } #statTonTimer[3096].TON(pt := #SeqDelayTime, et =>)
      Move(in := #JOB_30_STEP_97, out1 => "Unit1.Em2.ControlNodes".semiAutoSplice.sequence.status.nextStep)
   END_RUNG
   // the same network as SCL:
   "Unit1.Em2.ControlNodes".semiAutoSplice."step".action1[3096] := ("Unit1.Em2.ControlNodes".semiAutoSplice.sequence.status.currentStep = #JOB_30_STEP_96) AND "Unit1.Em2.ControlNodes".semiAutoSplice.sequence.status.seqActive;
   "Unit1.Em2.ControlNodes".semiAutoSplice."step".transition1[3096] := ("Unit1.Em2.ControlNodes".semiAutoSplice.sequence.status.currentStep = #JOB_30_STEP_96) AND "Unit1.Em2.ControlNodes".semiAutoSplice.sequence.status.seqActive;
   #statTonTimer[3096].TON(IN := ("Unit1.Em2.ControlNodes".semiAutoSplice.sequence.status.currentStep = #JOB_30_STEP_96) AND "Unit1.Em2.ControlNodes".semiAutoSplice.sequence.status.seqActive AND "Unit1.Em2.ControlNodes".semiAutoSplice."step".transition1[3096],
                           PT := #SeqDelayTime);
   IF #statTonTimer[3096].Q THEN
       "Unit1.Em2.ControlNodes".semiAutoSplice.sequence.status.nextStep := #JOB_30_STEP_97;
   END_IF;
END_REGION

REGION Network 247: Step[3097] :
   RUNG wire#powerrail
      { S7_Templates := "SrcType := DInt" } EQ_Contact(in1 := "Unit1.Em2.ControlNodes".semiAutoSplice.sequence.status.currentStep, in2 := #JOB_30_STEP_97)
      Contact( "Unit1.Em2.ControlNodes".semiAutoSplice.sequence.status.seqActive )
      wire#w1
      Coil( "Unit1.Em2.ControlNodes".semiAutoSplice."step".action1[3097] )
   END_RUNG
   RUNG wire#w1
      Coil( "Unit1.Em2.ControlNodes".semiAutoSplice."step".transition1[3097] )
   END_RUNG
   RUNG wire#w1
      Contact( "Unit1.Em2.ControlNodes".semiAutoSplice."step".transition1[3097] )
      { S7_Templates := "time_type := Time" } #statTonTimer[3097].TON(pt := #SeqDelayTime, et =>)
      Move(in := #JOB_30_STEP_98, out1 => "Unit1.Em2.ControlNodes".semiAutoSplice.sequence.status.nextStep)
   END_RUNG
   // the same network as SCL:
   "Unit1.Em2.ControlNodes".semiAutoSplice."step".action1[3097] := ("Unit1.Em2.ControlNodes".semiAutoSplice.sequence.status.currentStep = #JOB_30_STEP_97) AND "Unit1.Em2.ControlNodes".semiAutoSplice.sequence.status.seqActive;
   "Unit1.Em2.ControlNodes".semiAutoSplice."step".transition1[3097] := ("Unit1.Em2.ControlNodes".semiAutoSplice.sequence.status.currentStep = #JOB_30_STEP_97) AND "Unit1.Em2.ControlNodes".semiAutoSplice.sequence.status.seqActive;
   #statTonTimer[3097].TON(IN := ("Unit1.Em2.ControlNodes".semiAutoSplice.sequence.status.currentStep = #JOB_30_STEP_97) AND "Unit1.Em2.ControlNodes".semiAutoSplice.sequence.status.seqActive AND "Unit1.Em2.ControlNodes".semiAutoSplice."step".transition1[3097],
                           PT := #SeqDelayTime);
   IF #statTonTimer[3097].Q THEN
       "Unit1.Em2.ControlNodes".semiAutoSplice.sequence.status.nextStep := #JOB_30_STEP_98;
   END_IF;
END_REGION

REGION Network 248: Step[3098] :
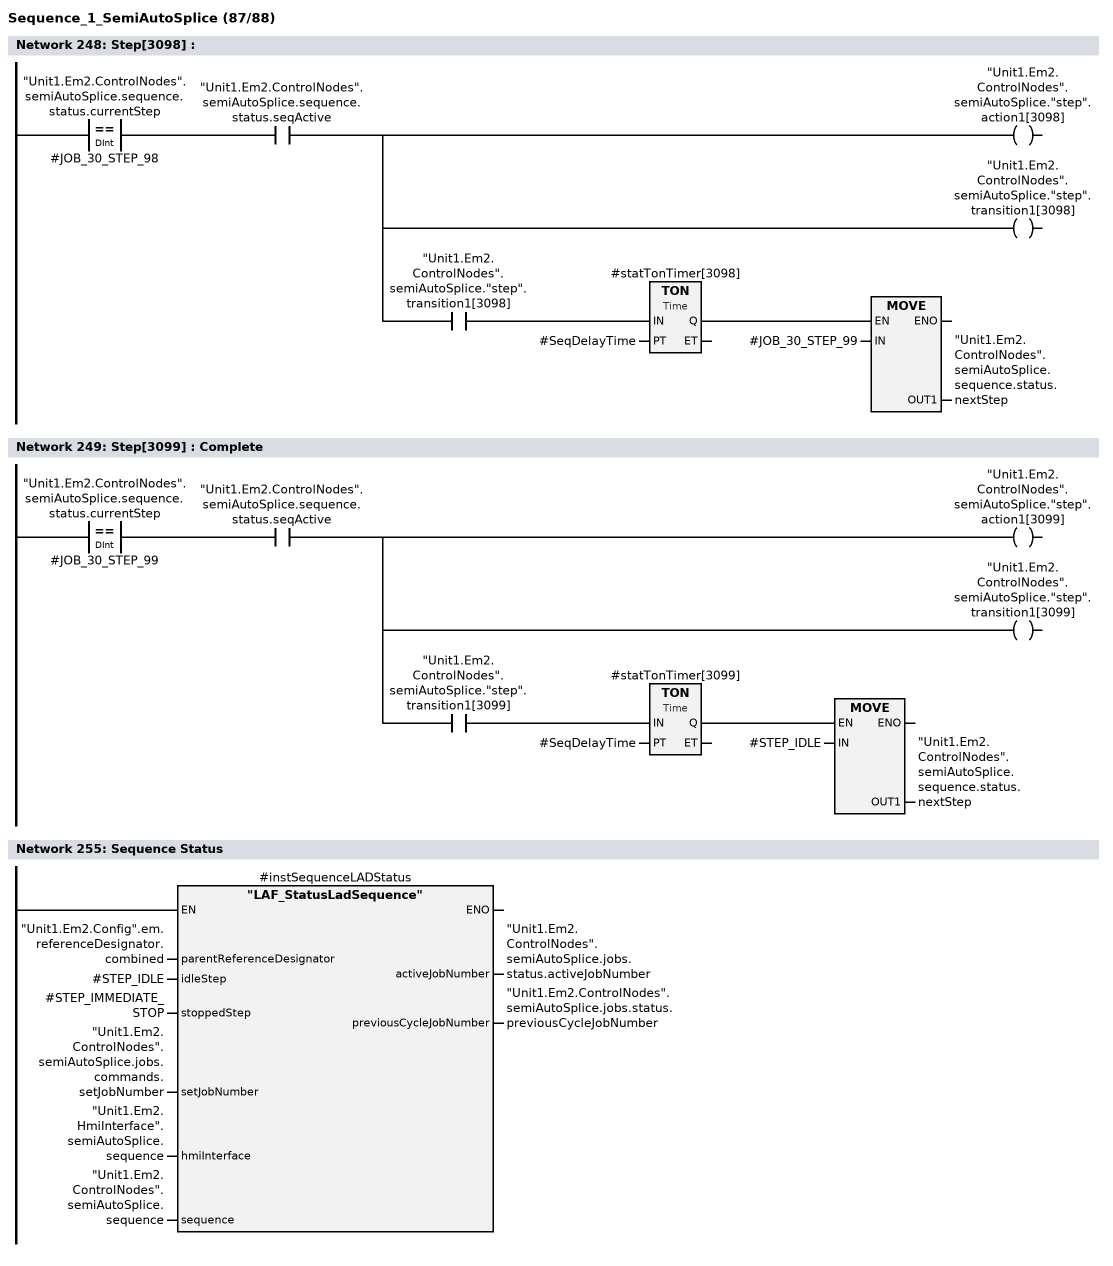
   RUNG wire#powerrail
      { S7_Templates := "SrcType := DInt" } EQ_Contact(in1 := "Unit1.Em2.ControlNodes".semiAutoSplice.sequence.status.currentStep, in2 := #JOB_30_STEP_98)
      Contact( "Unit1.Em2.ControlNodes".semiAutoSplice.sequence.status.seqActive )
      wire#w1
      Coil( "Unit1.Em2.ControlNodes".semiAutoSplice."step".action1[3098] )
   END_RUNG
   RUNG wire#w1
      Coil( "Unit1.Em2.ControlNodes".semiAutoSplice."step".transition1[3098] )
   END_RUNG
   RUNG wire#w1
      Contact( "Unit1.Em2.ControlNodes".semiAutoSplice."step".transition1[3098] )
      { S7_Templates := "time_type := Time" } #statTonTimer[3098].TON(pt := #SeqDelayTime, et =>)
      Move(in := #JOB_30_STEP_99, out1 => "Unit1.Em2.ControlNodes".semiAutoSplice.sequence.status.nextStep)
   END_RUNG
   // the same network as SCL:
   "Unit1.Em2.ControlNodes".semiAutoSplice."step".action1[3098] := ("Unit1.Em2.ControlNodes".semiAutoSplice.sequence.status.currentStep = #JOB_30_STEP_98) AND "Unit1.Em2.ControlNodes".semiAutoSplice.sequence.status.seqActive;
   "Unit1.Em2.ControlNodes".semiAutoSplice."step".transition1[3098] := ("Unit1.Em2.ControlNodes".semiAutoSplice.sequence.status.currentStep = #JOB_30_STEP_98) AND "Unit1.Em2.ControlNodes".semiAutoSplice.sequence.status.seqActive;
   #statTonTimer[3098].TON(IN := ("Unit1.Em2.ControlNodes".semiAutoSplice.sequence.status.currentStep = #JOB_30_STEP_98) AND "Unit1.Em2.ControlNodes".semiAutoSplice.sequence.status.seqActive AND "Unit1.Em2.ControlNodes".semiAutoSplice."step".transition1[3098],
                           PT := #SeqDelayTime);
   IF #statTonTimer[3098].Q THEN
       "Unit1.Em2.ControlNodes".semiAutoSplice.sequence.status.nextStep := #JOB_30_STEP_99;
   END_IF;
END_REGION

REGION Network 249: Step[3099] : Complete
   RUNG wire#powerrail
      { S7_Templates := "SrcType := DInt" } EQ_Contact(in1 := "Unit1.Em2.ControlNodes".semiAutoSplice.sequence.status.currentStep, in2 := #JOB_30_STEP_99)
      Contact( "Unit1.Em2.ControlNodes".semiAutoSplice.sequence.status.seqActive )
      wire#w1
      Coil( "Unit1.Em2.ControlNodes".semiAutoSplice."step".action1[3099] )
   END_RUNG
   RUNG wire#w1
      Coil( "Unit1.Em2.ControlNodes".semiAutoSplice."step".transition1[3099] )
   END_RUNG
   RUNG wire#w1
      Contact( "Unit1.Em2.ControlNodes".semiAutoSplice."step".transition1[3099] )
      { S7_Templates := "time_type := Time" } #statTonTimer[3099].TON(pt := #SeqDelayTime, et =>)
      Move(in := #STEP_IDLE, out1 => "Unit1.Em2.ControlNodes".semiAutoSplice.sequence.status.nextStep)
   END_RUNG
   // the same network as SCL:
   "Unit1.Em2.ControlNodes".semiAutoSplice."step".action1[3099] := ("Unit1.Em2.ControlNodes".semiAutoSplice.sequence.status.currentStep = #JOB_30_STEP_99) AND "Unit1.Em2.ControlNodes".semiAutoSplice.sequence.status.seqActive;
   "Unit1.Em2.ControlNodes".semiAutoSplice."step".transition1[3099] := ("Unit1.Em2.ControlNodes".semiAutoSplice.sequence.status.currentStep = #JOB_30_STEP_99) AND "Unit1.Em2.ControlNodes".semiAutoSplice.sequence.status.seqActive;
   #statTonTimer[3099].TON(IN := ("Unit1.Em2.ControlNodes".semiAutoSplice.sequence.status.currentStep = #JOB_30_STEP_99) AND "Unit1.Em2.ControlNodes".semiAutoSplice.sequence.status.seqActive AND "Unit1.Em2.ControlNodes".semiAutoSplice."step".transition1[3099],
                           PT := #SeqDelayTime);
   IF #statTonTimer[3099].Q THEN
       "Unit1.Em2.ControlNodes".semiAutoSplice.sequence.status.nextStep := #STEP_IDLE;
   END_IF;
END_REGION

REGION Network 251: *************** IMMEDIATE STOP **************************
END_REGION

REGION Network 252: Immediate Stop
END_REGION

REGION Network 254: *************** Status updates **************************
END_REGION

REGION Network 255: Sequence Status
   RUNG wire#powerrail
      #instSequenceLADStatus(parentReferenceDesignator := "Unit1.Em2.Config".em.referenceDesignator.combined, idleStep := #STEP_IDLE, stoppedStep := #STEP_IMMEDIATE_STOP, setJobNumber := "Unit1.Em2.ControlNodes".semiAutoSplice.jobs.commands.setJobNumber, hmiInterface := "Unit1.Em2.HmiInterface".semiAutoSplice.sequence, sequence := "Unit1.Em2.ControlNodes".semiAutoSplice.sequence, activeJobNumber => "Unit1.Em2.ControlNodes".semiAutoSplice.jobs.status.activeJobNumber, previousCycleJobNumber => "Unit1.Em2.ControlNodes".semiAutoSplice.jobs.status.previousCycleJobNumber)
   END_RUNG
   // the same network as SCL:
   #instSequenceLADStatus(parentReferenceDesignator := "Unit1.Em2.Config".em.referenceDesignator.combined,   // "LAF_StatusLadSequence"
                          idleStep := #STEP_IDLE,
                          stoppedStep := #STEP_IMMEDIATE_STOP,
                          setJobNumber := "Unit1.Em2.ControlNodes".semiAutoSplice.jobs.commands.setJobNumber,
                          hmiInterface := "Unit1.Em2.HmiInterface".semiAutoSplice.sequence,
                          sequence := "Unit1.Em2.ControlNodes".semiAutoSplice.sequence,
                          activeJobNumber => "Unit1.Em2.ControlNodes".semiAutoSplice.jobs.status.activeJobNumber,
                          previousCycleJobNumber => "Unit1.Em2.ControlNodes".semiAutoSplice.jobs.status.previousCycleJobNumber);
END_REGION

